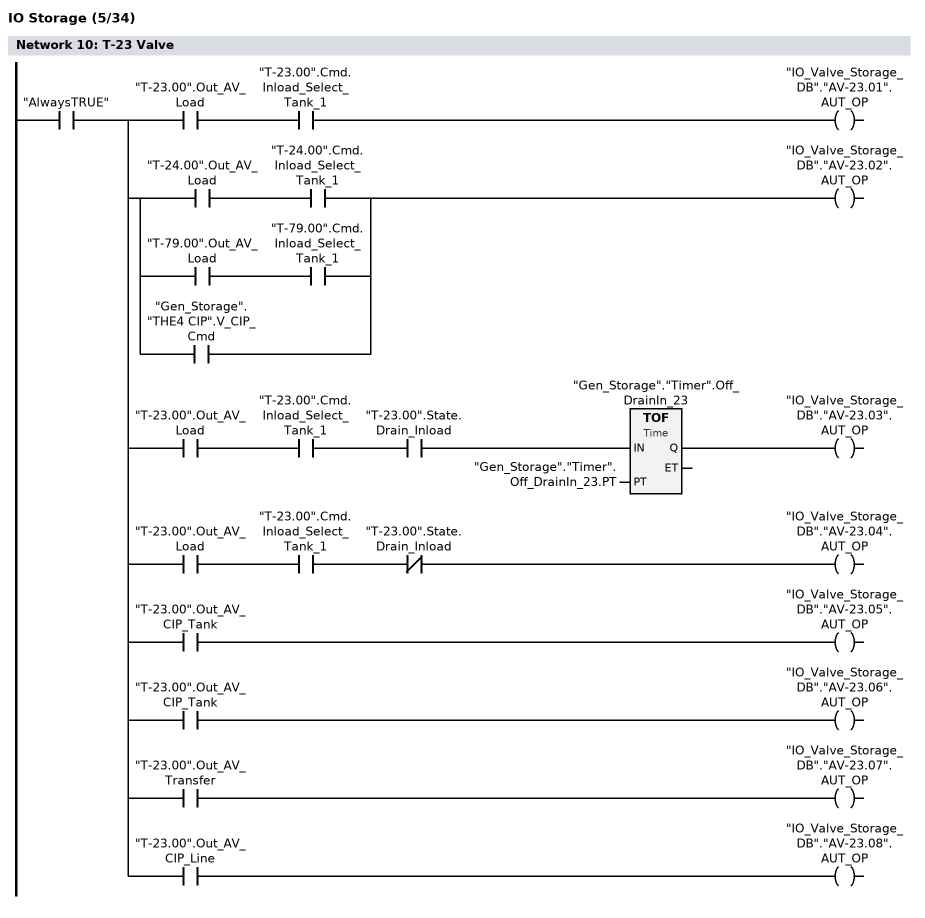
   RUNG wire#powerrail
      Contact( "AlwaysTRUE" )
      wire#w1
      Contact( "T-23.00".Out_AV_Load )
      Contact( "T-23.00".Cmd.Inload_Select_Tank_1 )
      Coil( "IO_Valve_Storage_DB"."AV-23.01".AUT_OP )
   END_RUNG
   RUNG wire#w1
      Contact( "T-24.00".Out_AV_Load )
      Contact( "T-24.00".Cmd.Inload_Select_Tank_1 )
      wire#w2
      Coil( "IO_Valve_Storage_DB"."AV-23.02".AUT_OP )
   END_RUNG
   RUNG wire#w1
      Contact( "T-79.00".Out_AV_Load )
      Contact( "T-79.00".Cmd.Inload_Select_Tank_1 )
   END_RUNG wire#w2
   RUNG wire#w1
      Contact( "Gen_Storage"."THE4 CIP".V_CIP_Cmd )
   END_RUNG wire#w2
   RUNG wire#w1
      Contact( "T-23.00".Out_AV_Load )
      Contact( "T-23.00".Cmd.Inload_Select_Tank_1 )
      Contact( "T-23.00".State.Drain_Inload )
      { S7_Templates := "time_type := Time" } "Gen_Storage"."Timer".Off_DrainIn_23.TOF(pt := "Gen_Storage"."Timer".Off_DrainIn_23.PT, et =>)
      Coil( "IO_Valve_Storage_DB"."AV-23.03".AUT_OP )
   END_RUNG
   RUNG wire#w1
      Contact( "T-23.00".Out_AV_Load )
      Contact( "T-23.00".Cmd.Inload_Select_Tank_1 )
      I_Contact( "T-23.00".State.Drain_Inload )
      Coil( "IO_Valve_Storage_DB"."AV-23.04".AUT_OP )
   END_RUNG
   RUNG wire#w1
      Contact( "T-23.00".Out_AV_CIP_Tank )
      Coil( "IO_Valve_Storage_DB"."AV-23.05".AUT_OP )
   END_RUNG
   RUNG wire#w1
      Contact( "T-23.00".Out_AV_CIP_Tank )
      Coil( "IO_Valve_Storage_DB"."AV-23.06".AUT_OP )
   END_RUNG
   RUNG wire#w1
      Contact( "T-23.00".Out_AV_Transfer )
      Coil( "IO_Valve_Storage_DB"."AV-23.07".AUT_OP )
   END_RUNG
   RUNG wire#w1
      Contact( "T-23.00".Out_AV_CIP_Line )
      Coil( "IO_Valve_Storage_DB"."AV-23.08".AUT_OP )
   END_RUNG
   // the same network as SCL:
   "IO_Valve_Storage_DB"."AV-23.01".AUT_OP := "AlwaysTRUE" AND "T-23.00".Out_AV_Load AND "T-23.00".Cmd.Inload_Select_Tank_1;
   "IO_Valve_Storage_DB"."AV-23.02".AUT_OP := "AlwaysTRUE" AND (("T-24.00".Out_AV_Load AND "T-24.00".Cmd.Inload_Select_Tank_1) OR ("T-79.00".Out_AV_Load AND "T-79.00".Cmd.Inload_Select_Tank_1) OR "Gen_Storage"."THE4 CIP".V_CIP_Cmd);
   "Gen_Storage"."Timer".Off_DrainIn_23.TOF(IN := "AlwaysTRUE" AND "T-23.00".Out_AV_Load AND "T-23.00".Cmd.Inload_Select_Tank_1 AND "T-23.00".State.Drain_Inload,
                           PT := "Gen_Storage"."Timer".Off_DrainIn_23.PT);
   "IO_Valve_Storage_DB"."AV-23.03".AUT_OP := "Gen_Storage"."Timer".Off_DrainIn_23.Q;
   "IO_Valve_Storage_DB"."AV-23.04".AUT_OP := "AlwaysTRUE" AND "T-23.00".Out_AV_Load AND "T-23.00".Cmd.Inload_Select_Tank_1 AND NOT "T-23.00".State.Drain_Inload;
   "IO_Valve_Storage_DB"."AV-23.05".AUT_OP := "AlwaysTRUE" AND "T-23.00".Out_AV_CIP_Tank;
   "IO_Valve_Storage_DB"."AV-23.06".AUT_OP := "AlwaysTRUE" AND "T-23.00".Out_AV_CIP_Tank;
   "IO_Valve_Storage_DB"."AV-23.07".AUT_OP := "AlwaysTRUE" AND "T-23.00".Out_AV_Transfer;
   "IO_Valve_Storage_DB"."AV-23.08".AUT_OP := "AlwaysTRUE" AND "T-23.00".Out_AV_CIP_Line;
END_REGION

REGION Network 12: T-24.00 ST-07
   // Inload 1 : THE 4
   // Inload 2 : THE 1
   // Inload 3 : THE 5
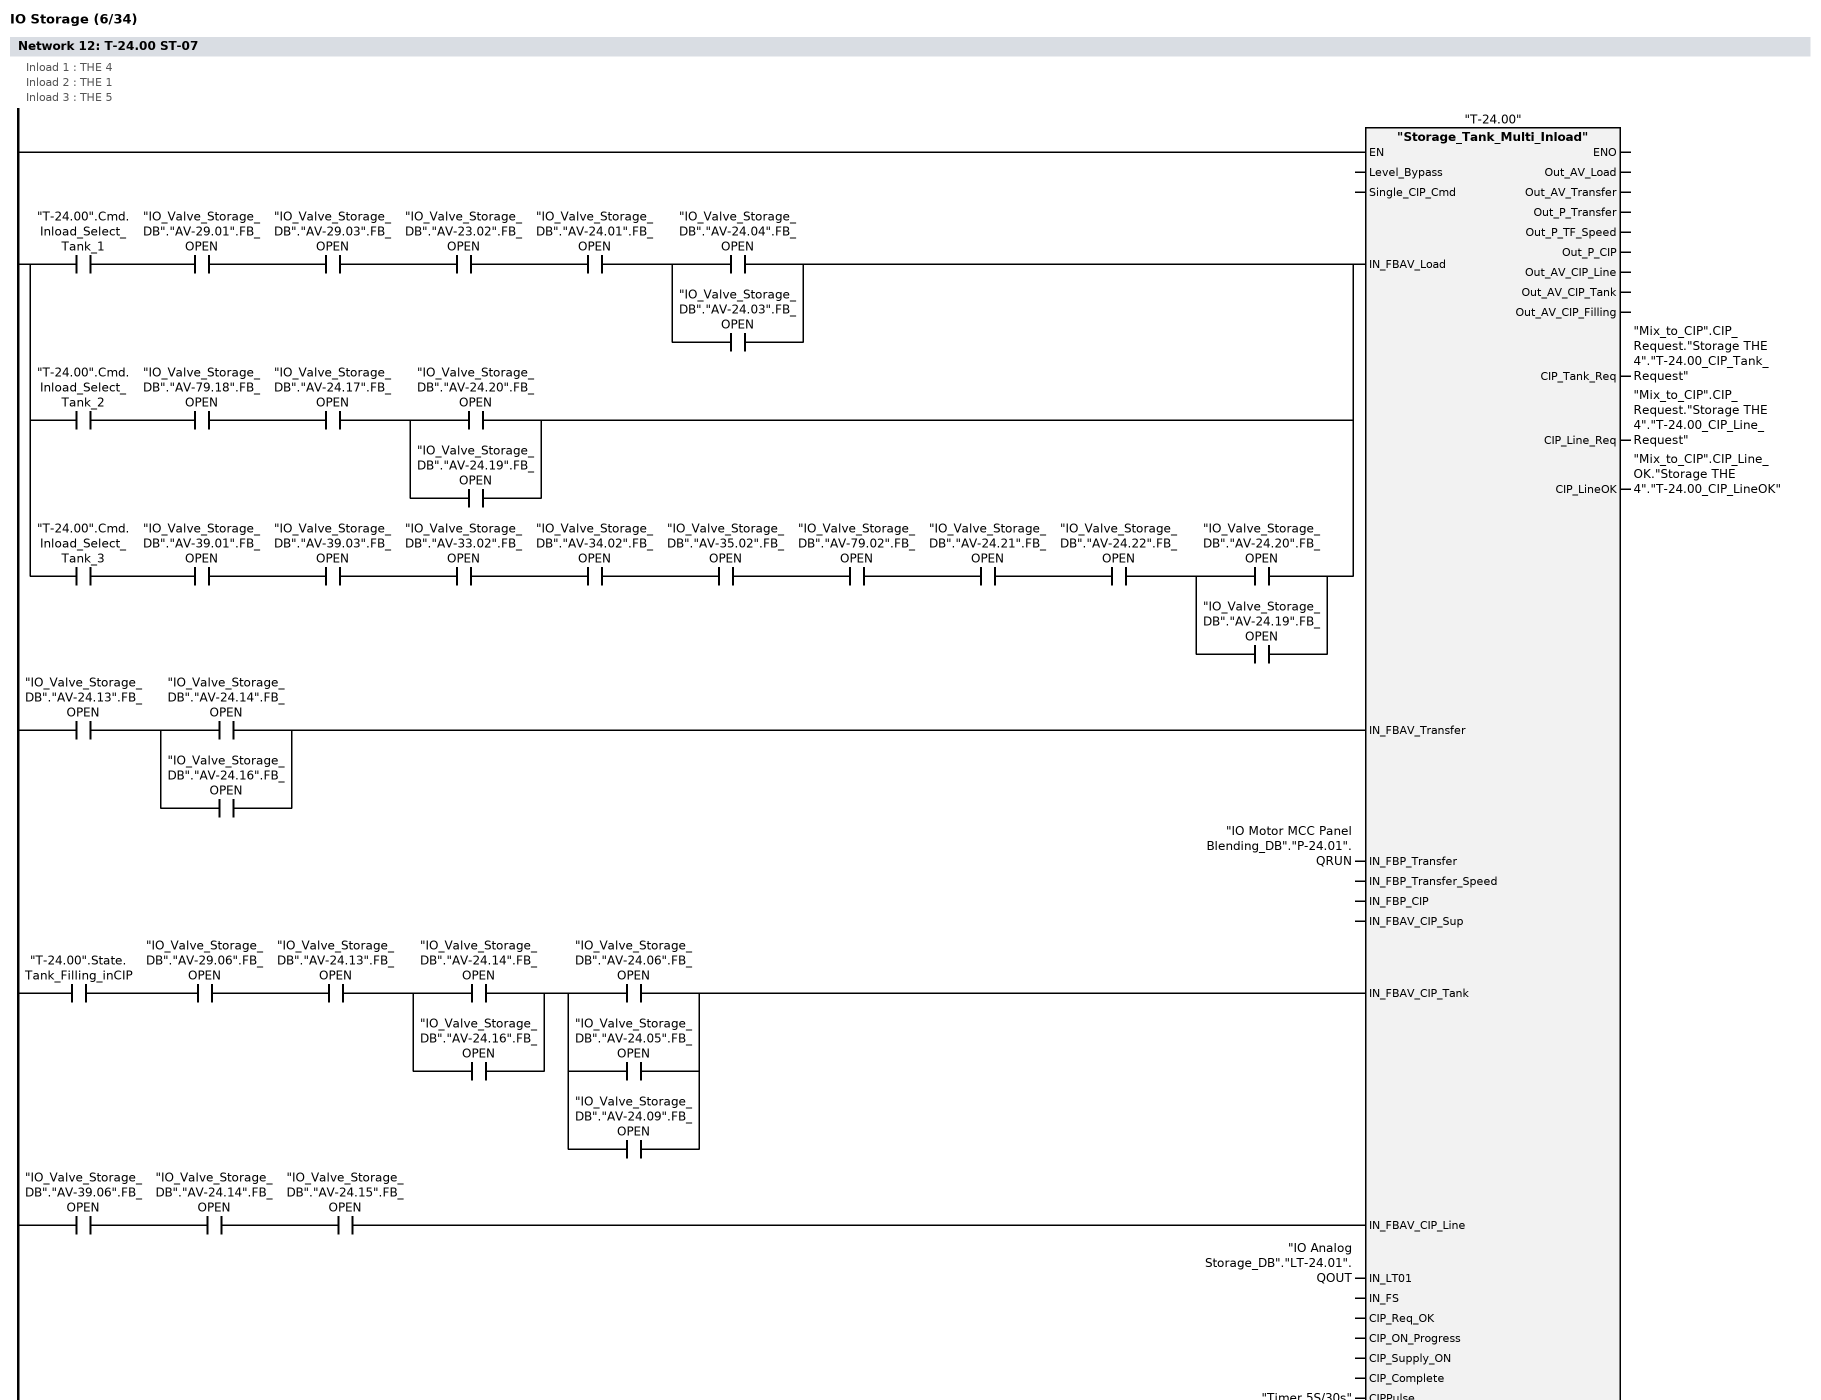
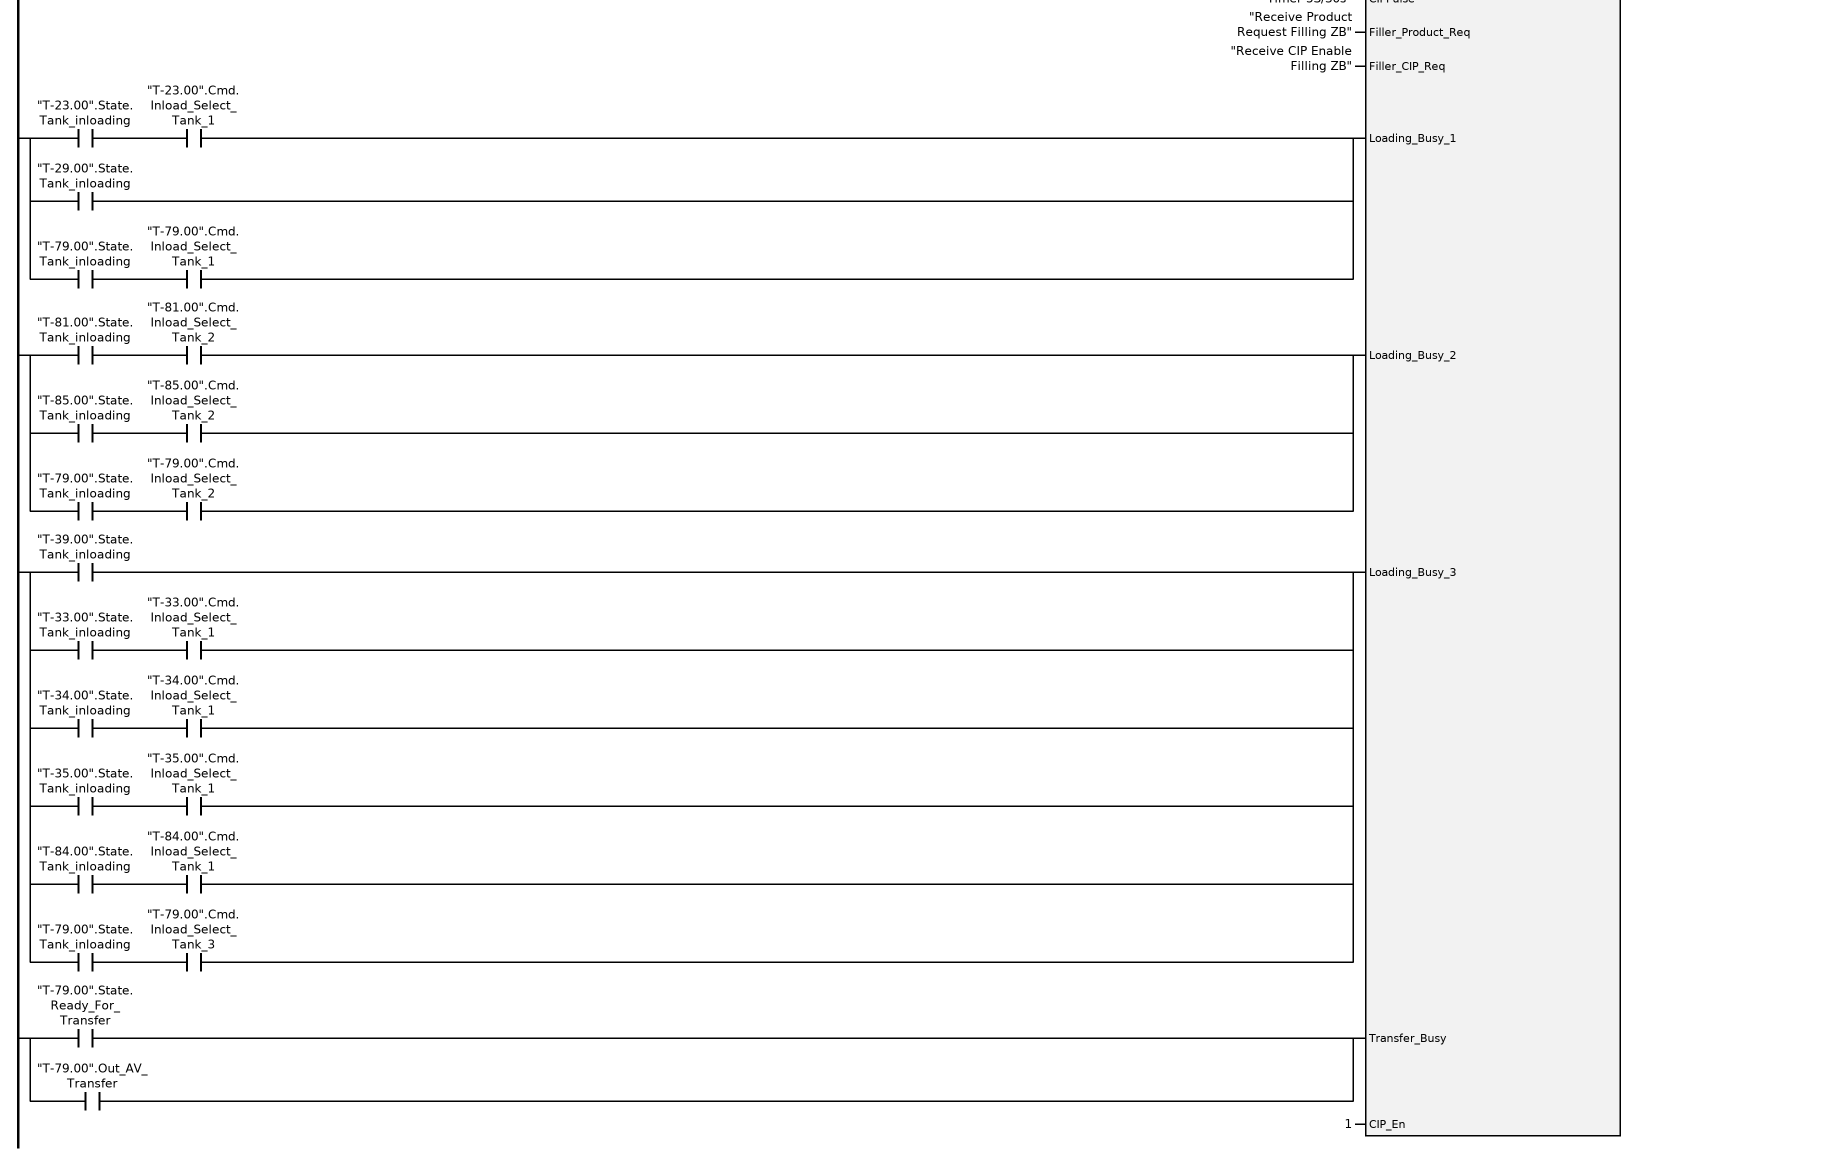
   RUNG wire#powerrail
      "T-24.00"(IN_FBAV_Load := wire#w4, IN_FBAV_Transfer := wire#w6, IN_FBAV_CIP_Tank := wire#w9, IN_FBAV_CIP_Line := wire#w10, Loading_Busy_1 := wire#w11, Loading_Busy_2 := wire#w12, Loading_Busy_3 := wire#w13, Transfer_Busy := wire#w14, Level_Bypass :=, Single_CIP_Cmd :=, IN_FBP_Transfer := "IO Motor MCC Panel Blending_DB"."P-24.01".QRUN, IN_FBP_Transfer_Speed :=, IN_FBP_CIP :=, IN_FBAV_CIP_Sup :=, IN_LT01 := "IO Analog Storage_DB"."LT-24.01".QOUT, IN_FS :=, CIP_Req_OK :=, CIP_ON_Progress :=, CIP_Supply_ON :=, CIP_Complete :=, CIPPulse := "Timer 5S/30s", Filler_Product_Req := "Receive Product Request Filling ZB", Filler_CIP_Req := "Receive CIP Enable Filling ZB", CIP_En := 1, Out_AV_Load =>, Out_AV_Transfer =>, Out_P_Transfer =>, Out_P_TF_Speed =>, Out_P_CIP =>, Out_AV_CIP_Line =>, Out_AV_CIP_Tank =>, Out_AV_CIP_Filling =>, CIP_Tank_Req => "Mix_to_CIP".CIP_Request."Storage THE 4"."T-24.00_CIP_Tank_Request", CIP_Line_Req => "Mix_to_CIP".CIP_Request."Storage THE 4"."T-24.00_CIP_Line_Request", CIP_LineOK => "Mix_to_CIP".CIP_Line_OK."Storage THE 4"."T-24.00_CIP_LineOK")
   END_RUNG
   RUNG wire#powerrail
      Contact( "T-24.00".Cmd.Inload_Select_Tank_1 )
      Contact( "IO_Valve_Storage_DB"."AV-29.01".FB_OPEN )
      Contact( "IO_Valve_Storage_DB"."AV-29.03".FB_OPEN )
      Contact( "IO_Valve_Storage_DB"."AV-23.02".FB_OPEN )
      Contact( "IO_Valve_Storage_DB"."AV-24.01".FB_OPEN )
      wire#w1
      Contact( "IO_Valve_Storage_DB"."AV-24.04".FB_OPEN )
   END_RUNG wire#w4
   RUNG wire#w1
      Contact( "IO_Valve_Storage_DB"."AV-24.03".FB_OPEN )
   END_RUNG wire#w4
   RUNG wire#powerrail
      Contact( "T-24.00".Cmd.Inload_Select_Tank_2 )
      Contact( "IO_Valve_Storage_DB"."AV-79.18".FB_OPEN )
      Contact( "IO_Valve_Storage_DB"."AV-24.17".FB_OPEN )
      wire#w2
      Contact( "IO_Valve_Storage_DB"."AV-24.20".FB_OPEN )
   END_RUNG wire#w4
   RUNG wire#w2
      Contact( "IO_Valve_Storage_DB"."AV-24.19".FB_OPEN )
   END_RUNG wire#w4
   RUNG wire#powerrail
      Contact( "T-24.00".Cmd.Inload_Select_Tank_3 )
      Contact( "IO_Valve_Storage_DB"."AV-39.01".FB_OPEN )
      Contact( "IO_Valve_Storage_DB"."AV-39.03".FB_OPEN )
      Contact( "IO_Valve_Storage_DB"."AV-33.02".FB_OPEN )
      Contact( "IO_Valve_Storage_DB"."AV-34.02".FB_OPEN )
      Contact( "IO_Valve_Storage_DB"."AV-35.02".FB_OPEN )
      Contact( "IO_Valve_Storage_DB"."AV-79.02".FB_OPEN )
      Contact( "IO_Valve_Storage_DB"."AV-24.21".FB_OPEN )
      Contact( "IO_Valve_Storage_DB"."AV-24.22".FB_OPEN )
      wire#w3
      Contact( "IO_Valve_Storage_DB"."AV-24.20".FB_OPEN )
   END_RUNG wire#w4
   RUNG wire#w3
      Contact( "IO_Valve_Storage_DB"."AV-24.19".FB_OPEN )
   END_RUNG wire#w4
   RUNG wire#powerrail
      Contact( "IO_Valve_Storage_DB"."AV-24.13".FB_OPEN )
      wire#w5
      Contact( "IO_Valve_Storage_DB"."AV-24.14".FB_OPEN )
   END_RUNG wire#w6
   RUNG wire#w5
      Contact( "IO_Valve_Storage_DB"."AV-24.16".FB_OPEN )
   END_RUNG wire#w6
   RUNG wire#powerrail
      Contact( "T-24.00".State.Tank_Filling_inCIP )
      Contact( "IO_Valve_Storage_DB"."AV-29.06".FB_OPEN )
      Contact( "IO_Valve_Storage_DB"."AV-24.13".FB_OPEN )
      wire#w7
      Contact( "IO_Valve_Storage_DB"."AV-24.14".FB_OPEN )
      wire#w8
      Contact( "IO_Valve_Storage_DB"."AV-24.06".FB_OPEN )
   END_RUNG wire#w9
   RUNG wire#w7
      Contact( "IO_Valve_Storage_DB"."AV-24.16".FB_OPEN )
   END_RUNG wire#w8
   RUNG wire#w8
      Contact( "IO_Valve_Storage_DB"."AV-24.05".FB_OPEN )
   END_RUNG wire#w9
   RUNG wire#w8
      Contact( "IO_Valve_Storage_DB"."AV-24.09".FB_OPEN )
   END_RUNG wire#w9
   RUNG wire#powerrail
      Contact( "IO_Valve_Storage_DB"."AV-39.06".FB_OPEN )
      Contact( "IO_Valve_Storage_DB"."AV-24.14".FB_OPEN )
      Contact( "IO_Valve_Storage_DB"."AV-24.15".FB_OPEN )
   END_RUNG wire#w10
   RUNG wire#powerrail
      Contact( "T-23.00".State.Tank_inloading )
      Contact( "T-23.00".Cmd.Inload_Select_Tank_1 )
   END_RUNG wire#w11
   RUNG wire#powerrail
      Contact( "T-29.00".State.Tank_inloading )
   END_RUNG wire#w11
   RUNG wire#powerrail
      Contact( "T-79.00".State.Tank_inloading )
      Contact( "T-79.00".Cmd.Inload_Select_Tank_1 )
   END_RUNG wire#w11
   RUNG wire#powerrail
      Contact( "T-81.00".State.Tank_inloading )
      Contact( "T-81.00".Cmd.Inload_Select_Tank_2 )
   END_RUNG wire#w12
   RUNG wire#powerrail
      Contact( "T-85.00".State.Tank_inloading )
      Contact( "T-85.00".Cmd.Inload_Select_Tank_2 )
   END_RUNG wire#w12
   RUNG wire#powerrail
      Contact( "T-79.00".State.Tank_inloading )
      Contact( "T-79.00".Cmd.Inload_Select_Tank_2 )
   END_RUNG wire#w12
   RUNG wire#powerrail
      Contact( "T-39.00".State.Tank_inloading )
   END_RUNG wire#w13
   RUNG wire#powerrail
      Contact( "T-33.00".State.Tank_inloading )
      Contact( "T-33.00".Cmd.Inload_Select_Tank_1 )
   END_RUNG wire#w13
   RUNG wire#powerrail
      Contact( "T-34.00".State.Tank_inloading )
      Contact( "T-34.00".Cmd.Inload_Select_Tank_1 )
   END_RUNG wire#w13
   RUNG wire#powerrail
      Contact( "T-35.00".State.Tank_inloading )
      Contact( "T-35.00".Cmd.Inload_Select_Tank_1 )
   END_RUNG wire#w13
   RUNG wire#powerrail
      Contact( "T-84.00".State.Tank_inloading )
      Contact( "T-84.00".Cmd.Inload_Select_Tank_1 )
   END_RUNG wire#w13
   RUNG wire#powerrail
      Contact( "T-79.00".State.Tank_inloading )
      Contact( "T-79.00".Cmd.Inload_Select_Tank_3 )
   END_RUNG wire#w13
   RUNG wire#powerrail
      Contact( "T-79.00".State.Ready_For_Transfer )
   END_RUNG wire#w14
   RUNG wire#powerrail
      Contact( "T-79.00".Out_AV_Transfer )
   END_RUNG wire#w14
   // the same network as SCL:
   "T-24.00"(IN_FBAV_Load := ("T-24.00".Cmd.Inload_Select_Tank_1 AND "IO_Valve_Storage_DB"."AV-29.01".FB_OPEN AND "IO_Valve_Storage_DB"."AV-29.03".FB_OPEN AND "IO_Valve_Storage_DB"."AV-23.02".FB_OPEN AND "IO_Valve_Storage_DB"."AV-24.01".FB_OPEN AND ("IO_Valve_Storage_DB"."AV-24.04".FB_OPEN OR "IO_Valve_Storage_DB"."AV-24.03".FB_OPEN)) OR ("T-24.00".Cmd.Inload_Select_Tank_2 AND "IO_Valve_Storage_DB"."AV-79.18".FB_OPEN AND "IO_Valve_Storage_DB"."AV-24.17".FB_OPEN AND ("IO_Valve_Storage_DB"."AV-24.20".FB_OPEN OR "IO_Valve_Storage_DB"."AV-24.19".FB_OPEN)) OR ("T-24.00".Cmd.Inload_Select_Tank_3 AND "IO_Valve_Storage_DB"."AV-39.01".FB_OPEN AND "IO_Valve_Storage_DB"."AV-39.03".FB_OPEN AND "IO_Valve_Storage_DB"."AV-33.02".FB_OPEN AND "IO_Valve_Storage_DB"."AV-34.02".FB_OPEN AND "IO_Valve_Storage_DB"."AV-35.02".FB_OPEN AND "IO_Valve_Storage_DB"."AV-79.02".FB_OPEN AND "IO_Valve_Storage_DB"."AV-24.21".FB_OPEN AND "IO_Valve_Storage_DB"."AV-24.22".FB_OPEN AND ("IO_Valve_Storage_DB"."AV-24.20".FB_OPEN OR "IO_Valve_Storage_DB"."AV-24.19".FB_OPEN)),   // "Storage_Tank_Multi_Inload"
             IN_FBAV_Transfer := "IO_Valve_Storage_DB"."AV-24.13".FB_OPEN AND ("IO_Valve_Storage_DB"."AV-24.14".FB_OPEN OR "IO_Valve_Storage_DB"."AV-24.16".FB_OPEN),
             IN_FBP_Transfer := "IO Motor MCC Panel Blending_DB"."P-24.01".QRUN,
             IN_FBAV_CIP_Tank := "T-24.00".State.Tank_Filling_inCIP AND "IO_Valve_Storage_DB"."AV-29.06".FB_OPEN AND "IO_Valve_Storage_DB"."AV-24.13".FB_OPEN AND ("IO_Valve_Storage_DB"."AV-24.14".FB_OPEN OR "IO_Valve_Storage_DB"."AV-24.16".FB_OPEN) AND ("IO_Valve_Storage_DB"."AV-24.06".FB_OPEN OR "IO_Valve_Storage_DB"."AV-24.05".FB_OPEN OR "IO_Valve_Storage_DB"."AV-24.09".FB_OPEN),
             IN_FBAV_CIP_Line := "IO_Valve_Storage_DB"."AV-39.06".FB_OPEN AND "IO_Valve_Storage_DB"."AV-24.14".FB_OPEN AND "IO_Valve_Storage_DB"."AV-24.15".FB_OPEN,
             IN_LT01 := "IO Analog Storage_DB"."LT-24.01".QOUT,
             CIPPulse := "Timer 5S/30s",
             Filler_Product_Req := "Receive Product Request Filling ZB",
             Filler_CIP_Req := "Receive CIP Enable Filling ZB",
             Loading_Busy_1 := ("T-23.00".State.Tank_inloading AND "T-23.00".Cmd.Inload_Select_Tank_1) OR "T-29.00".State.Tank_inloading OR ("T-79.00".State.Tank_inloading AND "T-79.00".Cmd.Inload_Select_Tank_1),
             Loading_Busy_2 := ("T-81.00".State.Tank_inloading AND "T-81.00".Cmd.Inload_Select_Tank_2) OR ("T-85.00".State.Tank_inloading AND "T-85.00".Cmd.Inload_Select_Tank_2) OR ("T-79.00".State.Tank_inloading AND "T-79.00".Cmd.Inload_Select_Tank_2),
             Loading_Busy_3 := "T-39.00".State.Tank_inloading OR ("T-33.00".State.Tank_inloading AND "T-33.00".Cmd.Inload_Select_Tank_1) OR ("T-34.00".State.Tank_inloading AND "T-34.00".Cmd.Inload_Select_Tank_1) OR ("T-35.00".State.Tank_inloading AND "T-35.00".Cmd.Inload_Select_Tank_1) OR ("T-84.00".State.Tank_inloading AND "T-84.00".Cmd.Inload_Select_Tank_1) OR ("T-79.00".State.Tank_inloading AND "T-79.00".Cmd.Inload_Select_Tank_3),
             Transfer_Busy := "T-79.00".State.Ready_For_Transfer OR "T-79.00".Out_AV_Transfer,
             CIP_En := 1,
             CIP_Tank_Req => "Mix_to_CIP".CIP_Request."Storage THE 4"."T-24.00_CIP_Tank_Request",
             CIP_Line_Req => "Mix_to_CIP".CIP_Request."Storage THE 4"."T-24.00_CIP_Line_Request",
             CIP_LineOK => "Mix_to_CIP".CIP_Line_OK."Storage THE 4"."T-24.00_CIP_LineOK");
END_REGION

REGION Network 13: T-24 CIP Interlock
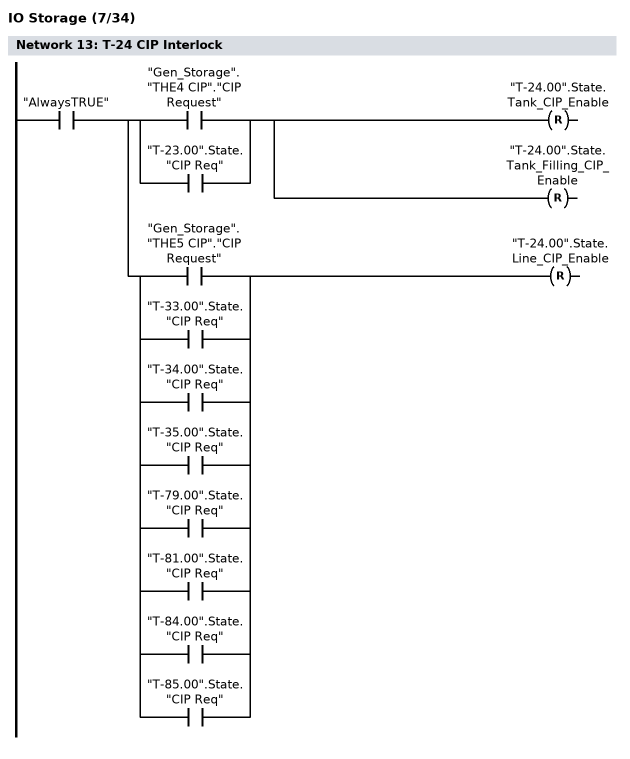
   RUNG wire#powerrail
      Contact( "AlwaysTRUE" )
      wire#w1
      Contact( "Gen_Storage"."THE4 CIP"."CIP Request" )
      wire#w2
      R_Coil( "T-24.00".State.Tank_CIP_Enable )
   END_RUNG
   RUNG wire#w1
      Contact( "T-23.00".State."CIP Req" )
   END_RUNG wire#w2
   RUNG wire#w2
      R_Coil( "T-24.00".State.Tank_Filling_CIP_Enable )
   END_RUNG
   RUNG wire#w1
      Contact( "Gen_Storage"."THE5 CIP"."CIP Request" )
      wire#w3
      R_Coil( "T-24.00".State.Line_CIP_Enable )
   END_RUNG
   RUNG wire#w1
      Contact( "T-33.00".State."CIP Req" )
   END_RUNG wire#w3
   RUNG wire#w1
      Contact( "T-34.00".State."CIP Req" )
   END_RUNG wire#w3
   RUNG wire#w1
      Contact( "T-35.00".State."CIP Req" )
   END_RUNG wire#w3
   RUNG wire#w1
      Contact( "T-79.00".State."CIP Req" )
   END_RUNG wire#w3
   RUNG wire#w1
      Contact( "T-81.00".State."CIP Req" )
   END_RUNG wire#w3
   RUNG wire#w1
      Contact( "T-84.00".State."CIP Req" )
   END_RUNG wire#w3
   RUNG wire#w1
      Contact( "T-85.00".State."CIP Req" )
   END_RUNG wire#w3
   // the same network as SCL:
   IF "AlwaysTRUE" AND ("Gen_Storage"."THE4 CIP"."CIP Request" OR "T-23.00".State."CIP Req") THEN
       "T-24.00".State.Tank_CIP_Enable := FALSE;
       "T-24.00".State.Tank_Filling_CIP_Enable := FALSE;
   END_IF;
   IF "AlwaysTRUE" AND ("Gen_Storage"."THE5 CIP"."CIP Request" OR "T-33.00".State."CIP Req" OR "T-34.00".State."CIP Req" OR "T-35.00".State."CIP Req" OR "T-79.00".State."CIP Req" OR "T-81.00".State."CIP Req" OR "T-84.00".State."CIP Req" OR "T-85.00".State."CIP Req") THEN
       "T-24.00".State.Line_CIP_Enable := FALSE;
   END_IF;
END_REGION

REGION Network 14: T-24 Valve
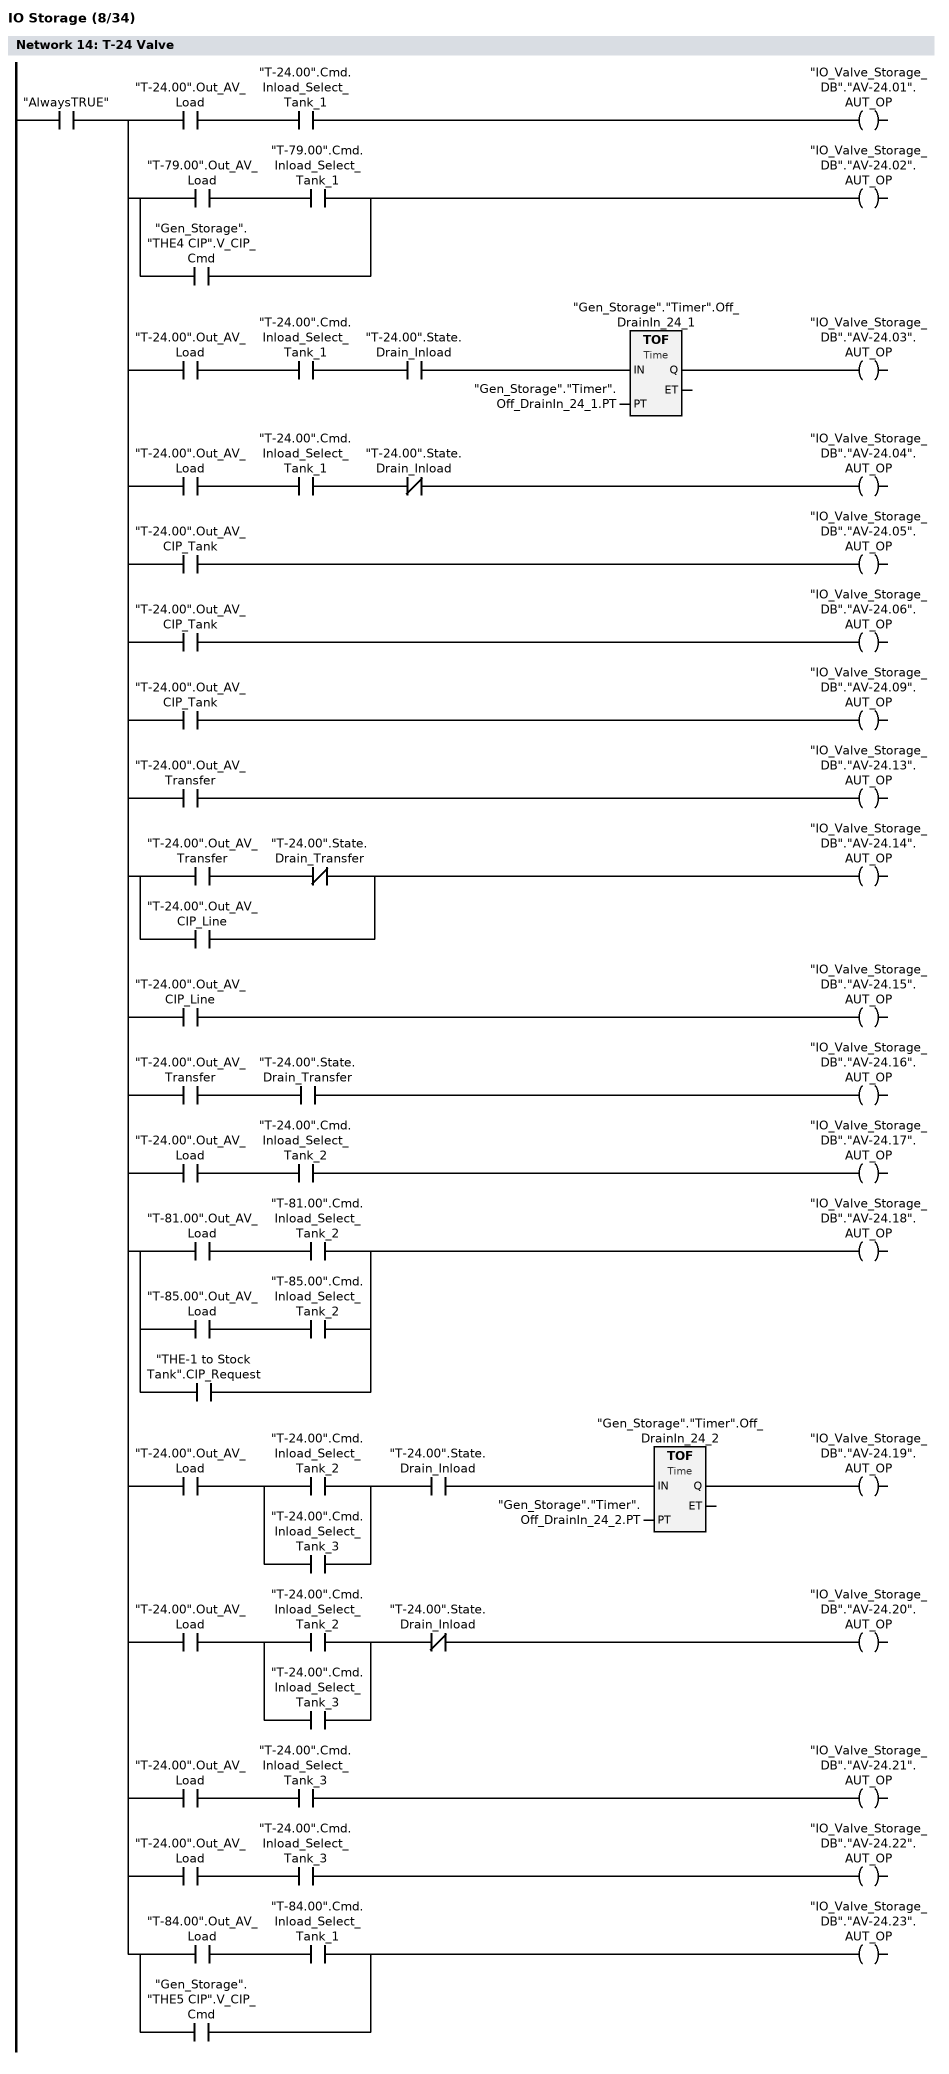
   RUNG wire#powerrail
      Contact( "AlwaysTRUE" )
      wire#w1
      Contact( "T-24.00".Out_AV_Load )
      Contact( "T-24.00".Cmd.Inload_Select_Tank_1 )
      Coil( "IO_Valve_Storage_DB"."AV-24.01".AUT_OP )
   END_RUNG
   RUNG wire#w1
      Contact( "T-79.00".Out_AV_Load )
      Contact( "T-79.00".Cmd.Inload_Select_Tank_1 )
      wire#w2
      Coil( "IO_Valve_Storage_DB"."AV-24.02".AUT_OP )
   END_RUNG
   RUNG wire#w1
      Contact( "Gen_Storage"."THE4 CIP".V_CIP_Cmd )
   END_RUNG wire#w2
   RUNG wire#w1
      Contact( "T-24.00".Out_AV_Load )
      Contact( "T-24.00".Cmd.Inload_Select_Tank_1 )
      Contact( "T-24.00".State.Drain_Inload )
      { S7_Templates := "time_type := Time" } "Gen_Storage"."Timer".Off_DrainIn_24_1.TOF(pt := "Gen_Storage"."Timer".Off_DrainIn_24_1.PT, et =>)
      Coil( "IO_Valve_Storage_DB"."AV-24.03".AUT_OP )
   END_RUNG
   RUNG wire#w1
      Contact( "T-24.00".Out_AV_Load )
      Contact( "T-24.00".Cmd.Inload_Select_Tank_1 )
      I_Contact( "T-24.00".State.Drain_Inload )
      Coil( "IO_Valve_Storage_DB"."AV-24.04".AUT_OP )
   END_RUNG
   RUNG wire#w1
      Contact( "T-24.00".Out_AV_CIP_Tank )
      Coil( "IO_Valve_Storage_DB"."AV-24.05".AUT_OP )
   END_RUNG
   RUNG wire#w1
      Contact( "T-24.00".Out_AV_CIP_Tank )
      Coil( "IO_Valve_Storage_DB"."AV-24.06".AUT_OP )
   END_RUNG
   RUNG wire#w1
      Contact( "T-24.00".Out_AV_CIP_Tank )
      Coil( "IO_Valve_Storage_DB"."AV-24.09".AUT_OP )
   END_RUNG
   RUNG wire#w1
      Contact( "T-24.00".Out_AV_Transfer )
      Coil( "IO_Valve_Storage_DB"."AV-24.13".AUT_OP )
   END_RUNG
   RUNG wire#w1
      Contact( "T-24.00".Out_AV_Transfer )
      I_Contact( "T-24.00".State.Drain_Transfer )
      wire#w3
      Coil( "IO_Valve_Storage_DB"."AV-24.14".AUT_OP )
   END_RUNG
   RUNG wire#w1
      Contact( "T-24.00".Out_AV_CIP_Line )
   END_RUNG wire#w3
   RUNG wire#w1
      Contact( "T-24.00".Out_AV_CIP_Line )
      Coil( "IO_Valve_Storage_DB"."AV-24.15".AUT_OP )
   END_RUNG
   RUNG wire#w1
      Contact( "T-24.00".Out_AV_Transfer )
      Contact( "T-24.00".State.Drain_Transfer )
      Coil( "IO_Valve_Storage_DB"."AV-24.16".AUT_OP )
   END_RUNG
   RUNG wire#w1
      Contact( "T-24.00".Out_AV_Load )
      Contact( "T-24.00".Cmd.Inload_Select_Tank_2 )
      Coil( "IO_Valve_Storage_DB"."AV-24.17".AUT_OP )
   END_RUNG
   RUNG wire#w1
      Contact( "T-81.00".Out_AV_Load )
      Contact( "T-81.00".Cmd.Inload_Select_Tank_2 )
      wire#w4
      Coil( "IO_Valve_Storage_DB"."AV-24.18".AUT_OP )
   END_RUNG
   RUNG wire#w1
      Contact( "T-85.00".Out_AV_Load )
      Contact( "T-85.00".Cmd.Inload_Select_Tank_2 )
   END_RUNG wire#w4
   RUNG wire#w1
      Contact( "THE-1 to Stock Tank".CIP_Request )
   END_RUNG wire#w4
   RUNG wire#w1
      Contact( "T-24.00".Out_AV_Load )
      wire#w5
      Contact( "T-24.00".Cmd.Inload_Select_Tank_2 )
      wire#w6
      Contact( "T-24.00".State.Drain_Inload )
      { S7_Templates := "time_type := Time" } "Gen_Storage"."Timer".Off_DrainIn_24_2.TOF(pt := "Gen_Storage"."Timer".Off_DrainIn_24_2.PT, et =>)
      Coil( "IO_Valve_Storage_DB"."AV-24.19".AUT_OP )
   END_RUNG
   RUNG wire#w5
      Contact( "T-24.00".Cmd.Inload_Select_Tank_3 )
   END_RUNG wire#w6
   RUNG wire#w1
      Contact( "T-24.00".Out_AV_Load )
      wire#w7
      Contact( "T-24.00".Cmd.Inload_Select_Tank_2 )
      wire#w8
      I_Contact( "T-24.00".State.Drain_Inload )
      Coil( "IO_Valve_Storage_DB"."AV-24.20".AUT_OP )
   END_RUNG
   RUNG wire#w7
      Contact( "T-24.00".Cmd.Inload_Select_Tank_3 )
   END_RUNG wire#w8
   RUNG wire#w1
      Contact( "T-24.00".Out_AV_Load )
      Contact( "T-24.00".Cmd.Inload_Select_Tank_3 )
      Coil( "IO_Valve_Storage_DB"."AV-24.21".AUT_OP )
   END_RUNG
   RUNG wire#w1
      Contact( "T-24.00".Out_AV_Load )
      Contact( "T-24.00".Cmd.Inload_Select_Tank_3 )
      Coil( "IO_Valve_Storage_DB"."AV-24.22".AUT_OP )
   END_RUNG
   RUNG wire#w1
      Contact( "T-84.00".Out_AV_Load )
      Contact( "T-84.00".Cmd.Inload_Select_Tank_1 )
      wire#w9
      Coil( "IO_Valve_Storage_DB"."AV-24.23".AUT_OP )
   END_RUNG
   RUNG wire#w1
      Contact( "Gen_Storage"."THE5 CIP".V_CIP_Cmd )
   END_RUNG wire#w9
   // the same network as SCL:
   "IO_Valve_Storage_DB"."AV-24.01".AUT_OP := "AlwaysTRUE" AND "T-24.00".Out_AV_Load AND "T-24.00".Cmd.Inload_Select_Tank_1;
   "IO_Valve_Storage_DB"."AV-24.02".AUT_OP := "AlwaysTRUE" AND (("T-79.00".Out_AV_Load AND "T-79.00".Cmd.Inload_Select_Tank_1) OR "Gen_Storage"."THE4 CIP".V_CIP_Cmd);
   "Gen_Storage"."Timer".Off_DrainIn_24_1.TOF(IN := "AlwaysTRUE" AND "T-24.00".Out_AV_Load AND "T-24.00".Cmd.Inload_Select_Tank_1 AND "T-24.00".State.Drain_Inload,
                           PT := "Gen_Storage"."Timer".Off_DrainIn_24_1.PT);
   "IO_Valve_Storage_DB"."AV-24.03".AUT_OP := "Gen_Storage"."Timer".Off_DrainIn_24_1.Q;
   "IO_Valve_Storage_DB"."AV-24.04".AUT_OP := "AlwaysTRUE" AND "T-24.00".Out_AV_Load AND "T-24.00".Cmd.Inload_Select_Tank_1 AND NOT "T-24.00".State.Drain_Inload;
   "IO_Valve_Storage_DB"."AV-24.05".AUT_OP := "AlwaysTRUE" AND "T-24.00".Out_AV_CIP_Tank;
   "IO_Valve_Storage_DB"."AV-24.06".AUT_OP := "AlwaysTRUE" AND "T-24.00".Out_AV_CIP_Tank;
   "IO_Valve_Storage_DB"."AV-24.09".AUT_OP := "AlwaysTRUE" AND "T-24.00".Out_AV_CIP_Tank;
   "IO_Valve_Storage_DB"."AV-24.13".AUT_OP := "AlwaysTRUE" AND "T-24.00".Out_AV_Transfer;
   "IO_Valve_Storage_DB"."AV-24.14".AUT_OP := "AlwaysTRUE" AND (("T-24.00".Out_AV_Transfer AND NOT "T-24.00".State.Drain_Transfer) OR "T-24.00".Out_AV_CIP_Line);
   "IO_Valve_Storage_DB"."AV-24.15".AUT_OP := "AlwaysTRUE" AND "T-24.00".Out_AV_CIP_Line;
   "IO_Valve_Storage_DB"."AV-24.16".AUT_OP := "AlwaysTRUE" AND "T-24.00".Out_AV_Transfer AND "T-24.00".State.Drain_Transfer;
   "IO_Valve_Storage_DB"."AV-24.17".AUT_OP := "AlwaysTRUE" AND "T-24.00".Out_AV_Load AND "T-24.00".Cmd.Inload_Select_Tank_2;
   "IO_Valve_Storage_DB"."AV-24.18".AUT_OP := "AlwaysTRUE" AND (("T-81.00".Out_AV_Load AND "T-81.00".Cmd.Inload_Select_Tank_2) OR ("T-85.00".Out_AV_Load AND "T-85.00".Cmd.Inload_Select_Tank_2) OR "THE-1 to Stock Tank".CIP_Request);
   "Gen_Storage"."Timer".Off_DrainIn_24_2.TOF(IN := "AlwaysTRUE" AND "T-24.00".Out_AV_Load AND ("T-24.00".Cmd.Inload_Select_Tank_2 OR "T-24.00".Cmd.Inload_Select_Tank_3) AND "T-24.00".State.Drain_Inload,
                           PT := "Gen_Storage"."Timer".Off_DrainIn_24_2.PT);
   "IO_Valve_Storage_DB"."AV-24.19".AUT_OP := "Gen_Storage"."Timer".Off_DrainIn_24_2.Q;
   "IO_Valve_Storage_DB"."AV-24.20".AUT_OP := "AlwaysTRUE" AND "T-24.00".Out_AV_Load AND ("T-24.00".Cmd.Inload_Select_Tank_2 OR "T-24.00".Cmd.Inload_Select_Tank_3) AND NOT "T-24.00".State.Drain_Inload;
   "IO_Valve_Storage_DB"."AV-24.21".AUT_OP := "AlwaysTRUE" AND "T-24.00".Out_AV_Load AND "T-24.00".Cmd.Inload_Select_Tank_3;
   "IO_Valve_Storage_DB"."AV-24.22".AUT_OP := "AlwaysTRUE" AND "T-24.00".Out_AV_Load AND "T-24.00".Cmd.Inload_Select_Tank_3;
   "IO_Valve_Storage_DB"."AV-24.23".AUT_OP := "AlwaysTRUE" AND (("T-84.00".Out_AV_Load AND "T-84.00".Cmd.Inload_Select_Tank_1) OR "Gen_Storage"."THE5 CIP".V_CIP_Cmd);
END_REGION

REGION Network 15: Comm T-24 to THE-1
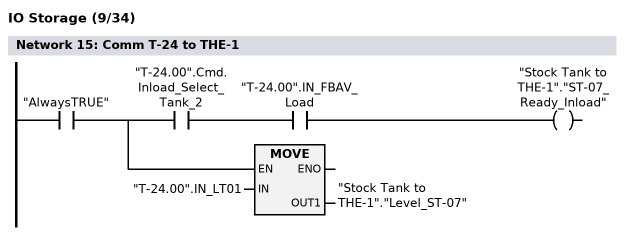
   RUNG wire#powerrail
      Contact( "AlwaysTRUE" )
      wire#w1
      Contact( "T-24.00".Cmd.Inload_Select_Tank_2 )
      Contact( "T-24.00".IN_FBAV_Load )
      Coil( "Stock Tank to THE-1"."ST-07_Ready_Inload" )
   END_RUNG
   RUNG wire#w1
      Move(in := "T-24.00".IN_LT01, out1 => "Stock Tank to THE-1"."Level_ST-07")
   END_RUNG
   // the same network as SCL:
   "Stock Tank to THE-1"."ST-07_Ready_Inload" := "AlwaysTRUE" AND "T-24.00".Cmd.Inload_Select_Tank_2 AND "T-24.00".IN_FBAV_Load;
   IF "AlwaysTRUE" THEN "Stock Tank to THE-1"."Level_ST-07" := "T-24.00".IN_LT01; END_IF;
END_REGION

REGION Network 16: Line THE 4
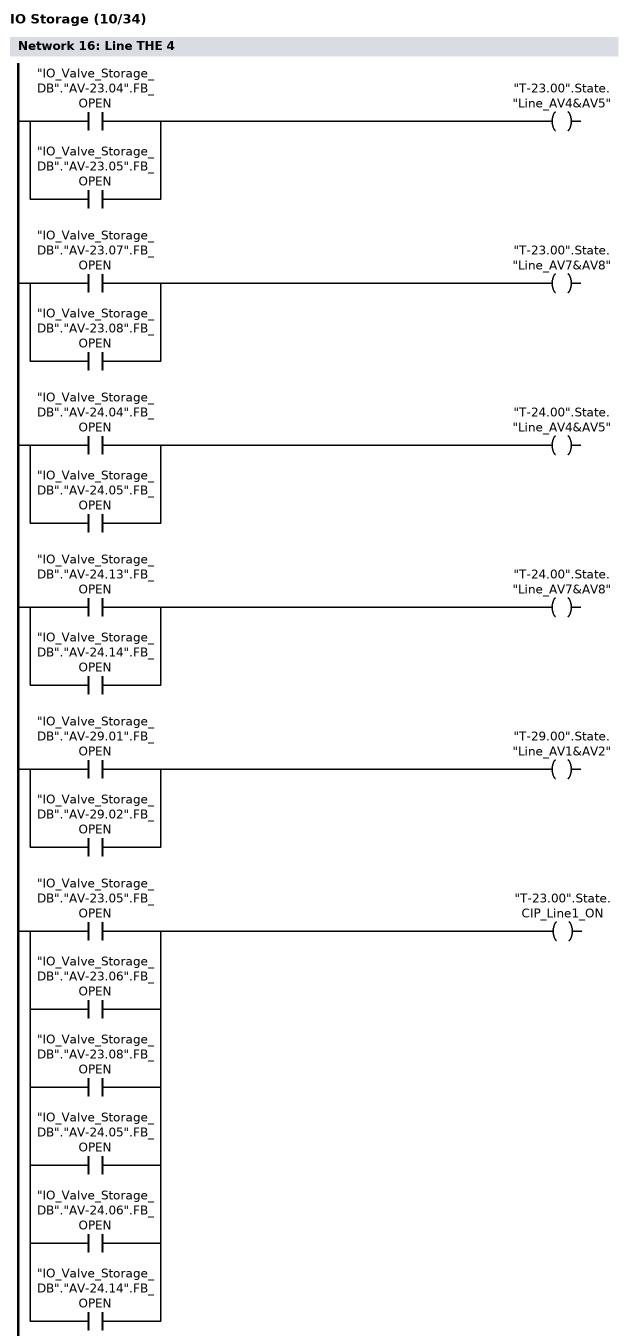
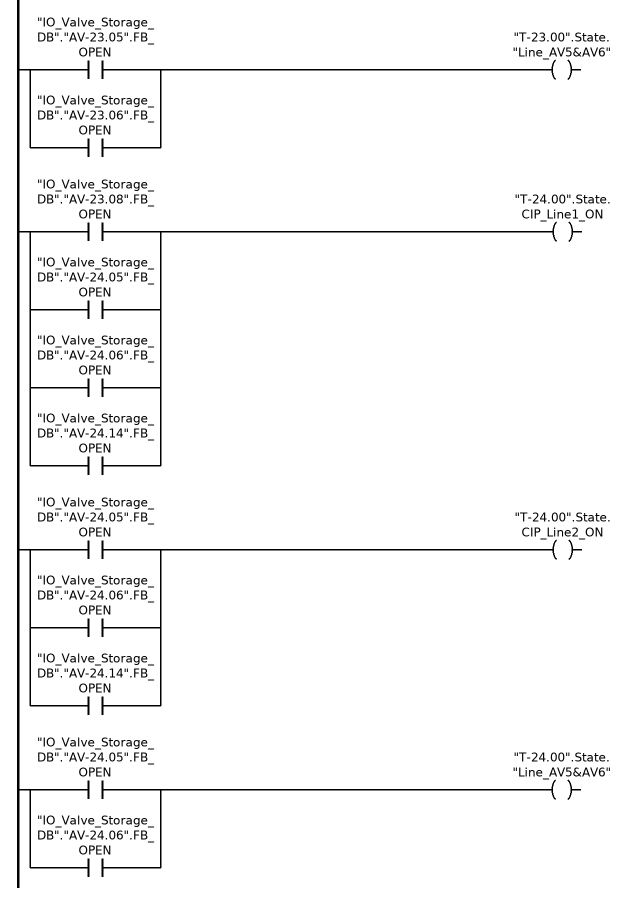
   RUNG wire#powerrail
      Contact( "IO_Valve_Storage_DB"."AV-23.04".FB_OPEN )
      wire#w1
      Coil( "T-23.00".State."Line_AV4&AV5" )
   END_RUNG
   RUNG wire#powerrail
      Contact( "IO_Valve_Storage_DB"."AV-23.05".FB_OPEN )
   END_RUNG wire#w1
   RUNG wire#powerrail
      Contact( "IO_Valve_Storage_DB"."AV-23.07".FB_OPEN )
      wire#w2
      Coil( "T-23.00".State."Line_AV7&AV8" )
   END_RUNG
   RUNG wire#powerrail
      Contact( "IO_Valve_Storage_DB"."AV-23.08".FB_OPEN )
   END_RUNG wire#w2
   RUNG wire#powerrail
      Contact( "IO_Valve_Storage_DB"."AV-24.04".FB_OPEN )
      wire#w3
      Coil( "T-24.00".State."Line_AV4&AV5" )
   END_RUNG
   RUNG wire#powerrail
      Contact( "IO_Valve_Storage_DB"."AV-24.05".FB_OPEN )
   END_RUNG wire#w3
   RUNG wire#powerrail
      Contact( "IO_Valve_Storage_DB"."AV-24.13".FB_OPEN )
      wire#w4
      Coil( "T-24.00".State."Line_AV7&AV8" )
   END_RUNG
   RUNG wire#powerrail
      Contact( "IO_Valve_Storage_DB"."AV-24.14".FB_OPEN )
   END_RUNG wire#w4
   RUNG wire#powerrail
      Contact( "IO_Valve_Storage_DB"."AV-29.01".FB_OPEN )
      wire#w5
      Coil( "T-29.00".State."Line_AV1&AV2" )
   END_RUNG
   RUNG wire#powerrail
      Contact( "IO_Valve_Storage_DB"."AV-29.02".FB_OPEN )
   END_RUNG wire#w5
   RUNG wire#powerrail
      Contact( "IO_Valve_Storage_DB"."AV-23.05".FB_OPEN )
      wire#w6
      Coil( "T-23.00".State.CIP_Line1_ON )
   END_RUNG
   RUNG wire#powerrail
      Contact( "IO_Valve_Storage_DB"."AV-23.06".FB_OPEN )
   END_RUNG wire#w6
   RUNG wire#powerrail
      Contact( "IO_Valve_Storage_DB"."AV-23.08".FB_OPEN )
   END_RUNG wire#w6
   RUNG wire#powerrail
      Contact( "IO_Valve_Storage_DB"."AV-24.05".FB_OPEN )
   END_RUNG wire#w6
   RUNG wire#powerrail
      Contact( "IO_Valve_Storage_DB"."AV-24.06".FB_OPEN )
   END_RUNG wire#w6
   RUNG wire#powerrail
      Contact( "IO_Valve_Storage_DB"."AV-24.14".FB_OPEN )
   END_RUNG wire#w6
   RUNG wire#powerrail
      Contact( "IO_Valve_Storage_DB"."AV-23.05".FB_OPEN )
      wire#w7
      Coil( "T-23.00".State."Line_AV5&AV6" )
   END_RUNG
   RUNG wire#powerrail
      Contact( "IO_Valve_Storage_DB"."AV-23.06".FB_OPEN )
   END_RUNG wire#w7
   RUNG wire#powerrail
      Contact( "IO_Valve_Storage_DB"."AV-23.08".FB_OPEN )
      wire#w8
      Coil( "T-24.00".State.CIP_Line1_ON )
   END_RUNG
   RUNG wire#powerrail
      Contact( "IO_Valve_Storage_DB"."AV-24.05".FB_OPEN )
   END_RUNG wire#w8
   RUNG wire#powerrail
      Contact( "IO_Valve_Storage_DB"."AV-24.06".FB_OPEN )
   END_RUNG wire#w8
   RUNG wire#powerrail
      Contact( "IO_Valve_Storage_DB"."AV-24.14".FB_OPEN )
   END_RUNG wire#w8
   RUNG wire#powerrail
      Contact( "IO_Valve_Storage_DB"."AV-24.05".FB_OPEN )
      wire#w9
      Coil( "T-24.00".State.CIP_Line2_ON )
   END_RUNG
   RUNG wire#powerrail
      Contact( "IO_Valve_Storage_DB"."AV-24.06".FB_OPEN )
   END_RUNG wire#w9
   RUNG wire#powerrail
      Contact( "IO_Valve_Storage_DB"."AV-24.14".FB_OPEN )
   END_RUNG wire#w9
   RUNG wire#powerrail
      Contact( "IO_Valve_Storage_DB"."AV-24.05".FB_OPEN )
      wire#w10
      Coil( "T-24.00".State."Line_AV5&AV6" )
   END_RUNG
   RUNG wire#powerrail
      Contact( "IO_Valve_Storage_DB"."AV-24.06".FB_OPEN )
   END_RUNG wire#w10
   // the same network as SCL:
   "T-23.00".State."Line_AV4&AV5" := "IO_Valve_Storage_DB"."AV-23.04".FB_OPEN OR "IO_Valve_Storage_DB"."AV-23.05".FB_OPEN;
   "T-23.00".State."Line_AV7&AV8" := "IO_Valve_Storage_DB"."AV-23.07".FB_OPEN OR "IO_Valve_Storage_DB"."AV-23.08".FB_OPEN;
   "T-24.00".State."Line_AV4&AV5" := "IO_Valve_Storage_DB"."AV-24.04".FB_OPEN OR "IO_Valve_Storage_DB"."AV-24.05".FB_OPEN;
   "T-24.00".State."Line_AV7&AV8" := "IO_Valve_Storage_DB"."AV-24.13".FB_OPEN OR "IO_Valve_Storage_DB"."AV-24.14".FB_OPEN;
   "T-29.00".State."Line_AV1&AV2" := "IO_Valve_Storage_DB"."AV-29.01".FB_OPEN OR "IO_Valve_Storage_DB"."AV-29.02".FB_OPEN;
   "T-23.00".State.CIP_Line1_ON := "IO_Valve_Storage_DB"."AV-23.05".FB_OPEN OR "IO_Valve_Storage_DB"."AV-23.06".FB_OPEN OR "IO_Valve_Storage_DB"."AV-23.08".FB_OPEN OR "IO_Valve_Storage_DB"."AV-24.05".FB_OPEN OR "IO_Valve_Storage_DB"."AV-24.06".FB_OPEN OR "IO_Valve_Storage_DB"."AV-24.14".FB_OPEN;
   "T-23.00".State."Line_AV5&AV6" := "IO_Valve_Storage_DB"."AV-23.05".FB_OPEN OR "IO_Valve_Storage_DB"."AV-23.06".FB_OPEN;
   "T-24.00".State.CIP_Line1_ON := "IO_Valve_Storage_DB"."AV-23.08".FB_OPEN OR "IO_Valve_Storage_DB"."AV-24.05".FB_OPEN OR "IO_Valve_Storage_DB"."AV-24.06".FB_OPEN OR "IO_Valve_Storage_DB"."AV-24.14".FB_OPEN;
   "T-24.00".State.CIP_Line2_ON := "IO_Valve_Storage_DB"."AV-24.05".FB_OPEN OR "IO_Valve_Storage_DB"."AV-24.06".FB_OPEN OR "IO_Valve_Storage_DB"."AV-24.14".FB_OPEN;
   "T-24.00".State."Line_AV5&AV6" := "IO_Valve_Storage_DB"."AV-24.05".FB_OPEN OR "IO_Valve_Storage_DB"."AV-24.06".FB_OPEN;
END_REGION

REGION Network 18: T-39.00 ST-04 -> Tank Storage By JBT
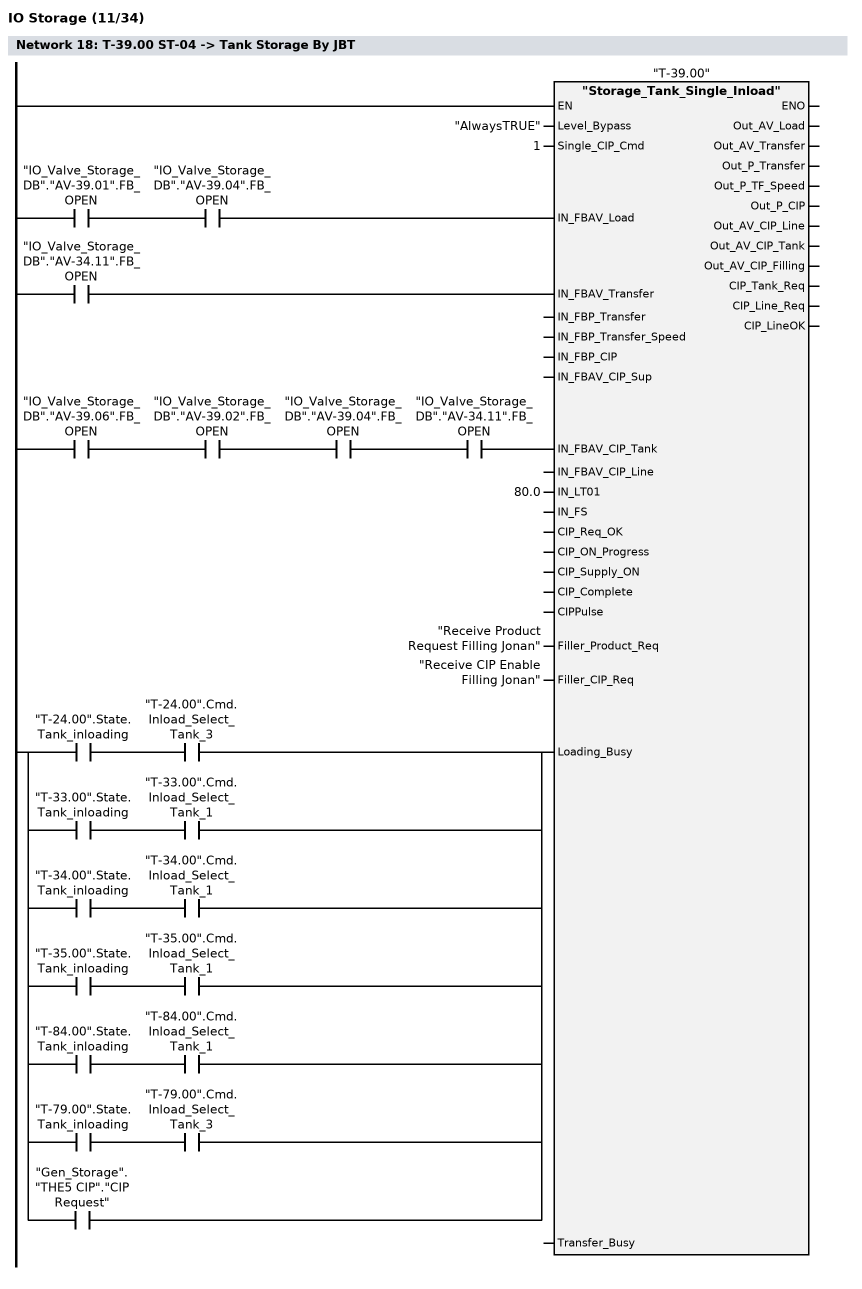
   RUNG wire#powerrail
      "T-39.00"(IN_FBAV_Load := wire#w1, IN_FBAV_Transfer := wire#w2, IN_FBAV_CIP_Tank := wire#w3, Loading_Busy := wire#w4, Level_Bypass := "AlwaysTRUE", Single_CIP_Cmd := 1, IN_FBP_Transfer :=, IN_FBP_Transfer_Speed :=, IN_FBP_CIP :=, IN_FBAV_CIP_Sup :=, IN_FBAV_CIP_Line :=, IN_LT01 := 80.0, IN_FS :=, CIP_Req_OK :=, CIP_ON_Progress :=, CIP_Supply_ON :=, CIP_Complete :=, CIPPulse :=, Filler_Product_Req := "Receive Product Request Filling Jonan", Filler_CIP_Req := "Receive CIP Enable Filling Jonan", Transfer_Busy :=, Out_AV_Load =>, Out_AV_Transfer =>, Out_P_Transfer =>, Out_P_TF_Speed =>, Out_P_CIP =>, Out_AV_CIP_Line =>, Out_AV_CIP_Tank =>, Out_AV_CIP_Filling =>, CIP_Tank_Req =>, CIP_Line_Req =>, CIP_LineOK =>)
   END_RUNG
   RUNG wire#powerrail
      Contact( "IO_Valve_Storage_DB"."AV-39.01".FB_OPEN )
      Contact( "IO_Valve_Storage_DB"."AV-39.04".FB_OPEN )
   END_RUNG wire#w1
   RUNG wire#powerrail
      Contact( "IO_Valve_Storage_DB"."AV-34.11".FB_OPEN )
   END_RUNG wire#w2
   RUNG wire#powerrail
      Contact( "IO_Valve_Storage_DB"."AV-39.06".FB_OPEN )
      Contact( "IO_Valve_Storage_DB"."AV-39.02".FB_OPEN )
      Contact( "IO_Valve_Storage_DB"."AV-39.04".FB_OPEN )
      Contact( "IO_Valve_Storage_DB"."AV-34.11".FB_OPEN )
   END_RUNG wire#w3
   RUNG wire#powerrail
      Contact( "T-24.00".State.Tank_inloading )
      Contact( "T-24.00".Cmd.Inload_Select_Tank_3 )
   END_RUNG wire#w4
   RUNG wire#powerrail
      Contact( "T-33.00".State.Tank_inloading )
      Contact( "T-33.00".Cmd.Inload_Select_Tank_1 )
   END_RUNG wire#w4
   RUNG wire#powerrail
      Contact( "T-34.00".State.Tank_inloading )
      Contact( "T-34.00".Cmd.Inload_Select_Tank_1 )
   END_RUNG wire#w4
   RUNG wire#powerrail
      Contact( "T-35.00".State.Tank_inloading )
      Contact( "T-35.00".Cmd.Inload_Select_Tank_1 )
   END_RUNG wire#w4
   RUNG wire#powerrail
      Contact( "T-84.00".State.Tank_inloading )
      Contact( "T-84.00".Cmd.Inload_Select_Tank_1 )
   END_RUNG wire#w4
   RUNG wire#powerrail
      Contact( "T-79.00".State.Tank_inloading )
      Contact( "T-79.00".Cmd.Inload_Select_Tank_3 )
   END_RUNG wire#w4
   RUNG wire#powerrail
      Contact( "Gen_Storage"."THE5 CIP"."CIP Request" )
   END_RUNG wire#w4
   // the same network as SCL:
   "T-39.00"(Level_Bypass := "AlwaysTRUE",   // "Storage_Tank_Single_Inload"
             Single_CIP_Cmd := 1,
             IN_FBAV_Load := "IO_Valve_Storage_DB"."AV-39.01".FB_OPEN AND "IO_Valve_Storage_DB"."AV-39.04".FB_OPEN,
             IN_FBAV_Transfer := "IO_Valve_Storage_DB"."AV-34.11".FB_OPEN,
             IN_FBAV_CIP_Tank := "IO_Valve_Storage_DB"."AV-39.06".FB_OPEN AND "IO_Valve_Storage_DB"."AV-39.02".FB_OPEN AND "IO_Valve_Storage_DB"."AV-39.04".FB_OPEN AND "IO_Valve_Storage_DB"."AV-34.11".FB_OPEN,
             IN_LT01 := 80.0,
             Filler_Product_Req := "Receive Product Request Filling Jonan",
             Filler_CIP_Req := "Receive CIP Enable Filling Jonan",
             Loading_Busy := ("T-24.00".State.Tank_inloading AND "T-24.00".Cmd.Inload_Select_Tank_3) OR ("T-33.00".State.Tank_inloading AND "T-33.00".Cmd.Inload_Select_Tank_1) OR ("T-34.00".State.Tank_inloading AND "T-34.00".Cmd.Inload_Select_Tank_1) OR ("T-35.00".State.Tank_inloading AND "T-35.00".Cmd.Inload_Select_Tank_1) OR ("T-84.00".State.Tank_inloading AND "T-84.00".Cmd.Inload_Select_Tank_1) OR ("T-79.00".State.Tank_inloading AND "T-79.00".Cmd.Inload_Select_Tank_3) OR "Gen_Storage"."THE5 CIP"."CIP Request");
END_REGION

REGION Network 19: T-39 Valve
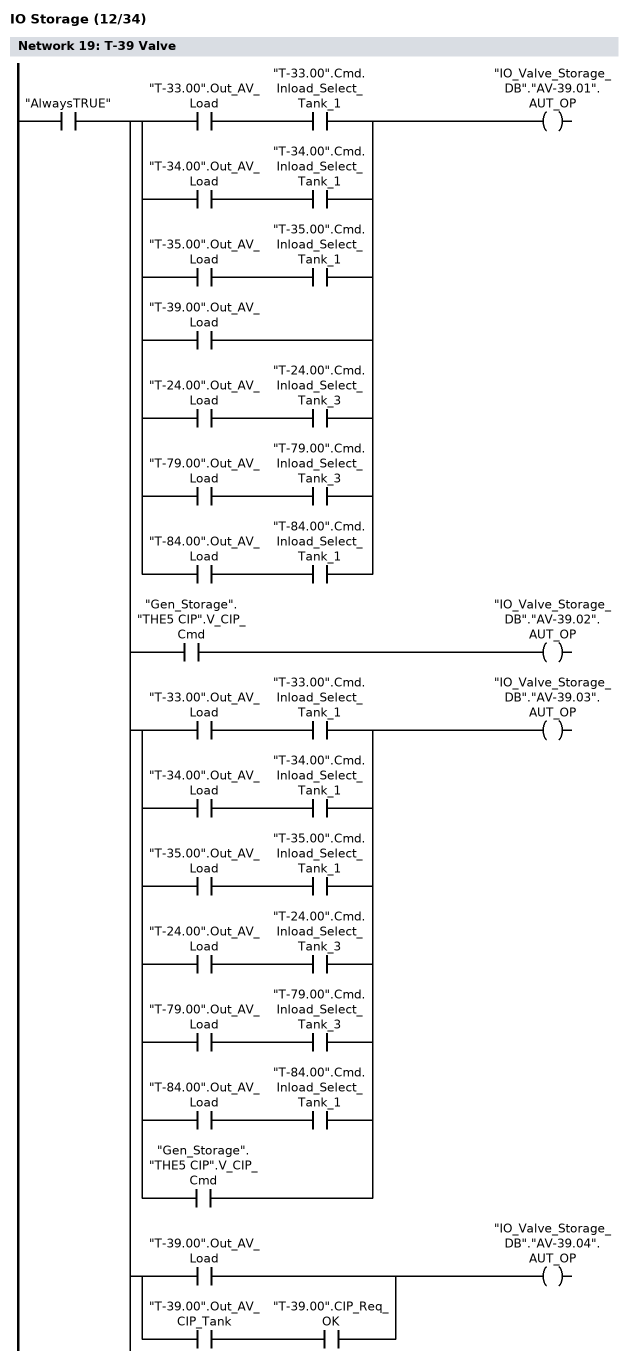
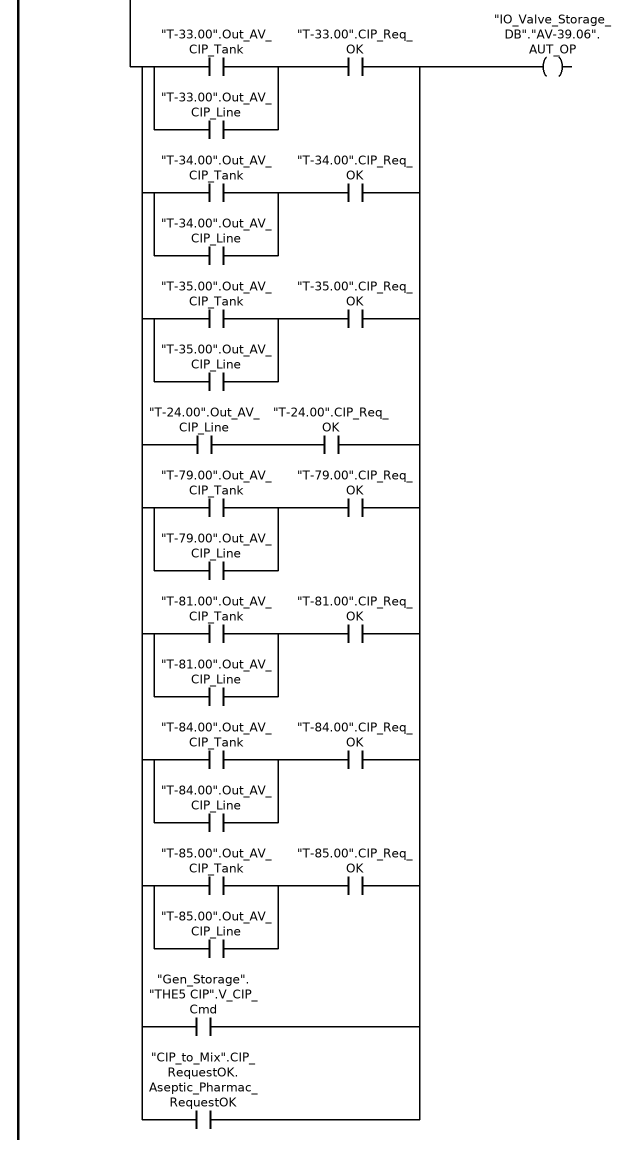
   RUNG wire#powerrail
      Contact( "AlwaysTRUE" )
      wire#w1
      Contact( "T-33.00".Out_AV_Load )
      Contact( "T-33.00".Cmd.Inload_Select_Tank_1 )
      wire#w2
      Coil( "IO_Valve_Storage_DB"."AV-39.01".AUT_OP )
   END_RUNG
   RUNG wire#w1
      Contact( "T-34.00".Out_AV_Load )
      Contact( "T-34.00".Cmd.Inload_Select_Tank_1 )
   END_RUNG wire#w2
   RUNG wire#w1
      Contact( "T-35.00".Out_AV_Load )
      Contact( "T-35.00".Cmd.Inload_Select_Tank_1 )
   END_RUNG wire#w2
   RUNG wire#w1
      Contact( "T-39.00".Out_AV_Load )
   END_RUNG wire#w2
   RUNG wire#w1
      Contact( "T-24.00".Out_AV_Load )
      Contact( "T-24.00".Cmd.Inload_Select_Tank_3 )
   END_RUNG wire#w2
   RUNG wire#w1
      Contact( "T-79.00".Out_AV_Load )
      Contact( "T-79.00".Cmd.Inload_Select_Tank_3 )
   END_RUNG wire#w2
   RUNG wire#w1
      Contact( "T-84.00".Out_AV_Load )
      Contact( "T-84.00".Cmd.Inload_Select_Tank_1 )
   END_RUNG wire#w2
   RUNG wire#w1
      Contact( "Gen_Storage"."THE5 CIP".V_CIP_Cmd )
      Coil( "IO_Valve_Storage_DB"."AV-39.02".AUT_OP )
   END_RUNG
   RUNG wire#w1
      Contact( "T-33.00".Out_AV_Load )
      Contact( "T-33.00".Cmd.Inload_Select_Tank_1 )
      wire#w3
      Coil( "IO_Valve_Storage_DB"."AV-39.03".AUT_OP )
   END_RUNG
   RUNG wire#w1
      Contact( "T-34.00".Out_AV_Load )
      Contact( "T-34.00".Cmd.Inload_Select_Tank_1 )
   END_RUNG wire#w3
   RUNG wire#w1
      Contact( "T-35.00".Out_AV_Load )
      Contact( "T-35.00".Cmd.Inload_Select_Tank_1 )
   END_RUNG wire#w3
   RUNG wire#w1
      Contact( "T-24.00".Out_AV_Load )
      Contact( "T-24.00".Cmd.Inload_Select_Tank_3 )
   END_RUNG wire#w3
   RUNG wire#w1
      Contact( "T-79.00".Out_AV_Load )
      Contact( "T-79.00".Cmd.Inload_Select_Tank_3 )
   END_RUNG wire#w3
   RUNG wire#w1
      Contact( "T-84.00".Out_AV_Load )
      Contact( "T-84.00".Cmd.Inload_Select_Tank_1 )
   END_RUNG wire#w3
   RUNG wire#w1
      Contact( "Gen_Storage"."THE5 CIP".V_CIP_Cmd )
   END_RUNG wire#w3
   RUNG wire#w1
      Contact( "T-39.00".Out_AV_Load )
      wire#w4
      Coil( "IO_Valve_Storage_DB"."AV-39.04".AUT_OP )
   END_RUNG
   RUNG wire#w1
      Contact( "T-39.00".Out_AV_CIP_Tank )
      Contact( "T-39.00".CIP_Req_OK )
   END_RUNG wire#w4
   RUNG wire#w1
      Contact( "T-33.00".Out_AV_CIP_Tank )
      wire#w5
      Contact( "T-33.00".CIP_Req_OK )
      wire#w6
      Coil( "IO_Valve_Storage_DB"."AV-39.06".AUT_OP )
   END_RUNG
   RUNG wire#w1
      Contact( "T-33.00".Out_AV_CIP_Line )
   END_RUNG wire#w5
   RUNG wire#w1
      Contact( "T-34.00".Out_AV_CIP_Tank )
      wire#w7
      Contact( "T-34.00".CIP_Req_OK )
   END_RUNG wire#w6
   RUNG wire#w1
      Contact( "T-34.00".Out_AV_CIP_Line )
   END_RUNG wire#w7
   RUNG wire#w1
      Contact( "T-35.00".Out_AV_CIP_Tank )
      wire#w8
      Contact( "T-35.00".CIP_Req_OK )
   END_RUNG wire#w6
   RUNG wire#w1
      Contact( "T-35.00".Out_AV_CIP_Line )
   END_RUNG wire#w8
   RUNG wire#w1
      Contact( "T-24.00".Out_AV_CIP_Line )
      Contact( "T-24.00".CIP_Req_OK )
   END_RUNG wire#w6
   RUNG wire#w1
      Contact( "T-79.00".Out_AV_CIP_Tank )
      wire#w9
      Contact( "T-79.00".CIP_Req_OK )
   END_RUNG wire#w6
   RUNG wire#w1
      Contact( "T-79.00".Out_AV_CIP_Line )
   END_RUNG wire#w9
   RUNG wire#w1
      Contact( "T-81.00".Out_AV_CIP_Tank )
      wire#w10
      Contact( "T-81.00".CIP_Req_OK )
   END_RUNG wire#w6
   RUNG wire#w1
      Contact( "T-81.00".Out_AV_CIP_Line )
   END_RUNG wire#w10
   RUNG wire#w1
      Contact( "T-84.00".Out_AV_CIP_Tank )
      wire#w11
      Contact( "T-84.00".CIP_Req_OK )
   END_RUNG wire#w6
   RUNG wire#w1
      Contact( "T-84.00".Out_AV_CIP_Line )
   END_RUNG wire#w11
   RUNG wire#w1
      Contact( "T-85.00".Out_AV_CIP_Tank )
      wire#w12
      Contact( "T-85.00".CIP_Req_OK )
   END_RUNG wire#w6
   RUNG wire#w1
      Contact( "T-85.00".Out_AV_CIP_Line )
   END_RUNG wire#w12
   RUNG wire#w1
      Contact( "Gen_Storage"."THE5 CIP".V_CIP_Cmd )
   END_RUNG wire#w6
   RUNG wire#w1
      Contact( "CIP_to_Mix".CIP_RequestOK.Aseptic_Pharmac_RequestOK )
   END_RUNG wire#w6
   // the same network as SCL:
   "IO_Valve_Storage_DB"."AV-39.01".AUT_OP := "AlwaysTRUE" AND (("T-33.00".Out_AV_Load AND "T-33.00".Cmd.Inload_Select_Tank_1) OR ("T-34.00".Out_AV_Load AND "T-34.00".Cmd.Inload_Select_Tank_1) OR ("T-35.00".Out_AV_Load AND "T-35.00".Cmd.Inload_Select_Tank_1) OR "T-39.00".Out_AV_Load OR ("T-24.00".Out_AV_Load AND "T-24.00".Cmd.Inload_Select_Tank_3) OR ("T-79.00".Out_AV_Load AND "T-79.00".Cmd.Inload_Select_Tank_3) OR ("T-84.00".Out_AV_Load AND "T-84.00".Cmd.Inload_Select_Tank_1));
   "IO_Valve_Storage_DB"."AV-39.02".AUT_OP := "AlwaysTRUE" AND "Gen_Storage"."THE5 CIP".V_CIP_Cmd;
   "IO_Valve_Storage_DB"."AV-39.03".AUT_OP := "AlwaysTRUE" AND (("T-33.00".Out_AV_Load AND "T-33.00".Cmd.Inload_Select_Tank_1) OR ("T-34.00".Out_AV_Load AND "T-34.00".Cmd.Inload_Select_Tank_1) OR ("T-35.00".Out_AV_Load AND "T-35.00".Cmd.Inload_Select_Tank_1) OR ("T-24.00".Out_AV_Load AND "T-24.00".Cmd.Inload_Select_Tank_3) OR ("T-79.00".Out_AV_Load AND "T-79.00".Cmd.Inload_Select_Tank_3) OR ("T-84.00".Out_AV_Load AND "T-84.00".Cmd.Inload_Select_Tank_1) OR "Gen_Storage"."THE5 CIP".V_CIP_Cmd);
   "IO_Valve_Storage_DB"."AV-39.04".AUT_OP := "AlwaysTRUE" AND ("T-39.00".Out_AV_Load OR ("T-39.00".Out_AV_CIP_Tank AND "T-39.00".CIP_Req_OK));
   "IO_Valve_Storage_DB"."AV-39.06".AUT_OP := "AlwaysTRUE" AND ((("T-33.00".Out_AV_CIP_Tank OR "T-33.00".Out_AV_CIP_Line) AND "T-33.00".CIP_Req_OK) OR (("T-34.00".Out_AV_CIP_Tank OR "T-34.00".Out_AV_CIP_Line) AND "T-34.00".CIP_Req_OK) OR (("T-35.00".Out_AV_CIP_Tank OR "T-35.00".Out_AV_CIP_Line) AND "T-35.00".CIP_Req_OK) OR ("T-24.00".Out_AV_CIP_Line AND "T-24.00".CIP_Req_OK) OR (("T-79.00".Out_AV_CIP_Tank OR "T-79.00".Out_AV_CIP_Line) AND "T-79.00".CIP_Req_OK) OR (("T-81.00".Out_AV_CIP_Tank OR "T-81.00".Out_AV_CIP_Line) AND "T-81.00".CIP_Req_OK) OR (("T-84.00".Out_AV_CIP_Tank OR "T-84.00".Out_AV_CIP_Line) AND "T-84.00".CIP_Req_OK) OR (("T-85.00".Out_AV_CIP_Tank OR "T-85.00".Out_AV_CIP_Line) AND "T-85.00".CIP_Req_OK) OR "Gen_Storage"."THE5 CIP".V_CIP_Cmd OR "CIP_to_Mix".CIP_RequestOK.Aseptic_Pharmac_RequestOK);
END_REGION

REGION Network 21: T-33.00 ST-06
   // Inload 1 : THE-5
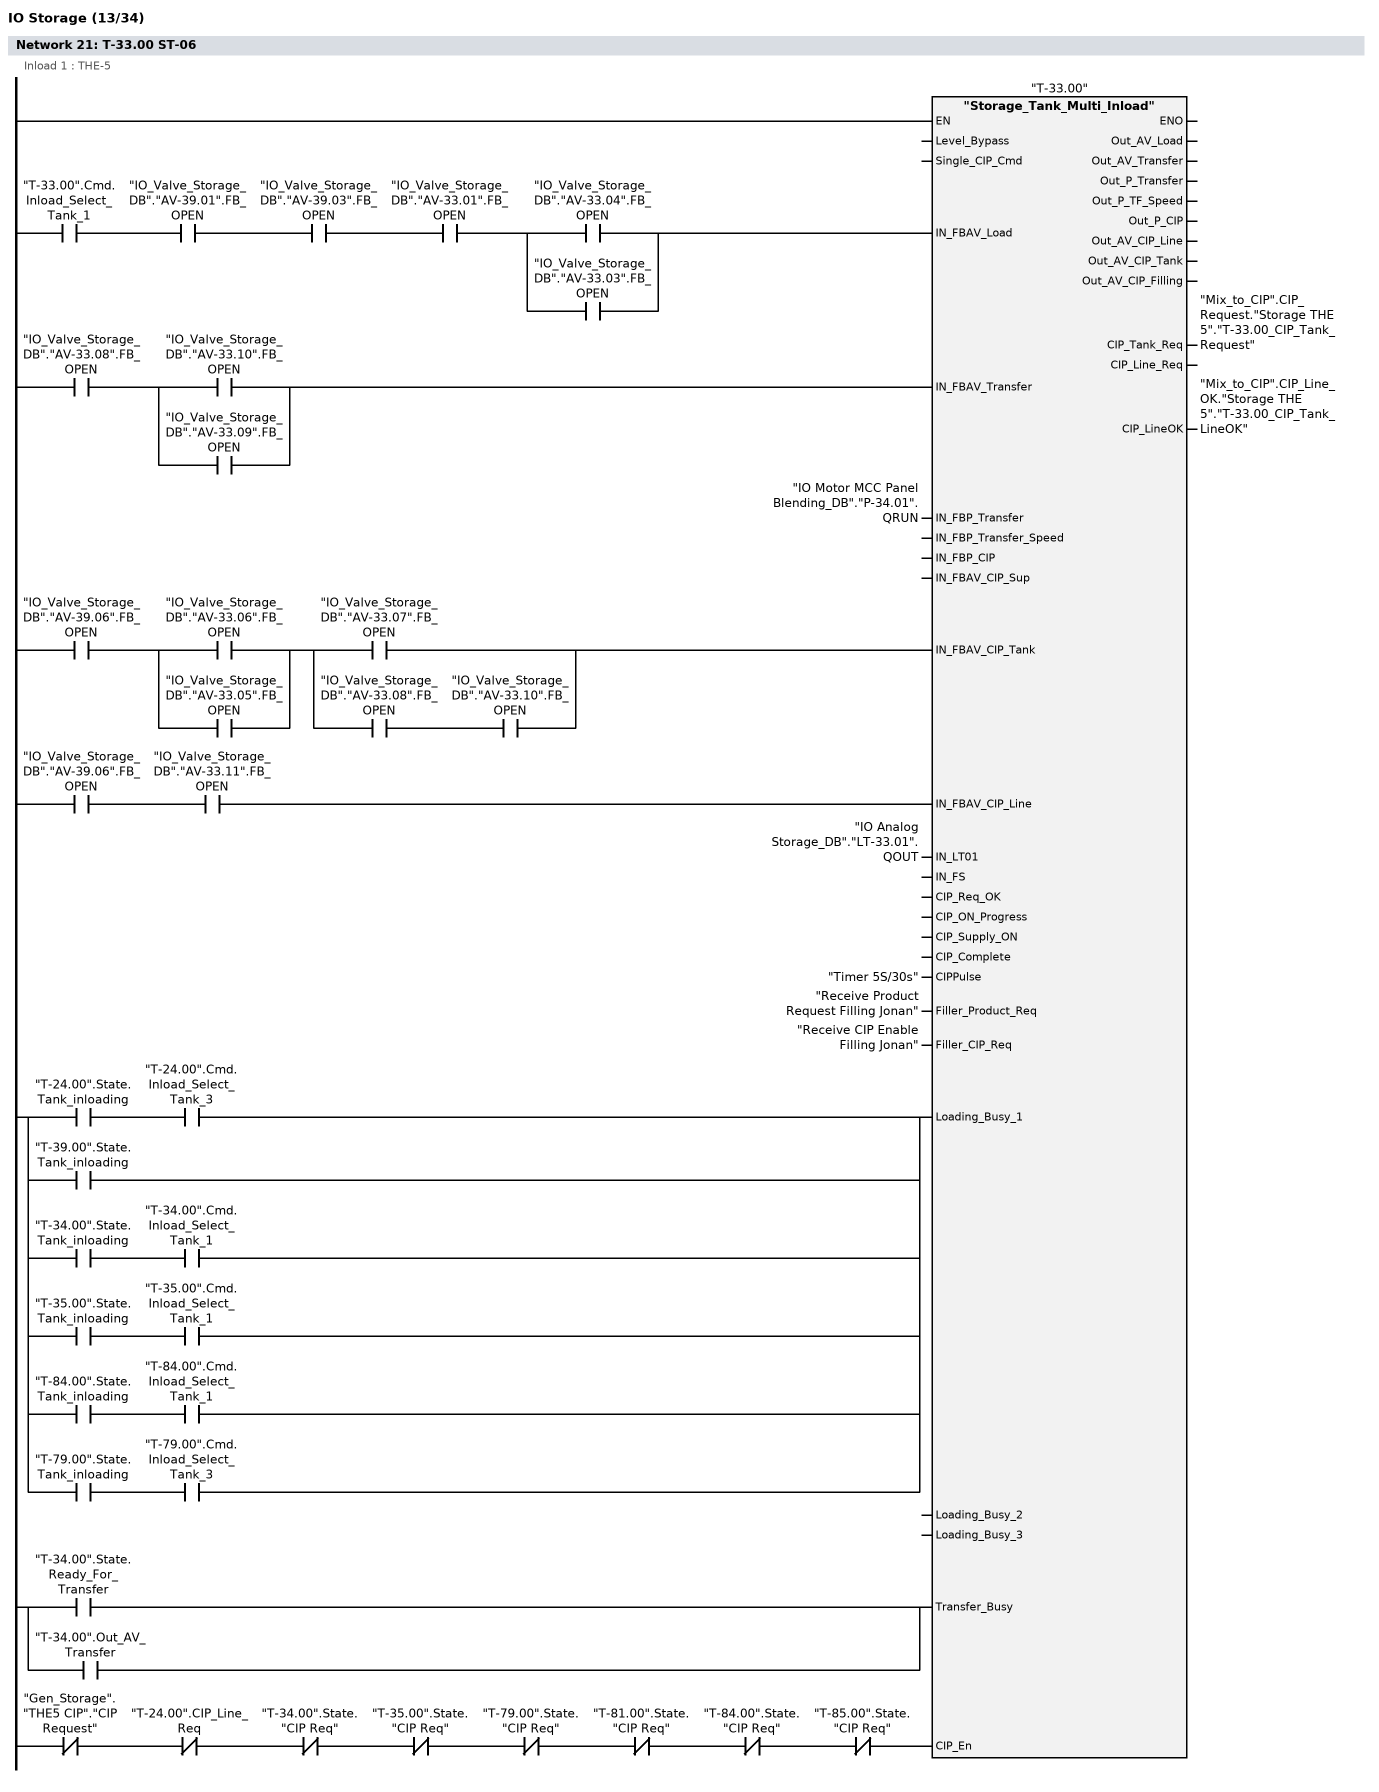
   RUNG wire#powerrail
      "T-33.00"(IN_FBAV_Load := wire#w2, IN_FBAV_Transfer := wire#w4, IN_FBAV_CIP_Tank := wire#w7, IN_FBAV_CIP_Line := wire#w8, Loading_Busy_1 := wire#w9, Transfer_Busy := wire#w10, CIP_En := wire#w11, Level_Bypass :=, Single_CIP_Cmd :=, IN_FBP_Transfer := "IO Motor MCC Panel Blending_DB"."P-34.01".QRUN, IN_FBP_Transfer_Speed :=, IN_FBP_CIP :=, IN_FBAV_CIP_Sup :=, IN_LT01 := "IO Analog Storage_DB"."LT-33.01".QOUT, IN_FS :=, CIP_Req_OK :=, CIP_ON_Progress :=, CIP_Supply_ON :=, CIP_Complete :=, CIPPulse := "Timer 5S/30s", Filler_Product_Req := "Receive Product Request Filling Jonan", Filler_CIP_Req := "Receive CIP Enable Filling Jonan", Loading_Busy_2 :=, Loading_Busy_3 :=, Out_AV_Load =>, Out_AV_Transfer =>, Out_P_Transfer =>, Out_P_TF_Speed =>, Out_P_CIP =>, Out_AV_CIP_Line =>, Out_AV_CIP_Tank =>, Out_AV_CIP_Filling =>, CIP_Tank_Req => "Mix_to_CIP".CIP_Request."Storage THE 5"."T-33.00_CIP_Tank_Request", CIP_Line_Req =>, CIP_LineOK => "Mix_to_CIP".CIP_Line_OK."Storage THE 5"."T-33.00_CIP_Tank_LineOK")
   END_RUNG
   RUNG wire#powerrail
      Contact( "T-33.00".Cmd.Inload_Select_Tank_1 )
      Contact( "IO_Valve_Storage_DB"."AV-39.01".FB_OPEN )
      Contact( "IO_Valve_Storage_DB"."AV-39.03".FB_OPEN )
      Contact( "IO_Valve_Storage_DB"."AV-33.01".FB_OPEN )
      wire#w1
      Contact( "IO_Valve_Storage_DB"."AV-33.04".FB_OPEN )
   END_RUNG wire#w2
   RUNG wire#w1
      Contact( "IO_Valve_Storage_DB"."AV-33.03".FB_OPEN )
   END_RUNG wire#w2
   RUNG wire#powerrail
      Contact( "IO_Valve_Storage_DB"."AV-33.08".FB_OPEN )
      wire#w3
      Contact( "IO_Valve_Storage_DB"."AV-33.10".FB_OPEN )
   END_RUNG wire#w4
   RUNG wire#w3
      Contact( "IO_Valve_Storage_DB"."AV-33.09".FB_OPEN )
   END_RUNG wire#w4
   RUNG wire#powerrail
      Contact( "IO_Valve_Storage_DB"."AV-39.06".FB_OPEN )
      wire#w5
      Contact( "IO_Valve_Storage_DB"."AV-33.06".FB_OPEN )
      wire#w6
      Contact( "IO_Valve_Storage_DB"."AV-33.07".FB_OPEN )
   END_RUNG wire#w7
   RUNG wire#w5
      Contact( "IO_Valve_Storage_DB"."AV-33.05".FB_OPEN )
   END_RUNG wire#w6
   RUNG wire#w6
      Contact( "IO_Valve_Storage_DB"."AV-33.08".FB_OPEN )
      Contact( "IO_Valve_Storage_DB"."AV-33.10".FB_OPEN )
   END_RUNG wire#w7
   RUNG wire#powerrail
      Contact( "IO_Valve_Storage_DB"."AV-39.06".FB_OPEN )
      Contact( "IO_Valve_Storage_DB"."AV-33.11".FB_OPEN )
   END_RUNG wire#w8
   RUNG wire#powerrail
      Contact( "T-24.00".State.Tank_inloading )
      Contact( "T-24.00".Cmd.Inload_Select_Tank_3 )
   END_RUNG wire#w9
   RUNG wire#powerrail
      Contact( "T-39.00".State.Tank_inloading )
   END_RUNG wire#w9
   RUNG wire#powerrail
      Contact( "T-34.00".State.Tank_inloading )
      Contact( "T-34.00".Cmd.Inload_Select_Tank_1 )
   END_RUNG wire#w9
   RUNG wire#powerrail
      Contact( "T-35.00".State.Tank_inloading )
      Contact( "T-35.00".Cmd.Inload_Select_Tank_1 )
   END_RUNG wire#w9
   RUNG wire#powerrail
      Contact( "T-84.00".State.Tank_inloading )
      Contact( "T-84.00".Cmd.Inload_Select_Tank_1 )
   END_RUNG wire#w9
   RUNG wire#powerrail
      Contact( "T-79.00".State.Tank_inloading )
      Contact( "T-79.00".Cmd.Inload_Select_Tank_3 )
   END_RUNG wire#w9
   RUNG wire#powerrail
      Contact( "T-34.00".State.Ready_For_Transfer )
   END_RUNG wire#w10
   RUNG wire#powerrail
      Contact( "T-34.00".Out_AV_Transfer )
   END_RUNG wire#w10
   RUNG wire#powerrail
      I_Contact( "Gen_Storage"."THE5 CIP"."CIP Request" )
      I_Contact( "T-24.00".CIP_Line_Req )
      I_Contact( "T-34.00".State."CIP Req" )
      I_Contact( "T-35.00".State."CIP Req" )
      I_Contact( "T-79.00".State."CIP Req" )
      I_Contact( "T-81.00".State."CIP Req" )
      I_Contact( "T-84.00".State."CIP Req" )
      I_Contact( "T-85.00".State."CIP Req" )
   END_RUNG wire#w11
   // the same network as SCL:
   "T-33.00"(IN_FBAV_Load := "T-33.00".Cmd.Inload_Select_Tank_1 AND "IO_Valve_Storage_DB"."AV-39.01".FB_OPEN AND "IO_Valve_Storage_DB"."AV-39.03".FB_OPEN AND "IO_Valve_Storage_DB"."AV-33.01".FB_OPEN AND ("IO_Valve_Storage_DB"."AV-33.04".FB_OPEN OR "IO_Valve_Storage_DB"."AV-33.03".FB_OPEN),   // "Storage_Tank_Multi_Inload"
             IN_FBAV_Transfer := "IO_Valve_Storage_DB"."AV-33.08".FB_OPEN AND ("IO_Valve_Storage_DB"."AV-33.10".FB_OPEN OR "IO_Valve_Storage_DB"."AV-33.09".FB_OPEN),
             IN_FBP_Transfer := "IO Motor MCC Panel Blending_DB"."P-34.01".QRUN,
             IN_FBAV_CIP_Tank := "IO_Valve_Storage_DB"."AV-39.06".FB_OPEN AND ("IO_Valve_Storage_DB"."AV-33.06".FB_OPEN OR "IO_Valve_Storage_DB"."AV-33.05".FB_OPEN) AND ("IO_Valve_Storage_DB"."AV-33.07".FB_OPEN OR ("IO_Valve_Storage_DB"."AV-33.08".FB_OPEN AND "IO_Valve_Storage_DB"."AV-33.10".FB_OPEN)),
             IN_FBAV_CIP_Line := "IO_Valve_Storage_DB"."AV-39.06".FB_OPEN AND "IO_Valve_Storage_DB"."AV-33.11".FB_OPEN,
             IN_LT01 := "IO Analog Storage_DB"."LT-33.01".QOUT,
             CIPPulse := "Timer 5S/30s",
             Filler_Product_Req := "Receive Product Request Filling Jonan",
             Filler_CIP_Req := "Receive CIP Enable Filling Jonan",
             Loading_Busy_1 := ("T-24.00".State.Tank_inloading AND "T-24.00".Cmd.Inload_Select_Tank_3) OR "T-39.00".State.Tank_inloading OR ("T-34.00".State.Tank_inloading AND "T-34.00".Cmd.Inload_Select_Tank_1) OR ("T-35.00".State.Tank_inloading AND "T-35.00".Cmd.Inload_Select_Tank_1) OR ("T-84.00".State.Tank_inloading AND "T-84.00".Cmd.Inload_Select_Tank_1) OR ("T-79.00".State.Tank_inloading AND "T-79.00".Cmd.Inload_Select_Tank_3),
             Transfer_Busy := "T-34.00".State.Ready_For_Transfer OR "T-34.00".Out_AV_Transfer,
             CIP_En := NOT "Gen_Storage"."THE5 CIP"."CIP Request" AND NOT "T-24.00".CIP_Line_Req AND NOT "T-34.00".State."CIP Req" AND NOT "T-35.00".State."CIP Req" AND NOT "T-79.00".State."CIP Req" AND NOT "T-81.00".State."CIP Req" AND NOT "T-84.00".State."CIP Req" AND NOT "T-85.00".State."CIP Req",
             CIP_Tank_Req => "Mix_to_CIP".CIP_Request."Storage THE 5"."T-33.00_CIP_Tank_Request",
             CIP_LineOK => "Mix_to_CIP".CIP_Line_OK."Storage THE 5"."T-33.00_CIP_Tank_LineOK");
END_REGION

REGION Network 22: T-33 Valve
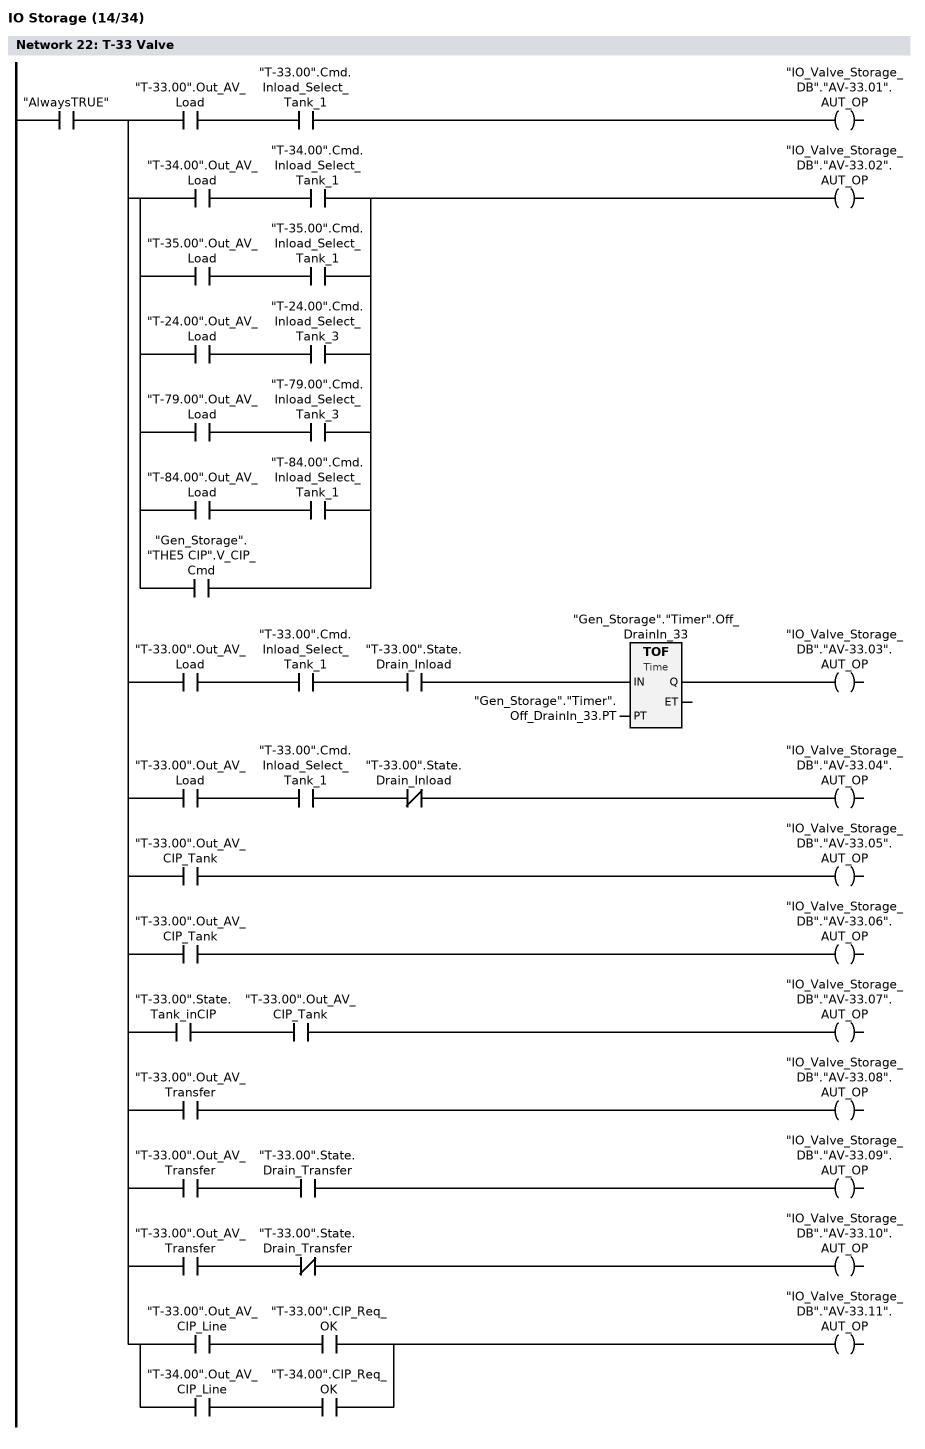
   RUNG wire#powerrail
      Contact( "AlwaysTRUE" )
      wire#w1
      Contact( "T-33.00".Out_AV_Load )
      Contact( "T-33.00".Cmd.Inload_Select_Tank_1 )
      Coil( "IO_Valve_Storage_DB"."AV-33.01".AUT_OP )
   END_RUNG
   RUNG wire#w1
      Contact( "T-34.00".Out_AV_Load )
      Contact( "T-34.00".Cmd.Inload_Select_Tank_1 )
      wire#w2
      Coil( "IO_Valve_Storage_DB"."AV-33.02".AUT_OP )
   END_RUNG
   RUNG wire#w1
      Contact( "T-35.00".Out_AV_Load )
      Contact( "T-35.00".Cmd.Inload_Select_Tank_1 )
   END_RUNG wire#w2
   RUNG wire#w1
      Contact( "T-24.00".Out_AV_Load )
      Contact( "T-24.00".Cmd.Inload_Select_Tank_3 )
   END_RUNG wire#w2
   RUNG wire#w1
      Contact( "T-79.00".Out_AV_Load )
      Contact( "T-79.00".Cmd.Inload_Select_Tank_3 )
   END_RUNG wire#w2
   RUNG wire#w1
      Contact( "T-84.00".Out_AV_Load )
      Contact( "T-84.00".Cmd.Inload_Select_Tank_1 )
   END_RUNG wire#w2
   RUNG wire#w1
      Contact( "Gen_Storage"."THE5 CIP".V_CIP_Cmd )
   END_RUNG wire#w2
   RUNG wire#w1
      Contact( "T-33.00".Out_AV_Load )
      Contact( "T-33.00".Cmd.Inload_Select_Tank_1 )
      Contact( "T-33.00".State.Drain_Inload )
      { S7_Templates := "time_type := Time" } "Gen_Storage"."Timer".Off_DrainIn_33.TOF(pt := "Gen_Storage"."Timer".Off_DrainIn_33.PT, et =>)
      Coil( "IO_Valve_Storage_DB"."AV-33.03".AUT_OP )
   END_RUNG
   RUNG wire#w1
      Contact( "T-33.00".Out_AV_Load )
      Contact( "T-33.00".Cmd.Inload_Select_Tank_1 )
      I_Contact( "T-33.00".State.Drain_Inload )
      Coil( "IO_Valve_Storage_DB"."AV-33.04".AUT_OP )
   END_RUNG
   RUNG wire#w1
      Contact( "T-33.00".Out_AV_CIP_Tank )
      Coil( "IO_Valve_Storage_DB"."AV-33.05".AUT_OP )
   END_RUNG
   RUNG wire#w1
      Contact( "T-33.00".Out_AV_CIP_Tank )
      Coil( "IO_Valve_Storage_DB"."AV-33.06".AUT_OP )
   END_RUNG
   RUNG wire#w1
      Contact( "T-33.00".State.Tank_inCIP )
      Contact( "T-33.00".Out_AV_CIP_Tank )
      Coil( "IO_Valve_Storage_DB"."AV-33.07".AUT_OP )
   END_RUNG
   RUNG wire#w1
      Contact( "T-33.00".Out_AV_Transfer )
      Coil( "IO_Valve_Storage_DB"."AV-33.08".AUT_OP )
   END_RUNG
   RUNG wire#w1
      Contact( "T-33.00".Out_AV_Transfer )
      Contact( "T-33.00".State.Drain_Transfer )
      Coil( "IO_Valve_Storage_DB"."AV-33.09".AUT_OP )
   END_RUNG
   RUNG wire#w1
      Contact( "T-33.00".Out_AV_Transfer )
      I_Contact( "T-33.00".State.Drain_Transfer )
      Coil( "IO_Valve_Storage_DB"."AV-33.10".AUT_OP )
   END_RUNG
   RUNG wire#w1
      Contact( "T-33.00".Out_AV_CIP_Line )
      Contact( "T-33.00".CIP_Req_OK )
      wire#w3
      Coil( "IO_Valve_Storage_DB"."AV-33.11".AUT_OP )
   END_RUNG
   RUNG wire#w1
      Contact( "T-34.00".Out_AV_CIP_Line )
      Contact( "T-34.00".CIP_Req_OK )
   END_RUNG wire#w3
   // the same network as SCL:
   "IO_Valve_Storage_DB"."AV-33.01".AUT_OP := "AlwaysTRUE" AND "T-33.00".Out_AV_Load AND "T-33.00".Cmd.Inload_Select_Tank_1;
   "IO_Valve_Storage_DB"."AV-33.02".AUT_OP := "AlwaysTRUE" AND (("T-34.00".Out_AV_Load AND "T-34.00".Cmd.Inload_Select_Tank_1) OR ("T-35.00".Out_AV_Load AND "T-35.00".Cmd.Inload_Select_Tank_1) OR ("T-24.00".Out_AV_Load AND "T-24.00".Cmd.Inload_Select_Tank_3) OR ("T-79.00".Out_AV_Load AND "T-79.00".Cmd.Inload_Select_Tank_3) OR ("T-84.00".Out_AV_Load AND "T-84.00".Cmd.Inload_Select_Tank_1) OR "Gen_Storage"."THE5 CIP".V_CIP_Cmd);
   "Gen_Storage"."Timer".Off_DrainIn_33.TOF(IN := "AlwaysTRUE" AND "T-33.00".Out_AV_Load AND "T-33.00".Cmd.Inload_Select_Tank_1 AND "T-33.00".State.Drain_Inload,
                           PT := "Gen_Storage"."Timer".Off_DrainIn_33.PT);
   "IO_Valve_Storage_DB"."AV-33.03".AUT_OP := "Gen_Storage"."Timer".Off_DrainIn_33.Q;
   "IO_Valve_Storage_DB"."AV-33.04".AUT_OP := "AlwaysTRUE" AND "T-33.00".Out_AV_Load AND "T-33.00".Cmd.Inload_Select_Tank_1 AND NOT "T-33.00".State.Drain_Inload;
   "IO_Valve_Storage_DB"."AV-33.05".AUT_OP := "AlwaysTRUE" AND "T-33.00".Out_AV_CIP_Tank;
   "IO_Valve_Storage_DB"."AV-33.06".AUT_OP := "AlwaysTRUE" AND "T-33.00".Out_AV_CIP_Tank;
   "IO_Valve_Storage_DB"."AV-33.07".AUT_OP := "AlwaysTRUE" AND "T-33.00".State.Tank_inCIP AND "T-33.00".Out_AV_CIP_Tank;
   "IO_Valve_Storage_DB"."AV-33.08".AUT_OP := "AlwaysTRUE" AND "T-33.00".Out_AV_Transfer;
   "IO_Valve_Storage_DB"."AV-33.09".AUT_OP := "AlwaysTRUE" AND "T-33.00".Out_AV_Transfer AND "T-33.00".State.Drain_Transfer;
   "IO_Valve_Storage_DB"."AV-33.10".AUT_OP := "AlwaysTRUE" AND "T-33.00".Out_AV_Transfer AND NOT "T-33.00".State.Drain_Transfer;
   "IO_Valve_Storage_DB"."AV-33.11".AUT_OP := "AlwaysTRUE" AND (("T-33.00".Out_AV_CIP_Line AND "T-33.00".CIP_Req_OK) OR ("T-34.00".Out_AV_CIP_Line AND "T-34.00".CIP_Req_OK));
END_REGION

REGION Network 24: T-34.00 ST-08
   // Inload 1 : THE-5
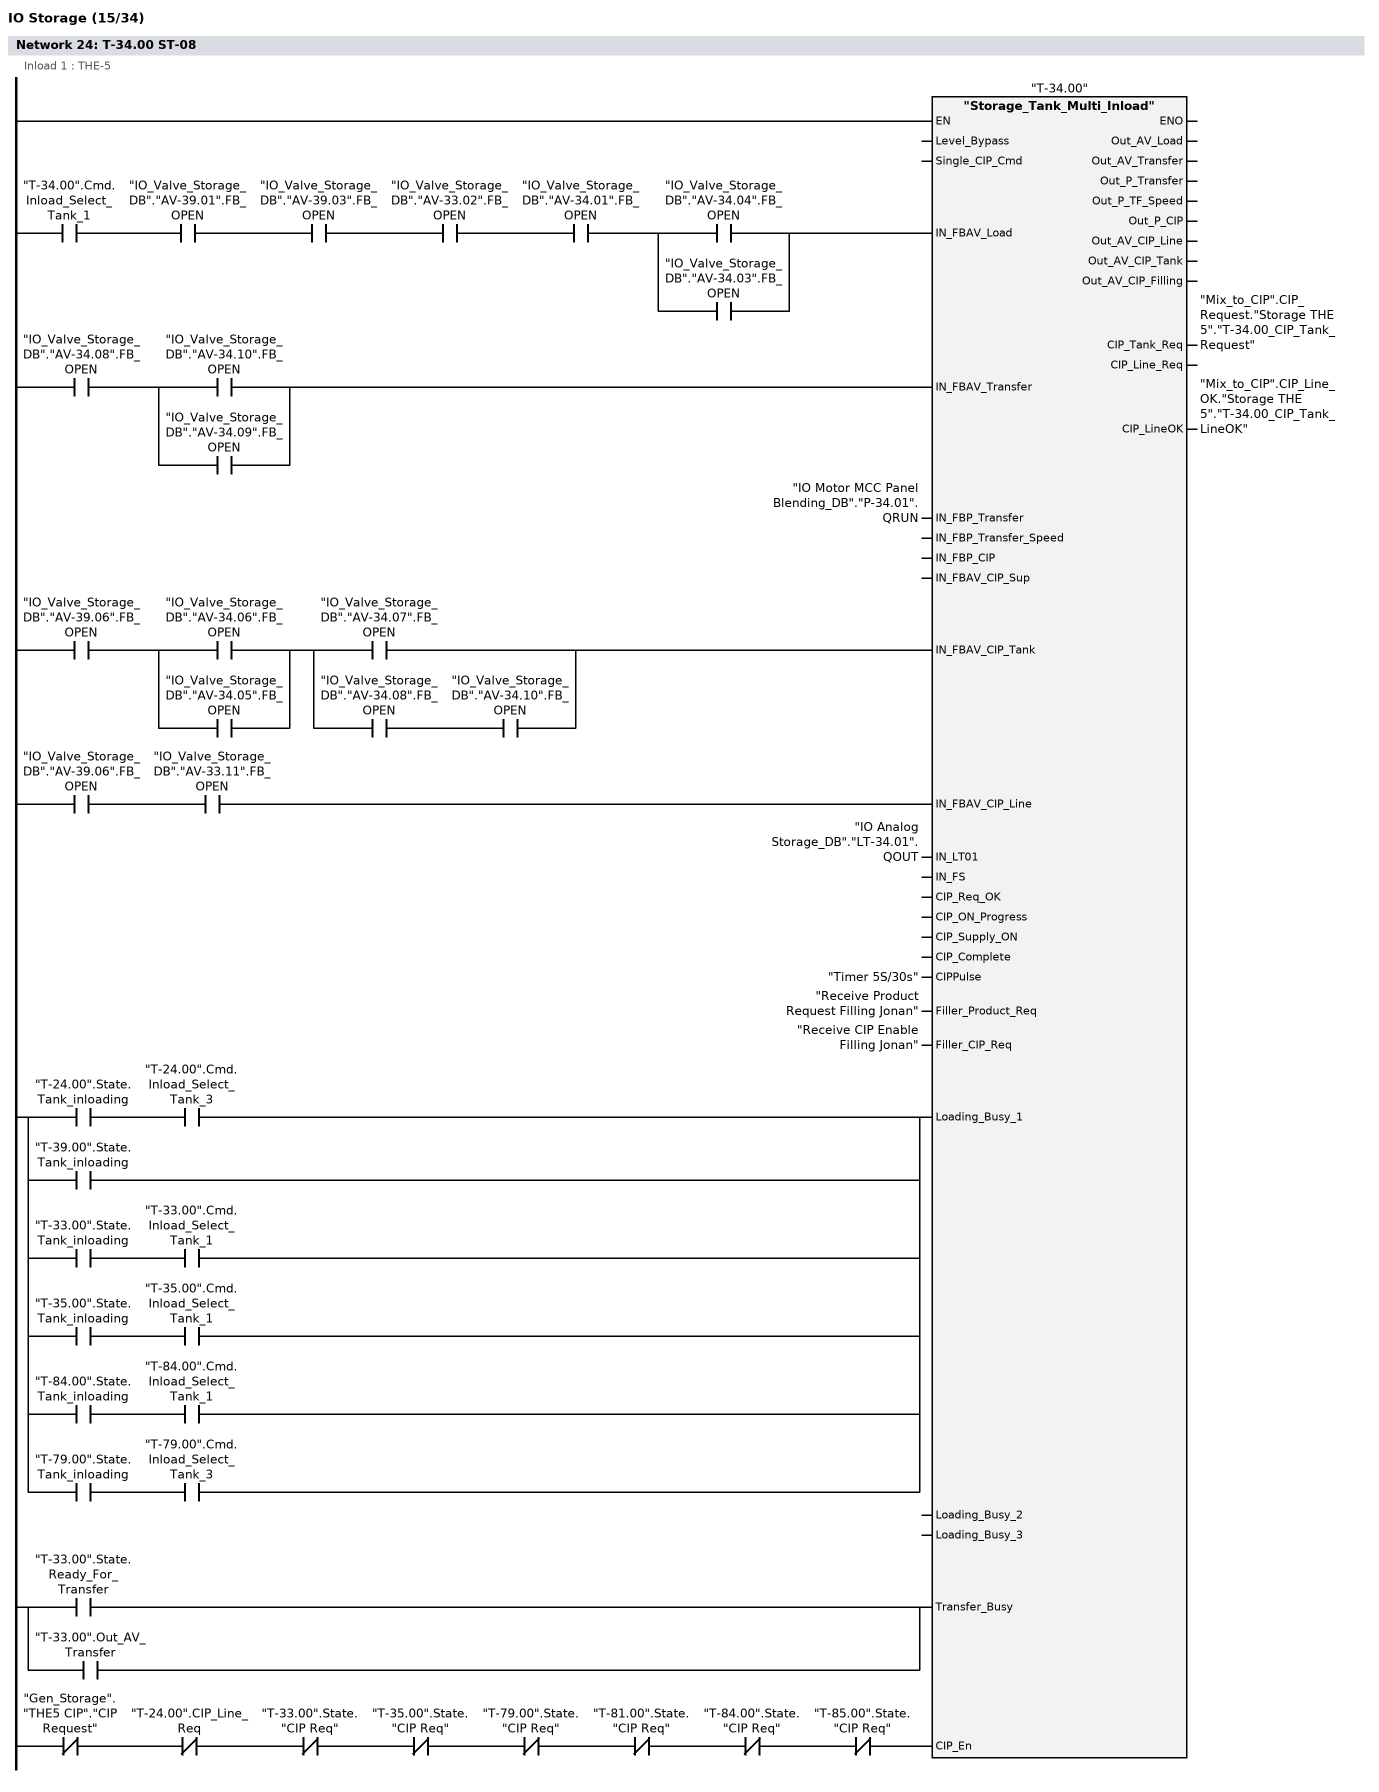
   RUNG wire#powerrail
      "T-34.00"(IN_FBAV_Load := wire#w2, IN_FBAV_Transfer := wire#w4, IN_FBAV_CIP_Tank := wire#w7, IN_FBAV_CIP_Line := wire#w8, Loading_Busy_1 := wire#w9, Transfer_Busy := wire#w10, CIP_En := wire#w11, Level_Bypass :=, Single_CIP_Cmd :=, IN_FBP_Transfer := "IO Motor MCC Panel Blending_DB"."P-34.01".QRUN, IN_FBP_Transfer_Speed :=, IN_FBP_CIP :=, IN_FBAV_CIP_Sup :=, IN_LT01 := "IO Analog Storage_DB"."LT-34.01".QOUT, IN_FS :=, CIP_Req_OK :=, CIP_ON_Progress :=, CIP_Supply_ON :=, CIP_Complete :=, CIPPulse := "Timer 5S/30s", Filler_Product_Req := "Receive Product Request Filling Jonan", Filler_CIP_Req := "Receive CIP Enable Filling Jonan", Loading_Busy_2 :=, Loading_Busy_3 :=, Out_AV_Load =>, Out_AV_Transfer =>, Out_P_Transfer =>, Out_P_TF_Speed =>, Out_P_CIP =>, Out_AV_CIP_Line =>, Out_AV_CIP_Tank =>, Out_AV_CIP_Filling =>, CIP_Tank_Req => "Mix_to_CIP".CIP_Request."Storage THE 5"."T-34.00_CIP_Tank_Request", CIP_Line_Req =>, CIP_LineOK => "Mix_to_CIP".CIP_Line_OK."Storage THE 5"."T-34.00_CIP_Tank_LineOK")
   END_RUNG
   RUNG wire#powerrail
      Contact( "T-34.00".Cmd.Inload_Select_Tank_1 )
      Contact( "IO_Valve_Storage_DB"."AV-39.01".FB_OPEN )
      Contact( "IO_Valve_Storage_DB"."AV-39.03".FB_OPEN )
      Contact( "IO_Valve_Storage_DB"."AV-33.02".FB_OPEN )
      Contact( "IO_Valve_Storage_DB"."AV-34.01".FB_OPEN )
      wire#w1
      Contact( "IO_Valve_Storage_DB"."AV-34.04".FB_OPEN )
   END_RUNG wire#w2
   RUNG wire#w1
      Contact( "IO_Valve_Storage_DB"."AV-34.03".FB_OPEN )
   END_RUNG wire#w2
   RUNG wire#powerrail
      Contact( "IO_Valve_Storage_DB"."AV-34.08".FB_OPEN )
      wire#w3
      Contact( "IO_Valve_Storage_DB"."AV-34.10".FB_OPEN )
   END_RUNG wire#w4
   RUNG wire#w3
      Contact( "IO_Valve_Storage_DB"."AV-34.09".FB_OPEN )
   END_RUNG wire#w4
   RUNG wire#powerrail
      Contact( "IO_Valve_Storage_DB"."AV-39.06".FB_OPEN )
      wire#w5
      Contact( "IO_Valve_Storage_DB"."AV-34.06".FB_OPEN )
      wire#w6
      Contact( "IO_Valve_Storage_DB"."AV-34.07".FB_OPEN )
   END_RUNG wire#w7
   RUNG wire#w5
      Contact( "IO_Valve_Storage_DB"."AV-34.05".FB_OPEN )
   END_RUNG wire#w6
   RUNG wire#w6
      Contact( "IO_Valve_Storage_DB"."AV-34.08".FB_OPEN )
      Contact( "IO_Valve_Storage_DB"."AV-34.10".FB_OPEN )
   END_RUNG wire#w7
   RUNG wire#powerrail
      Contact( "IO_Valve_Storage_DB"."AV-39.06".FB_OPEN )
      Contact( "IO_Valve_Storage_DB"."AV-33.11".FB_OPEN )
   END_RUNG wire#w8
   RUNG wire#powerrail
      Contact( "T-24.00".State.Tank_inloading )
      Contact( "T-24.00".Cmd.Inload_Select_Tank_3 )
   END_RUNG wire#w9
   RUNG wire#powerrail
      Contact( "T-39.00".State.Tank_inloading )
   END_RUNG wire#w9
   RUNG wire#powerrail
      Contact( "T-33.00".State.Tank_inloading )
      Contact( "T-33.00".Cmd.Inload_Select_Tank_1 )
   END_RUNG wire#w9
   RUNG wire#powerrail
      Contact( "T-35.00".State.Tank_inloading )
      Contact( "T-35.00".Cmd.Inload_Select_Tank_1 )
   END_RUNG wire#w9
   RUNG wire#powerrail
      Contact( "T-84.00".State.Tank_inloading )
      Contact( "T-84.00".Cmd.Inload_Select_Tank_1 )
   END_RUNG wire#w9
   RUNG wire#powerrail
      Contact( "T-79.00".State.Tank_inloading )
      Contact( "T-79.00".Cmd.Inload_Select_Tank_3 )
   END_RUNG wire#w9
   RUNG wire#powerrail
      Contact( "T-33.00".State.Ready_For_Transfer )
   END_RUNG wire#w10
   RUNG wire#powerrail
      Contact( "T-33.00".Out_AV_Transfer )
   END_RUNG wire#w10
   RUNG wire#powerrail
      I_Contact( "Gen_Storage"."THE5 CIP"."CIP Request" )
      I_Contact( "T-24.00".CIP_Line_Req )
      I_Contact( "T-33.00".State."CIP Req" )
      I_Contact( "T-35.00".State."CIP Req" )
      I_Contact( "T-79.00".State."CIP Req" )
      I_Contact( "T-81.00".State."CIP Req" )
      I_Contact( "T-84.00".State."CIP Req" )
      I_Contact( "T-85.00".State."CIP Req" )
   END_RUNG wire#w11
   // the same network as SCL:
   "T-34.00"(IN_FBAV_Load := "T-34.00".Cmd.Inload_Select_Tank_1 AND "IO_Valve_Storage_DB"."AV-39.01".FB_OPEN AND "IO_Valve_Storage_DB"."AV-39.03".FB_OPEN AND "IO_Valve_Storage_DB"."AV-33.02".FB_OPEN AND "IO_Valve_Storage_DB"."AV-34.01".FB_OPEN AND ("IO_Valve_Storage_DB"."AV-34.04".FB_OPEN OR "IO_Valve_Storage_DB"."AV-34.03".FB_OPEN),   // "Storage_Tank_Multi_Inload"
             IN_FBAV_Transfer := "IO_Valve_Storage_DB"."AV-34.08".FB_OPEN AND ("IO_Valve_Storage_DB"."AV-34.10".FB_OPEN OR "IO_Valve_Storage_DB"."AV-34.09".FB_OPEN),
             IN_FBP_Transfer := "IO Motor MCC Panel Blending_DB"."P-34.01".QRUN,
             IN_FBAV_CIP_Tank := "IO_Valve_Storage_DB"."AV-39.06".FB_OPEN AND ("IO_Valve_Storage_DB"."AV-34.06".FB_OPEN OR "IO_Valve_Storage_DB"."AV-34.05".FB_OPEN) AND ("IO_Valve_Storage_DB"."AV-34.07".FB_OPEN OR ("IO_Valve_Storage_DB"."AV-34.08".FB_OPEN AND "IO_Valve_Storage_DB"."AV-34.10".FB_OPEN)),
             IN_FBAV_CIP_Line := "IO_Valve_Storage_DB"."AV-39.06".FB_OPEN AND "IO_Valve_Storage_DB"."AV-33.11".FB_OPEN,
             IN_LT01 := "IO Analog Storage_DB"."LT-34.01".QOUT,
             CIPPulse := "Timer 5S/30s",
             Filler_Product_Req := "Receive Product Request Filling Jonan",
             Filler_CIP_Req := "Receive CIP Enable Filling Jonan",
             Loading_Busy_1 := ("T-24.00".State.Tank_inloading AND "T-24.00".Cmd.Inload_Select_Tank_3) OR "T-39.00".State.Tank_inloading OR ("T-33.00".State.Tank_inloading AND "T-33.00".Cmd.Inload_Select_Tank_1) OR ("T-35.00".State.Tank_inloading AND "T-35.00".Cmd.Inload_Select_Tank_1) OR ("T-84.00".State.Tank_inloading AND "T-84.00".Cmd.Inload_Select_Tank_1) OR ("T-79.00".State.Tank_inloading AND "T-79.00".Cmd.Inload_Select_Tank_3),
             Transfer_Busy := "T-33.00".State.Ready_For_Transfer OR "T-33.00".Out_AV_Transfer,
             CIP_En := NOT "Gen_Storage"."THE5 CIP"."CIP Request" AND NOT "T-24.00".CIP_Line_Req AND NOT "T-33.00".State."CIP Req" AND NOT "T-35.00".State."CIP Req" AND NOT "T-79.00".State."CIP Req" AND NOT "T-81.00".State."CIP Req" AND NOT "T-84.00".State."CIP Req" AND NOT "T-85.00".State."CIP Req",
             CIP_Tank_Req => "Mix_to_CIP".CIP_Request."Storage THE 5"."T-34.00_CIP_Tank_Request",
             CIP_LineOK => "Mix_to_CIP".CIP_Line_OK."Storage THE 5"."T-34.00_CIP_Tank_LineOK");
END_REGION

REGION Network 25: T-34 Valve
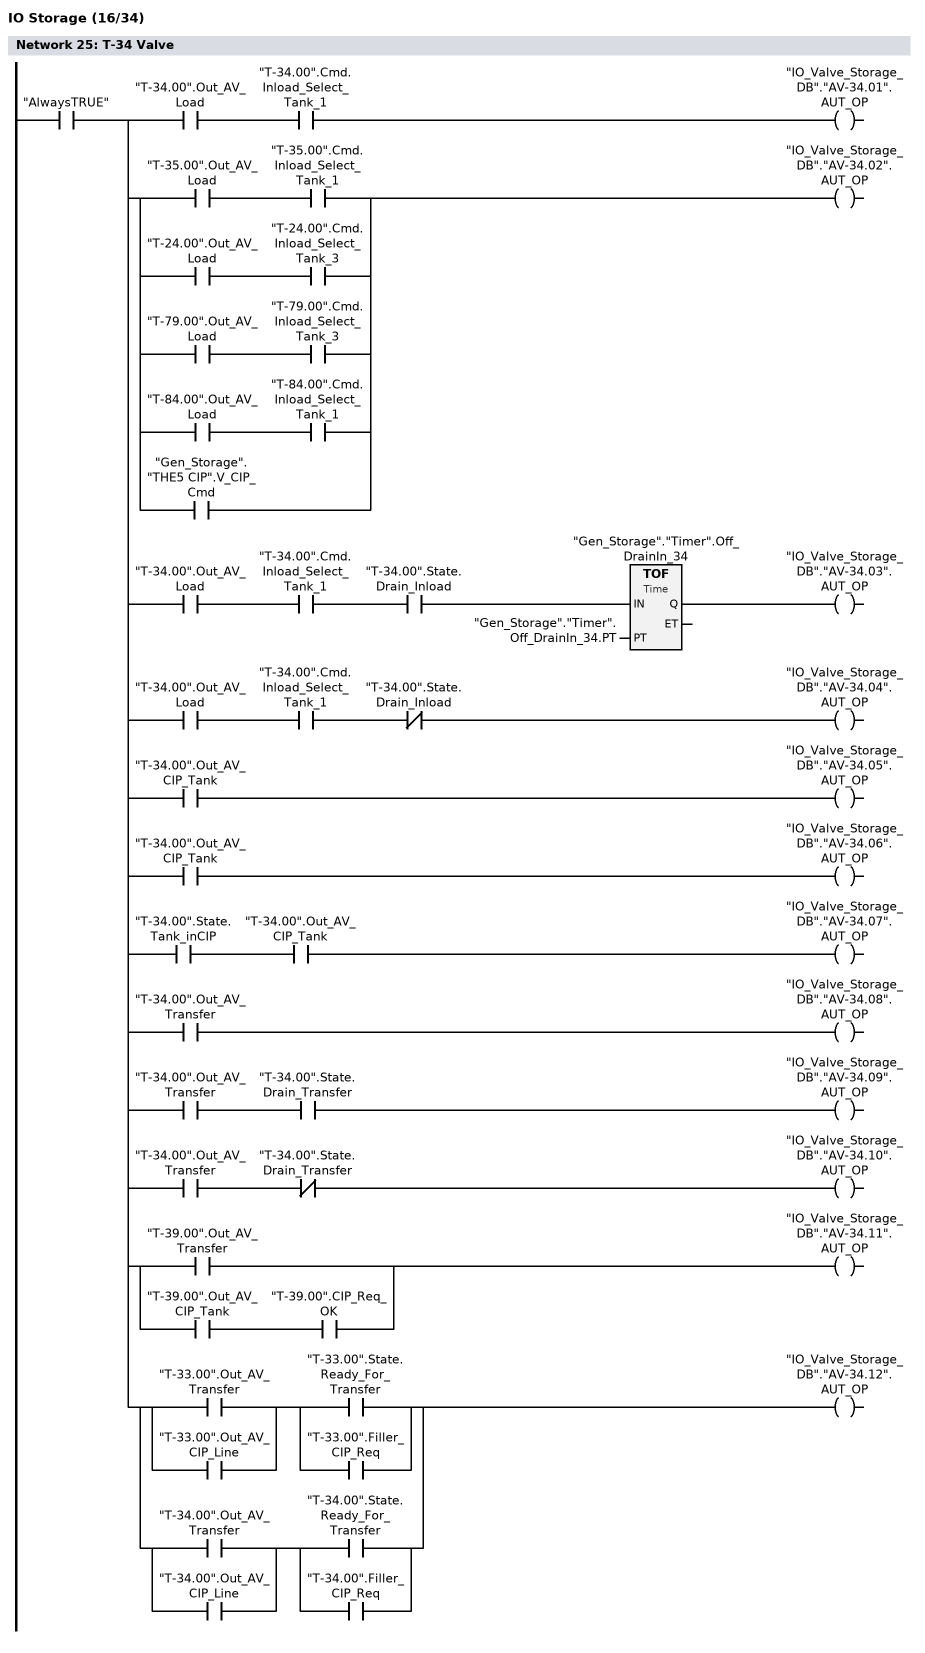
   RUNG wire#powerrail
      Contact( "AlwaysTRUE" )
      wire#w1
      Contact( "T-34.00".Out_AV_Load )
      Contact( "T-34.00".Cmd.Inload_Select_Tank_1 )
      Coil( "IO_Valve_Storage_DB"."AV-34.01".AUT_OP )
   END_RUNG
   RUNG wire#w1
      Contact( "T-35.00".Out_AV_Load )
      Contact( "T-35.00".Cmd.Inload_Select_Tank_1 )
      wire#w2
      Coil( "IO_Valve_Storage_DB"."AV-34.02".AUT_OP )
   END_RUNG
   RUNG wire#w1
      Contact( "T-24.00".Out_AV_Load )
      Contact( "T-24.00".Cmd.Inload_Select_Tank_3 )
   END_RUNG wire#w2
   RUNG wire#w1
      Contact( "T-79.00".Out_AV_Load )
      Contact( "T-79.00".Cmd.Inload_Select_Tank_3 )
   END_RUNG wire#w2
   RUNG wire#w1
      Contact( "T-84.00".Out_AV_Load )
      Contact( "T-84.00".Cmd.Inload_Select_Tank_1 )
   END_RUNG wire#w2
   RUNG wire#w1
      Contact( "Gen_Storage"."THE5 CIP".V_CIP_Cmd )
   END_RUNG wire#w2
   RUNG wire#w1
      Contact( "T-34.00".Out_AV_Load )
      Contact( "T-34.00".Cmd.Inload_Select_Tank_1 )
      Contact( "T-34.00".State.Drain_Inload )
      { S7_Templates := "time_type := Time" } "Gen_Storage"."Timer".Off_DrainIn_34.TOF(pt := "Gen_Storage"."Timer".Off_DrainIn_34.PT, et =>)
      Coil( "IO_Valve_Storage_DB"."AV-34.03".AUT_OP )
   END_RUNG
   RUNG wire#w1
      Contact( "T-34.00".Out_AV_Load )
      Contact( "T-34.00".Cmd.Inload_Select_Tank_1 )
      I_Contact( "T-34.00".State.Drain_Inload )
      Coil( "IO_Valve_Storage_DB"."AV-34.04".AUT_OP )
   END_RUNG
   RUNG wire#w1
      Contact( "T-34.00".Out_AV_CIP_Tank )
      Coil( "IO_Valve_Storage_DB"."AV-34.05".AUT_OP )
   END_RUNG
   RUNG wire#w1
      Contact( "T-34.00".Out_AV_CIP_Tank )
      Coil( "IO_Valve_Storage_DB"."AV-34.06".AUT_OP )
   END_RUNG
   RUNG wire#w1
      Contact( "T-34.00".State.Tank_inCIP )
      Contact( "T-34.00".Out_AV_CIP_Tank )
      Coil( "IO_Valve_Storage_DB"."AV-34.07".AUT_OP )
   END_RUNG
   RUNG wire#w1
      Contact( "T-34.00".Out_AV_Transfer )
      Coil( "IO_Valve_Storage_DB"."AV-34.08".AUT_OP )
   END_RUNG
   RUNG wire#w1
      Contact( "T-34.00".Out_AV_Transfer )
      Contact( "T-34.00".State.Drain_Transfer )
      Coil( "IO_Valve_Storage_DB"."AV-34.09".AUT_OP )
   END_RUNG
   RUNG wire#w1
      Contact( "T-34.00".Out_AV_Transfer )
      I_Contact( "T-34.00".State.Drain_Transfer )
      Coil( "IO_Valve_Storage_DB"."AV-34.10".AUT_OP )
   END_RUNG
   RUNG wire#w1
      Contact( "T-39.00".Out_AV_Transfer )
      wire#w3
      Coil( "IO_Valve_Storage_DB"."AV-34.11".AUT_OP )
   END_RUNG
   RUNG wire#w1
      Contact( "T-39.00".Out_AV_CIP_Tank )
      Contact( "T-39.00".CIP_Req_OK )
   END_RUNG wire#w3
   RUNG wire#w1
      Contact( "T-33.00".Out_AV_Transfer )
      wire#w4
      Contact( "T-33.00".State.Ready_For_Transfer )
      wire#w5
      Coil( "IO_Valve_Storage_DB"."AV-34.12".AUT_OP )
   END_RUNG
   RUNG wire#w1
      Contact( "T-33.00".Out_AV_CIP_Line )
   END_RUNG wire#w4
   RUNG wire#w4
      Contact( "T-33.00".Filler_CIP_Req )
   END_RUNG wire#w5
   RUNG wire#w1
      Contact( "T-34.00".Out_AV_Transfer )
      wire#w6
      Contact( "T-34.00".State.Ready_For_Transfer )
   END_RUNG wire#w5
   RUNG wire#w1
      Contact( "T-34.00".Out_AV_CIP_Line )
   END_RUNG wire#w6
   RUNG wire#w6
      Contact( "T-34.00".Filler_CIP_Req )
   END_RUNG wire#w5
   // the same network as SCL:
   "IO_Valve_Storage_DB"."AV-34.01".AUT_OP := "AlwaysTRUE" AND "T-34.00".Out_AV_Load AND "T-34.00".Cmd.Inload_Select_Tank_1;
   "IO_Valve_Storage_DB"."AV-34.02".AUT_OP := "AlwaysTRUE" AND (("T-35.00".Out_AV_Load AND "T-35.00".Cmd.Inload_Select_Tank_1) OR ("T-24.00".Out_AV_Load AND "T-24.00".Cmd.Inload_Select_Tank_3) OR ("T-79.00".Out_AV_Load AND "T-79.00".Cmd.Inload_Select_Tank_3) OR ("T-84.00".Out_AV_Load AND "T-84.00".Cmd.Inload_Select_Tank_1) OR "Gen_Storage"."THE5 CIP".V_CIP_Cmd);
   "Gen_Storage"."Timer".Off_DrainIn_34.TOF(IN := "AlwaysTRUE" AND "T-34.00".Out_AV_Load AND "T-34.00".Cmd.Inload_Select_Tank_1 AND "T-34.00".State.Drain_Inload,
                           PT := "Gen_Storage"."Timer".Off_DrainIn_34.PT);
   "IO_Valve_Storage_DB"."AV-34.03".AUT_OP := "Gen_Storage"."Timer".Off_DrainIn_34.Q;
   "IO_Valve_Storage_DB"."AV-34.04".AUT_OP := "AlwaysTRUE" AND "T-34.00".Out_AV_Load AND "T-34.00".Cmd.Inload_Select_Tank_1 AND NOT "T-34.00".State.Drain_Inload;
   "IO_Valve_Storage_DB"."AV-34.05".AUT_OP := "AlwaysTRUE" AND "T-34.00".Out_AV_CIP_Tank;
   "IO_Valve_Storage_DB"."AV-34.06".AUT_OP := "AlwaysTRUE" AND "T-34.00".Out_AV_CIP_Tank;
   "IO_Valve_Storage_DB"."AV-34.07".AUT_OP := "AlwaysTRUE" AND "T-34.00".State.Tank_inCIP AND "T-34.00".Out_AV_CIP_Tank;
   "IO_Valve_Storage_DB"."AV-34.08".AUT_OP := "AlwaysTRUE" AND "T-34.00".Out_AV_Transfer;
   "IO_Valve_Storage_DB"."AV-34.09".AUT_OP := "AlwaysTRUE" AND "T-34.00".Out_AV_Transfer AND "T-34.00".State.Drain_Transfer;
   "IO_Valve_Storage_DB"."AV-34.10".AUT_OP := "AlwaysTRUE" AND "T-34.00".Out_AV_Transfer AND NOT "T-34.00".State.Drain_Transfer;
   "IO_Valve_Storage_DB"."AV-34.11".AUT_OP := "AlwaysTRUE" AND ("T-39.00".Out_AV_Transfer OR ("T-39.00".Out_AV_CIP_Tank AND "T-39.00".CIP_Req_OK));
   "IO_Valve_Storage_DB"."AV-34.12".AUT_OP := "AlwaysTRUE" AND ((("T-33.00".Out_AV_Transfer OR "T-33.00".Out_AV_CIP_Line) AND ("T-33.00".State.Ready_For_Transfer OR "T-33.00".Filler_CIP_Req)) OR (("T-34.00".Out_AV_Transfer OR "T-34.00".Out_AV_CIP_Line) AND ("T-34.00".State.Ready_For_Transfer OR "T-34.00".Filler_CIP_Req)));
END_REGION

REGION Network 26: T-33.00 and T-34.00 CIP Line Request and LineOK
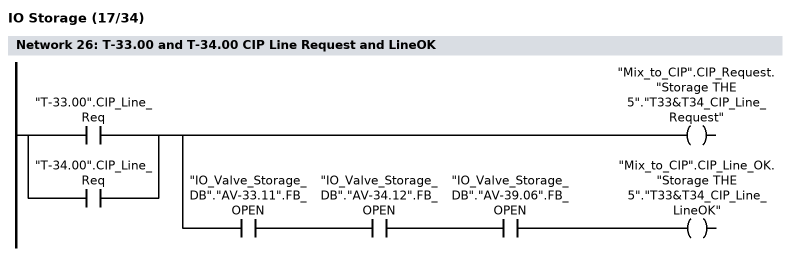
   RUNG wire#powerrail
      Contact( "T-33.00".CIP_Line_Req )
      wire#w1
      Coil( "Mix_to_CIP".CIP_Request."Storage THE 5"."T33&T34_CIP_Line_Request" )
   END_RUNG
   RUNG wire#powerrail
      Contact( "T-34.00".CIP_Line_Req )
   END_RUNG wire#w1
   RUNG wire#w1
      Contact( "IO_Valve_Storage_DB"."AV-33.11".FB_OPEN )
      Contact( "IO_Valve_Storage_DB"."AV-34.12".FB_OPEN )
      Contact( "IO_Valve_Storage_DB"."AV-39.06".FB_OPEN )
      Coil( "Mix_to_CIP".CIP_Line_OK."Storage THE 5"."T33&T34_CIP_Line_LineOK" )
   END_RUNG
   // the same network as SCL:
   "Mix_to_CIP".CIP_Request."Storage THE 5"."T33&T34_CIP_Line_Request" := "T-33.00".CIP_Line_Req OR "T-34.00".CIP_Line_Req;
   "Mix_to_CIP".CIP_Line_OK."Storage THE 5"."T33&T34_CIP_Line_LineOK" := "Mix_to_CIP".CIP_Request."Storage THE 5"."T33&T34_CIP_Line_Request" AND "IO_Valve_Storage_DB"."AV-33.11".FB_OPEN AND "IO_Valve_Storage_DB"."AV-34.12".FB_OPEN AND "IO_Valve_Storage_DB"."AV-39.06".FB_OPEN;
END_REGION

REGION Network 28: T-35.00 ST-10
   // Inload 1 : THE 5
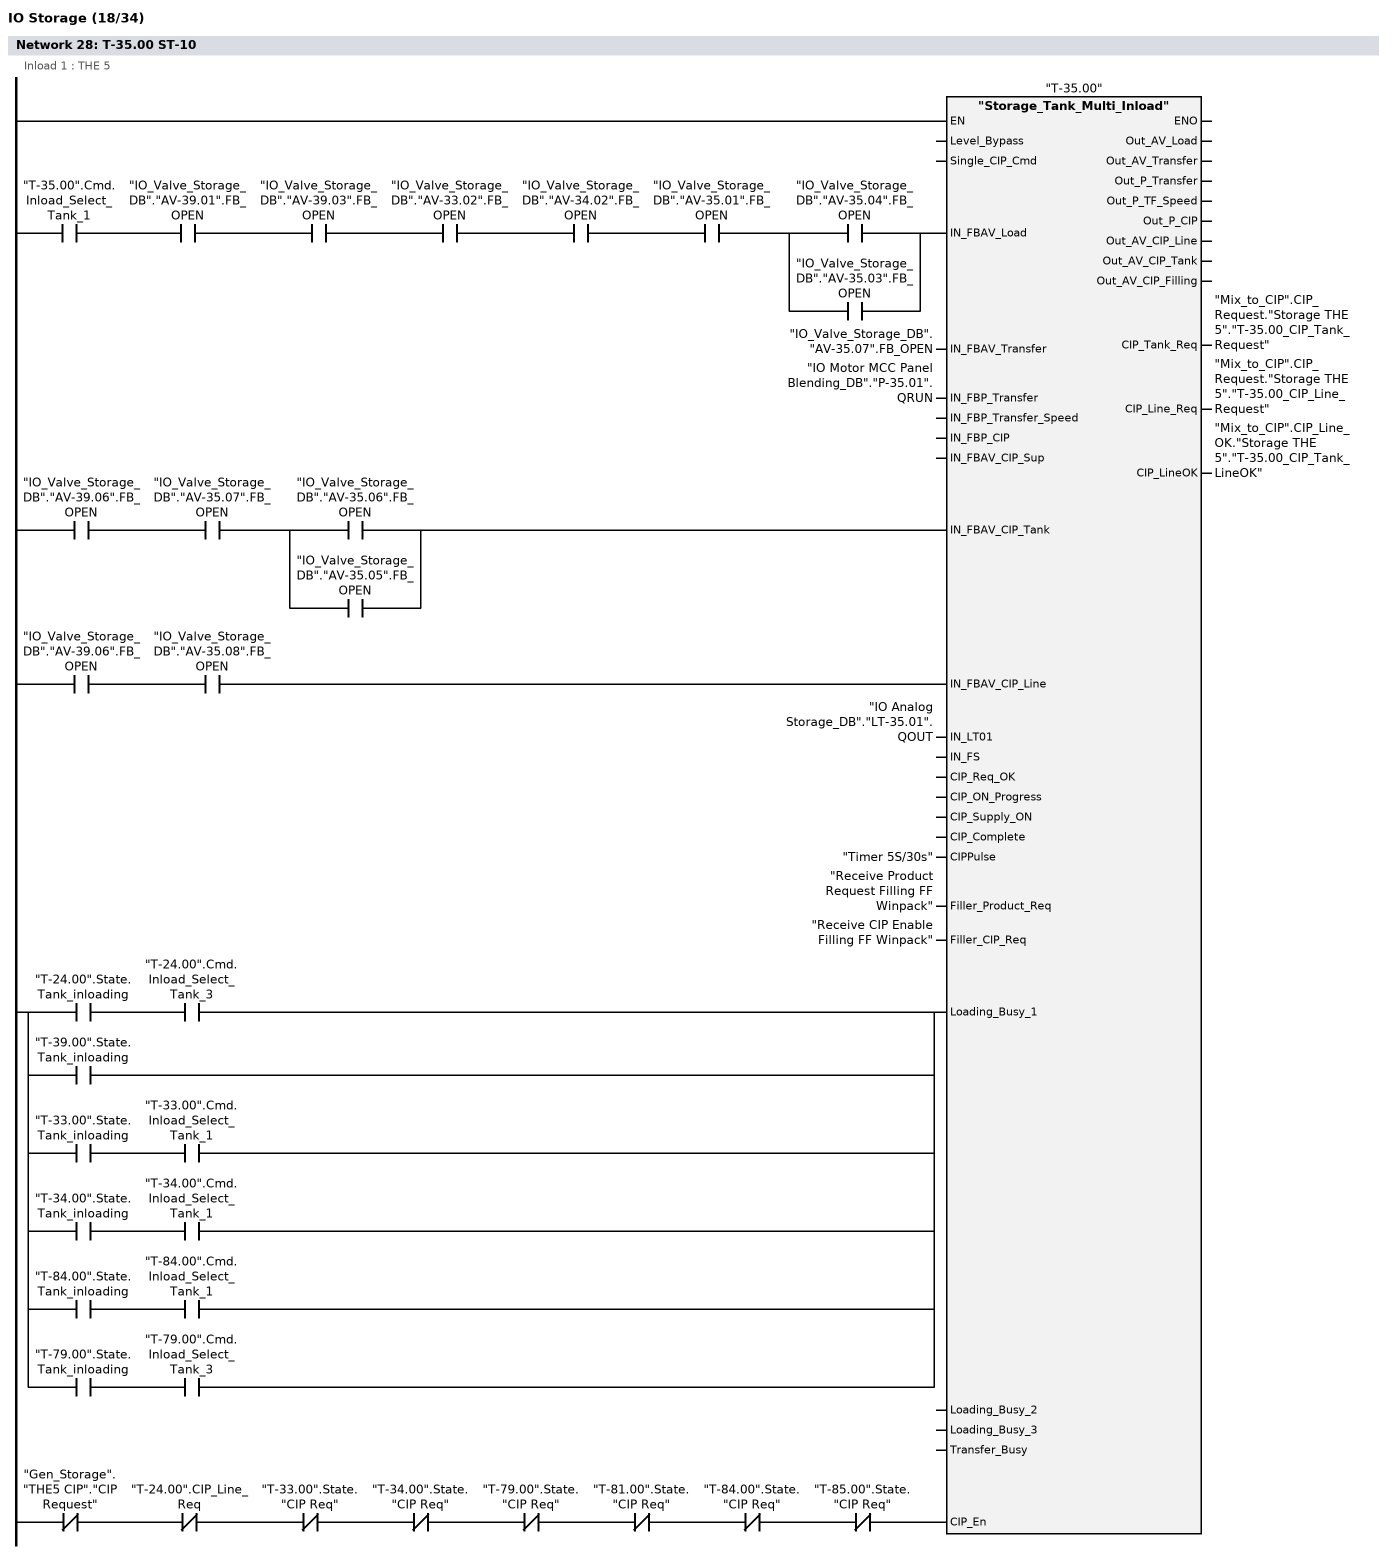
   RUNG wire#powerrail
      "T-35.00"(IN_FBAV_Load := wire#w2, IN_FBAV_CIP_Tank := wire#w4, IN_FBAV_CIP_Line := wire#w5, Loading_Busy_1 := wire#w6, CIP_En := wire#w7, Level_Bypass :=, Single_CIP_Cmd :=, IN_FBAV_Transfer := "IO_Valve_Storage_DB"."AV-35.07".FB_OPEN, IN_FBP_Transfer := "IO Motor MCC Panel Blending_DB"."P-35.01".QRUN, IN_FBP_Transfer_Speed :=, IN_FBP_CIP :=, IN_FBAV_CIP_Sup :=, IN_LT01 := "IO Analog Storage_DB"."LT-35.01".QOUT, IN_FS :=, CIP_Req_OK :=, CIP_ON_Progress :=, CIP_Supply_ON :=, CIP_Complete :=, CIPPulse := "Timer 5S/30s", Filler_Product_Req := "Receive Product Request Filling FF Winpack", Filler_CIP_Req := "Receive CIP Enable Filling FF Winpack", Loading_Busy_2 :=, Loading_Busy_3 :=, Transfer_Busy :=, Out_AV_Load =>, Out_AV_Transfer =>, Out_P_Transfer =>, Out_P_TF_Speed =>, Out_P_CIP =>, Out_AV_CIP_Line =>, Out_AV_CIP_Tank =>, Out_AV_CIP_Filling =>, CIP_Tank_Req => "Mix_to_CIP".CIP_Request."Storage THE 5"."T-35.00_CIP_Tank_Request", CIP_Line_Req => "Mix_to_CIP".CIP_Request."Storage THE 5"."T-35.00_CIP_Line_Request", CIP_LineOK => "Mix_to_CIP".CIP_Line_OK."Storage THE 5"."T-35.00_CIP_Tank_LineOK")
   END_RUNG
   RUNG wire#powerrail
      Contact( "T-35.00".Cmd.Inload_Select_Tank_1 )
      Contact( "IO_Valve_Storage_DB"."AV-39.01".FB_OPEN )
      Contact( "IO_Valve_Storage_DB"."AV-39.03".FB_OPEN )
      Contact( "IO_Valve_Storage_DB"."AV-33.02".FB_OPEN )
      Contact( "IO_Valve_Storage_DB"."AV-34.02".FB_OPEN )
      Contact( "IO_Valve_Storage_DB"."AV-35.01".FB_OPEN )
      wire#w1
      Contact( "IO_Valve_Storage_DB"."AV-35.04".FB_OPEN )
   END_RUNG wire#w2
   RUNG wire#w1
      Contact( "IO_Valve_Storage_DB"."AV-35.03".FB_OPEN )
   END_RUNG wire#w2
   RUNG wire#powerrail
      Contact( "IO_Valve_Storage_DB"."AV-39.06".FB_OPEN )
      Contact( "IO_Valve_Storage_DB"."AV-35.07".FB_OPEN )
      wire#w3
      Contact( "IO_Valve_Storage_DB"."AV-35.06".FB_OPEN )
   END_RUNG wire#w4
   RUNG wire#w3
      Contact( "IO_Valve_Storage_DB"."AV-35.05".FB_OPEN )
   END_RUNG wire#w4
   RUNG wire#powerrail
      Contact( "IO_Valve_Storage_DB"."AV-39.06".FB_OPEN )
      Contact( "IO_Valve_Storage_DB"."AV-35.08".FB_OPEN )
   END_RUNG wire#w5
   RUNG wire#powerrail
      Contact( "T-24.00".State.Tank_inloading )
      Contact( "T-24.00".Cmd.Inload_Select_Tank_3 )
   END_RUNG wire#w6
   RUNG wire#powerrail
      Contact( "T-39.00".State.Tank_inloading )
   END_RUNG wire#w6
   RUNG wire#powerrail
      Contact( "T-33.00".State.Tank_inloading )
      Contact( "T-33.00".Cmd.Inload_Select_Tank_1 )
   END_RUNG wire#w6
   RUNG wire#powerrail
      Contact( "T-34.00".State.Tank_inloading )
      Contact( "T-34.00".Cmd.Inload_Select_Tank_1 )
   END_RUNG wire#w6
   RUNG wire#powerrail
      Contact( "T-84.00".State.Tank_inloading )
      Contact( "T-84.00".Cmd.Inload_Select_Tank_1 )
   END_RUNG wire#w6
   RUNG wire#powerrail
      Contact( "T-79.00".State.Tank_inloading )
      Contact( "T-79.00".Cmd.Inload_Select_Tank_3 )
   END_RUNG wire#w6
   RUNG wire#powerrail
      I_Contact( "Gen_Storage"."THE5 CIP"."CIP Request" )
      I_Contact( "T-24.00".CIP_Line_Req )
      I_Contact( "T-33.00".State."CIP Req" )
      I_Contact( "T-34.00".State."CIP Req" )
      I_Contact( "T-79.00".State."CIP Req" )
      I_Contact( "T-81.00".State."CIP Req" )
      I_Contact( "T-84.00".State."CIP Req" )
      I_Contact( "T-85.00".State."CIP Req" )
   END_RUNG wire#w7
   // the same network as SCL:
   "T-35.00"(IN_FBAV_Load := "T-35.00".Cmd.Inload_Select_Tank_1 AND "IO_Valve_Storage_DB"."AV-39.01".FB_OPEN AND "IO_Valve_Storage_DB"."AV-39.03".FB_OPEN AND "IO_Valve_Storage_DB"."AV-33.02".FB_OPEN AND "IO_Valve_Storage_DB"."AV-34.02".FB_OPEN AND "IO_Valve_Storage_DB"."AV-35.01".FB_OPEN AND ("IO_Valve_Storage_DB"."AV-35.04".FB_OPEN OR "IO_Valve_Storage_DB"."AV-35.03".FB_OPEN),   // "Storage_Tank_Multi_Inload"
             IN_FBAV_Transfer := "IO_Valve_Storage_DB"."AV-35.07".FB_OPEN,
             IN_FBP_Transfer := "IO Motor MCC Panel Blending_DB"."P-35.01".QRUN,
             IN_FBAV_CIP_Tank := "IO_Valve_Storage_DB"."AV-39.06".FB_OPEN AND "IO_Valve_Storage_DB"."AV-35.07".FB_OPEN AND ("IO_Valve_Storage_DB"."AV-35.06".FB_OPEN OR "IO_Valve_Storage_DB"."AV-35.05".FB_OPEN),
             IN_FBAV_CIP_Line := "IO_Valve_Storage_DB"."AV-39.06".FB_OPEN AND "IO_Valve_Storage_DB"."AV-35.08".FB_OPEN,
             IN_LT01 := "IO Analog Storage_DB"."LT-35.01".QOUT,
             CIPPulse := "Timer 5S/30s",
             Filler_Product_Req := "Receive Product Request Filling FF Winpack",
             Filler_CIP_Req := "Receive CIP Enable Filling FF Winpack",
             Loading_Busy_1 := ("T-24.00".State.Tank_inloading AND "T-24.00".Cmd.Inload_Select_Tank_3) OR "T-39.00".State.Tank_inloading OR ("T-33.00".State.Tank_inloading AND "T-33.00".Cmd.Inload_Select_Tank_1) OR ("T-34.00".State.Tank_inloading AND "T-34.00".Cmd.Inload_Select_Tank_1) OR ("T-84.00".State.Tank_inloading AND "T-84.00".Cmd.Inload_Select_Tank_1) OR ("T-79.00".State.Tank_inloading AND "T-79.00".Cmd.Inload_Select_Tank_3),
             CIP_En := NOT "Gen_Storage"."THE5 CIP"."CIP Request" AND NOT "T-24.00".CIP_Line_Req AND NOT "T-33.00".State."CIP Req" AND NOT "T-34.00".State."CIP Req" AND NOT "T-79.00".State."CIP Req" AND NOT "T-81.00".State."CIP Req" AND NOT "T-84.00".State."CIP Req" AND NOT "T-85.00".State."CIP Req",
             CIP_Tank_Req => "Mix_to_CIP".CIP_Request."Storage THE 5"."T-35.00_CIP_Tank_Request",
             CIP_Line_Req => "Mix_to_CIP".CIP_Request."Storage THE 5"."T-35.00_CIP_Line_Request",
             CIP_LineOK => "Mix_to_CIP".CIP_Line_OK."Storage THE 5"."T-35.00_CIP_Tank_LineOK");
END_REGION

REGION Network 29: T-35 Valve
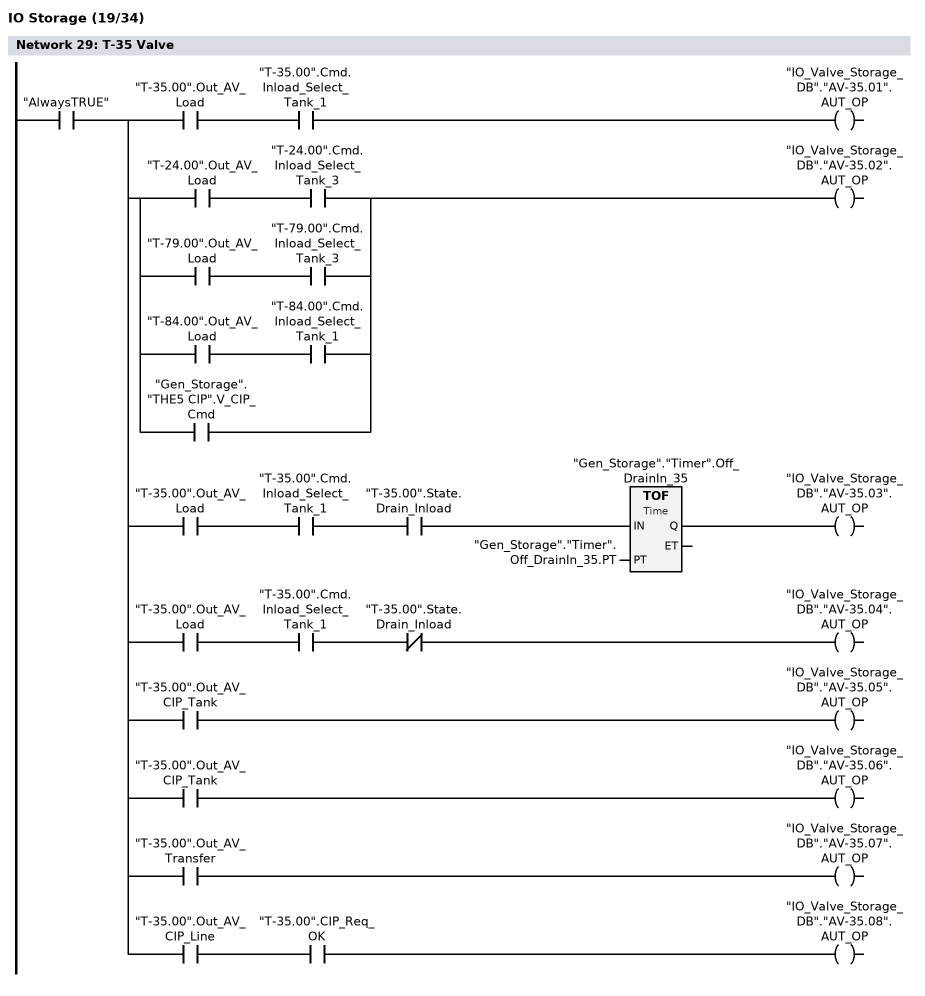
   RUNG wire#powerrail
      Contact( "AlwaysTRUE" )
      wire#w1
      Contact( "T-35.00".Out_AV_Load )
      Contact( "T-35.00".Cmd.Inload_Select_Tank_1 )
      Coil( "IO_Valve_Storage_DB"."AV-35.01".AUT_OP )
   END_RUNG
   RUNG wire#w1
      Contact( "T-24.00".Out_AV_Load )
      Contact( "T-24.00".Cmd.Inload_Select_Tank_3 )
      wire#w2
      Coil( "IO_Valve_Storage_DB"."AV-35.02".AUT_OP )
   END_RUNG
   RUNG wire#w1
      Contact( "T-79.00".Out_AV_Load )
      Contact( "T-79.00".Cmd.Inload_Select_Tank_3 )
   END_RUNG wire#w2
   RUNG wire#w1
      Contact( "T-84.00".Out_AV_Load )
      Contact( "T-84.00".Cmd.Inload_Select_Tank_1 )
   END_RUNG wire#w2
   RUNG wire#w1
      Contact( "Gen_Storage"."THE5 CIP".V_CIP_Cmd )
   END_RUNG wire#w2
   RUNG wire#w1
      Contact( "T-35.00".Out_AV_Load )
      Contact( "T-35.00".Cmd.Inload_Select_Tank_1 )
      Contact( "T-35.00".State.Drain_Inload )
      { S7_Templates := "time_type := Time" } "Gen_Storage"."Timer".Off_DrainIn_35.TOF(pt := "Gen_Storage"."Timer".Off_DrainIn_35.PT, et =>)
      Coil( "IO_Valve_Storage_DB"."AV-35.03".AUT_OP )
   END_RUNG
   RUNG wire#w1
      Contact( "T-35.00".Out_AV_Load )
      Contact( "T-35.00".Cmd.Inload_Select_Tank_1 )
      I_Contact( "T-35.00".State.Drain_Inload )
      Coil( "IO_Valve_Storage_DB"."AV-35.04".AUT_OP )
   END_RUNG
   RUNG wire#w1
      Contact( "T-35.00".Out_AV_CIP_Tank )
      Coil( "IO_Valve_Storage_DB"."AV-35.05".AUT_OP )
   END_RUNG
   RUNG wire#w1
      Contact( "T-35.00".Out_AV_CIP_Tank )
      Coil( "IO_Valve_Storage_DB"."AV-35.06".AUT_OP )
   END_RUNG
   RUNG wire#w1
      Contact( "T-35.00".Out_AV_Transfer )
      Coil( "IO_Valve_Storage_DB"."AV-35.07".AUT_OP )
   END_RUNG
   RUNG wire#w1
      Contact( "T-35.00".Out_AV_CIP_Line )
      Contact( "T-35.00".CIP_Req_OK )
      Coil( "IO_Valve_Storage_DB"."AV-35.08".AUT_OP )
   END_RUNG
   // the same network as SCL:
   "IO_Valve_Storage_DB"."AV-35.01".AUT_OP := "AlwaysTRUE" AND "T-35.00".Out_AV_Load AND "T-35.00".Cmd.Inload_Select_Tank_1;
   "IO_Valve_Storage_DB"."AV-35.02".AUT_OP := "AlwaysTRUE" AND (("T-24.00".Out_AV_Load AND "T-24.00".Cmd.Inload_Select_Tank_3) OR ("T-79.00".Out_AV_Load AND "T-79.00".Cmd.Inload_Select_Tank_3) OR ("T-84.00".Out_AV_Load AND "T-84.00".Cmd.Inload_Select_Tank_1) OR "Gen_Storage"."THE5 CIP".V_CIP_Cmd);
   "Gen_Storage"."Timer".Off_DrainIn_35.TOF(IN := "AlwaysTRUE" AND "T-35.00".Out_AV_Load AND "T-35.00".Cmd.Inload_Select_Tank_1 AND "T-35.00".State.Drain_Inload,
                           PT := "Gen_Storage"."Timer".Off_DrainIn_35.PT);
   "IO_Valve_Storage_DB"."AV-35.03".AUT_OP := "Gen_Storage"."Timer".Off_DrainIn_35.Q;
   "IO_Valve_Storage_DB"."AV-35.04".AUT_OP := "AlwaysTRUE" AND "T-35.00".Out_AV_Load AND "T-35.00".Cmd.Inload_Select_Tank_1 AND NOT "T-35.00".State.Drain_Inload;
   "IO_Valve_Storage_DB"."AV-35.05".AUT_OP := "AlwaysTRUE" AND "T-35.00".Out_AV_CIP_Tank;
   "IO_Valve_Storage_DB"."AV-35.06".AUT_OP := "AlwaysTRUE" AND "T-35.00".Out_AV_CIP_Tank;
   "IO_Valve_Storage_DB"."AV-35.07".AUT_OP := "AlwaysTRUE" AND "T-35.00".Out_AV_Transfer;
   "IO_Valve_Storage_DB"."AV-35.08".AUT_OP := "AlwaysTRUE" AND "T-35.00".Out_AV_CIP_Line AND "T-35.00".CIP_Req_OK;
END_REGION

REGION Network 30: Line THE 5
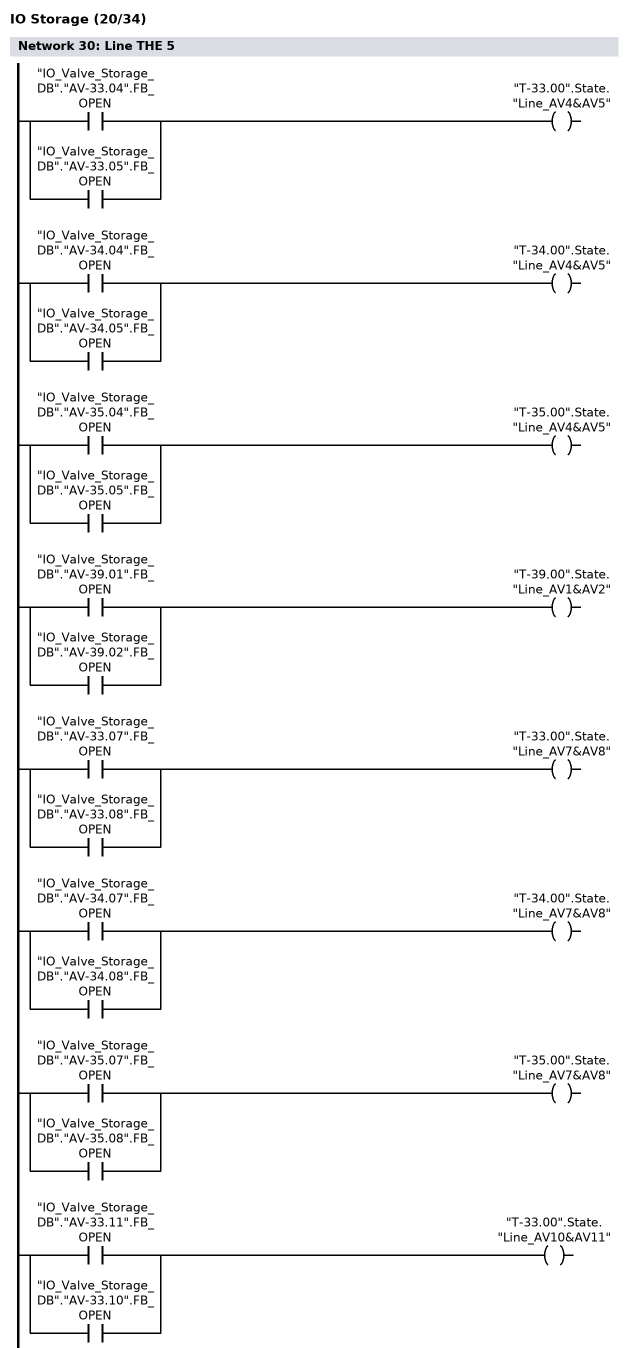
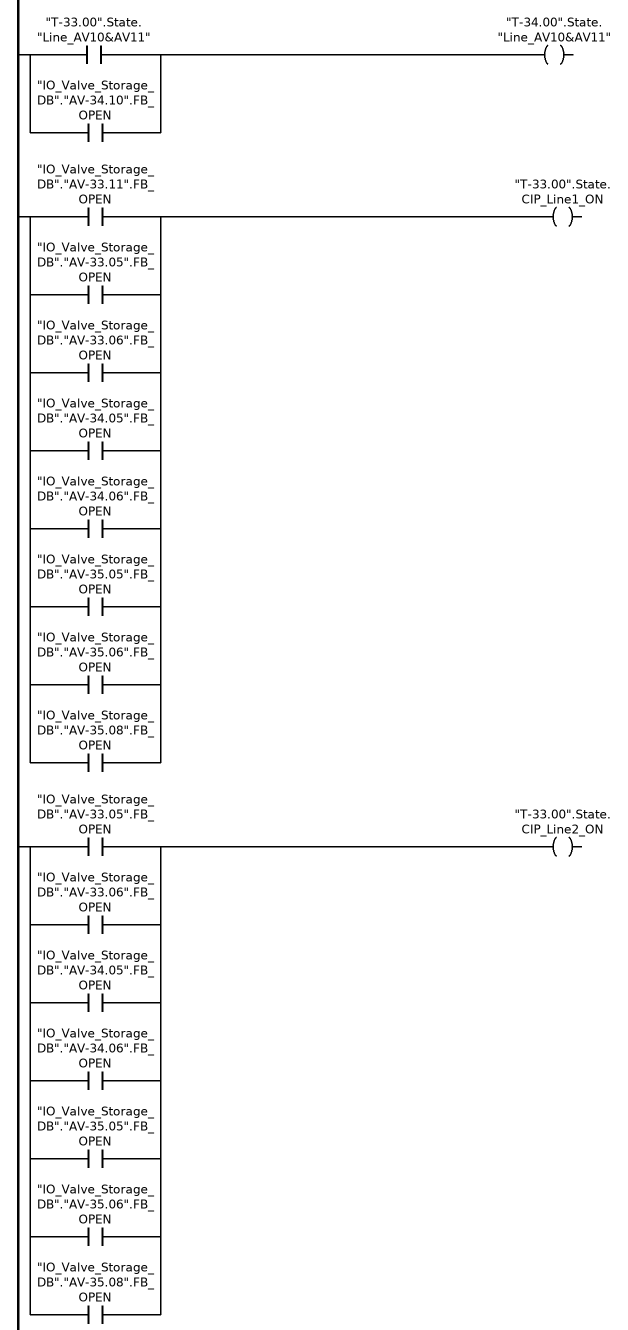
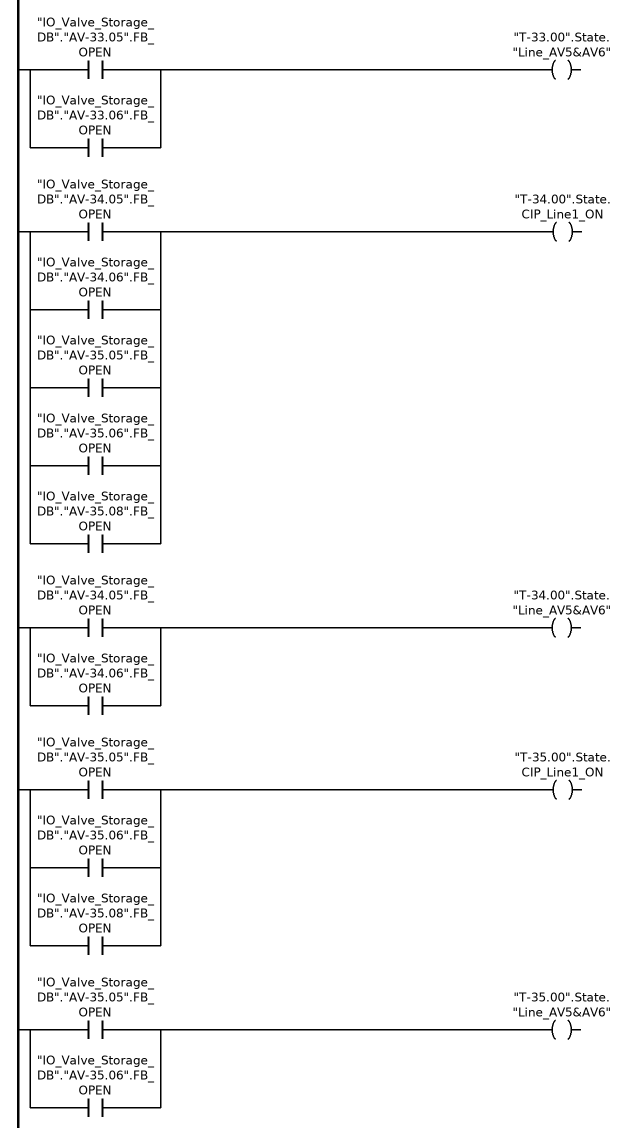
   RUNG wire#powerrail
      Contact( "IO_Valve_Storage_DB"."AV-33.04".FB_OPEN )
      wire#w1
      Coil( "T-33.00".State."Line_AV4&AV5" )
   END_RUNG
   RUNG wire#powerrail
      Contact( "IO_Valve_Storage_DB"."AV-33.05".FB_OPEN )
   END_RUNG wire#w1
   RUNG wire#powerrail
      Contact( "IO_Valve_Storage_DB"."AV-34.04".FB_OPEN )
      wire#w2
      Coil( "T-34.00".State."Line_AV4&AV5" )
   END_RUNG
   RUNG wire#powerrail
      Contact( "IO_Valve_Storage_DB"."AV-34.05".FB_OPEN )
   END_RUNG wire#w2
   RUNG wire#powerrail
      Contact( "IO_Valve_Storage_DB"."AV-35.04".FB_OPEN )
      wire#w3
      Coil( "T-35.00".State."Line_AV4&AV5" )
   END_RUNG
   RUNG wire#powerrail
      Contact( "IO_Valve_Storage_DB"."AV-35.05".FB_OPEN )
   END_RUNG wire#w3
   RUNG wire#powerrail
      Contact( "IO_Valve_Storage_DB"."AV-39.01".FB_OPEN )
      wire#w4
      Coil( "T-39.00".State."Line_AV1&AV2" )
   END_RUNG
   RUNG wire#powerrail
      Contact( "IO_Valve_Storage_DB"."AV-39.02".FB_OPEN )
   END_RUNG wire#w4
   RUNG wire#powerrail
      Contact( "IO_Valve_Storage_DB"."AV-33.07".FB_OPEN )
      wire#w5
      Coil( "T-33.00".State."Line_AV7&AV8" )
   END_RUNG
   RUNG wire#powerrail
      Contact( "IO_Valve_Storage_DB"."AV-33.08".FB_OPEN )
   END_RUNG wire#w5
   RUNG wire#powerrail
      Contact( "IO_Valve_Storage_DB"."AV-34.07".FB_OPEN )
      wire#w6
      Coil( "T-34.00".State."Line_AV7&AV8" )
   END_RUNG
   RUNG wire#powerrail
      Contact( "IO_Valve_Storage_DB"."AV-34.08".FB_OPEN )
   END_RUNG wire#w6
   RUNG wire#powerrail
      Contact( "IO_Valve_Storage_DB"."AV-35.07".FB_OPEN )
      wire#w7
      Coil( "T-35.00".State."Line_AV7&AV8" )
   END_RUNG
   RUNG wire#powerrail
      Contact( "IO_Valve_Storage_DB"."AV-35.08".FB_OPEN )
   END_RUNG wire#w7
   RUNG wire#powerrail
      Contact( "IO_Valve_Storage_DB"."AV-33.11".FB_OPEN )
      wire#w8
      Coil( "T-33.00".State."Line_AV10&AV11" )
   END_RUNG
   RUNG wire#powerrail
      Contact( "IO_Valve_Storage_DB"."AV-33.10".FB_OPEN )
   END_RUNG wire#w8
   RUNG wire#powerrail
      Contact( "T-33.00".State."Line_AV10&AV11" )
      wire#w9
      Coil( "T-34.00".State."Line_AV10&AV11" )
   END_RUNG
   RUNG wire#powerrail
      Contact( "IO_Valve_Storage_DB"."AV-34.10".FB_OPEN )
   END_RUNG wire#w9
   RUNG wire#powerrail
      Contact( "IO_Valve_Storage_DB"."AV-33.11".FB_OPEN )
      wire#w10
      Coil( "T-33.00".State.CIP_Line1_ON )
   END_RUNG
   RUNG wire#powerrail
      Contact( "IO_Valve_Storage_DB"."AV-33.05".FB_OPEN )
   END_RUNG wire#w10
   RUNG wire#powerrail
      Contact( "IO_Valve_Storage_DB"."AV-33.06".FB_OPEN )
   END_RUNG wire#w10
   RUNG wire#powerrail
      Contact( "IO_Valve_Storage_DB"."AV-34.05".FB_OPEN )
   END_RUNG wire#w10
   RUNG wire#powerrail
      Contact( "IO_Valve_Storage_DB"."AV-34.06".FB_OPEN )
   END_RUNG wire#w10
   RUNG wire#powerrail
      Contact( "IO_Valve_Storage_DB"."AV-35.05".FB_OPEN )
   END_RUNG wire#w10
   RUNG wire#powerrail
      Contact( "IO_Valve_Storage_DB"."AV-35.06".FB_OPEN )
   END_RUNG wire#w10
   RUNG wire#powerrail
      Contact( "IO_Valve_Storage_DB"."AV-35.08".FB_OPEN )
   END_RUNG wire#w10
   RUNG wire#powerrail
      Contact( "IO_Valve_Storage_DB"."AV-33.05".FB_OPEN )
      wire#w11
      Coil( "T-33.00".State.CIP_Line2_ON )
   END_RUNG
   RUNG wire#powerrail
      Contact( "IO_Valve_Storage_DB"."AV-33.06".FB_OPEN )
   END_RUNG wire#w11
   RUNG wire#powerrail
      Contact( "IO_Valve_Storage_DB"."AV-34.05".FB_OPEN )
   END_RUNG wire#w11
   RUNG wire#powerrail
      Contact( "IO_Valve_Storage_DB"."AV-34.06".FB_OPEN )
   END_RUNG wire#w11
   RUNG wire#powerrail
      Contact( "IO_Valve_Storage_DB"."AV-35.05".FB_OPEN )
   END_RUNG wire#w11
   RUNG wire#powerrail
      Contact( "IO_Valve_Storage_DB"."AV-35.06".FB_OPEN )
   END_RUNG wire#w11
   RUNG wire#powerrail
      Contact( "IO_Valve_Storage_DB"."AV-35.08".FB_OPEN )
   END_RUNG wire#w11
   RUNG wire#powerrail
      Contact( "IO_Valve_Storage_DB"."AV-33.05".FB_OPEN )
      wire#w12
      Coil( "T-33.00".State."Line_AV5&AV6" )
   END_RUNG
   RUNG wire#powerrail
      Contact( "IO_Valve_Storage_DB"."AV-33.06".FB_OPEN )
   END_RUNG wire#w12
   RUNG wire#powerrail
      Contact( "IO_Valve_Storage_DB"."AV-34.05".FB_OPEN )
      wire#w13
      Coil( "T-34.00".State.CIP_Line1_ON )
   END_RUNG
   RUNG wire#powerrail
      Contact( "IO_Valve_Storage_DB"."AV-34.06".FB_OPEN )
   END_RUNG wire#w13
   RUNG wire#powerrail
      Contact( "IO_Valve_Storage_DB"."AV-35.05".FB_OPEN )
   END_RUNG wire#w13
   RUNG wire#powerrail
      Contact( "IO_Valve_Storage_DB"."AV-35.06".FB_OPEN )
   END_RUNG wire#w13
   RUNG wire#powerrail
      Contact( "IO_Valve_Storage_DB"."AV-35.08".FB_OPEN )
   END_RUNG wire#w13
   RUNG wire#powerrail
      Contact( "IO_Valve_Storage_DB"."AV-34.05".FB_OPEN )
      wire#w14
      Coil( "T-34.00".State."Line_AV5&AV6" )
   END_RUNG
   RUNG wire#powerrail
      Contact( "IO_Valve_Storage_DB"."AV-34.06".FB_OPEN )
   END_RUNG wire#w14
   RUNG wire#powerrail
      Contact( "IO_Valve_Storage_DB"."AV-35.05".FB_OPEN )
      wire#w15
      Coil( "T-35.00".State.CIP_Line1_ON )
   END_RUNG
   RUNG wire#powerrail
      Contact( "IO_Valve_Storage_DB"."AV-35.06".FB_OPEN )
   END_RUNG wire#w15
   RUNG wire#powerrail
      Contact( "IO_Valve_Storage_DB"."AV-35.08".FB_OPEN )
   END_RUNG wire#w15
   RUNG wire#powerrail
      Contact( "IO_Valve_Storage_DB"."AV-35.05".FB_OPEN )
      wire#w16
      Coil( "T-35.00".State."Line_AV5&AV6" )
   END_RUNG
   RUNG wire#powerrail
      Contact( "IO_Valve_Storage_DB"."AV-35.06".FB_OPEN )
   END_RUNG wire#w16
   // the same network as SCL:
   "T-33.00".State."Line_AV4&AV5" := "IO_Valve_Storage_DB"."AV-33.04".FB_OPEN OR "IO_Valve_Storage_DB"."AV-33.05".FB_OPEN;
   "T-34.00".State."Line_AV4&AV5" := "IO_Valve_Storage_DB"."AV-34.04".FB_OPEN OR "IO_Valve_Storage_DB"."AV-34.05".FB_OPEN;
   "T-35.00".State."Line_AV4&AV5" := "IO_Valve_Storage_DB"."AV-35.04".FB_OPEN OR "IO_Valve_Storage_DB"."AV-35.05".FB_OPEN;
   "T-39.00".State."Line_AV1&AV2" := "IO_Valve_Storage_DB"."AV-39.01".FB_OPEN OR "IO_Valve_Storage_DB"."AV-39.02".FB_OPEN;
   "T-33.00".State."Line_AV7&AV8" := "IO_Valve_Storage_DB"."AV-33.07".FB_OPEN OR "IO_Valve_Storage_DB"."AV-33.08".FB_OPEN;
   "T-34.00".State."Line_AV7&AV8" := "IO_Valve_Storage_DB"."AV-34.07".FB_OPEN OR "IO_Valve_Storage_DB"."AV-34.08".FB_OPEN;
   "T-35.00".State."Line_AV7&AV8" := "IO_Valve_Storage_DB"."AV-35.07".FB_OPEN OR "IO_Valve_Storage_DB"."AV-35.08".FB_OPEN;
   "T-33.00".State."Line_AV10&AV11" := "IO_Valve_Storage_DB"."AV-33.11".FB_OPEN OR "IO_Valve_Storage_DB"."AV-33.10".FB_OPEN;
   "T-34.00".State."Line_AV10&AV11" := "T-33.00".State."Line_AV10&AV11" OR "IO_Valve_Storage_DB"."AV-34.10".FB_OPEN;
   "T-33.00".State.CIP_Line1_ON := "IO_Valve_Storage_DB"."AV-33.11".FB_OPEN OR "IO_Valve_Storage_DB"."AV-33.05".FB_OPEN OR "IO_Valve_Storage_DB"."AV-33.06".FB_OPEN OR "IO_Valve_Storage_DB"."AV-34.05".FB_OPEN OR "IO_Valve_Storage_DB"."AV-34.06".FB_OPEN OR "IO_Valve_Storage_DB"."AV-35.05".FB_OPEN OR "IO_Valve_Storage_DB"."AV-35.06".FB_OPEN OR "IO_Valve_Storage_DB"."AV-35.08".FB_OPEN;
   "T-33.00".State.CIP_Line2_ON := "IO_Valve_Storage_DB"."AV-33.05".FB_OPEN OR "IO_Valve_Storage_DB"."AV-33.06".FB_OPEN OR "IO_Valve_Storage_DB"."AV-34.05".FB_OPEN OR "IO_Valve_Storage_DB"."AV-34.06".FB_OPEN OR "IO_Valve_Storage_DB"."AV-35.05".FB_OPEN OR "IO_Valve_Storage_DB"."AV-35.06".FB_OPEN OR "IO_Valve_Storage_DB"."AV-35.08".FB_OPEN;
   "T-33.00".State."Line_AV5&AV6" := "IO_Valve_Storage_DB"."AV-33.05".FB_OPEN OR "IO_Valve_Storage_DB"."AV-33.06".FB_OPEN;
   "T-34.00".State.CIP_Line1_ON := "IO_Valve_Storage_DB"."AV-34.05".FB_OPEN OR "IO_Valve_Storage_DB"."AV-34.06".FB_OPEN OR "IO_Valve_Storage_DB"."AV-35.05".FB_OPEN OR "IO_Valve_Storage_DB"."AV-35.06".FB_OPEN OR "IO_Valve_Storage_DB"."AV-35.08".FB_OPEN;
   "T-34.00".State."Line_AV5&AV6" := "IO_Valve_Storage_DB"."AV-34.05".FB_OPEN OR "IO_Valve_Storage_DB"."AV-34.06".FB_OPEN;
   "T-35.00".State.CIP_Line1_ON := "IO_Valve_Storage_DB"."AV-35.05".FB_OPEN OR "IO_Valve_Storage_DB"."AV-35.06".FB_OPEN OR "IO_Valve_Storage_DB"."AV-35.08".FB_OPEN;
   "T-35.00".State."Line_AV5&AV6" := "IO_Valve_Storage_DB"."AV-35.05".FB_OPEN OR "IO_Valve_Storage_DB"."AV-35.06".FB_OPEN;
END_REGION

REGION Network 32: T-81.00
   // Inload 1 : PHE-2
   // Inload 2 : THE-1
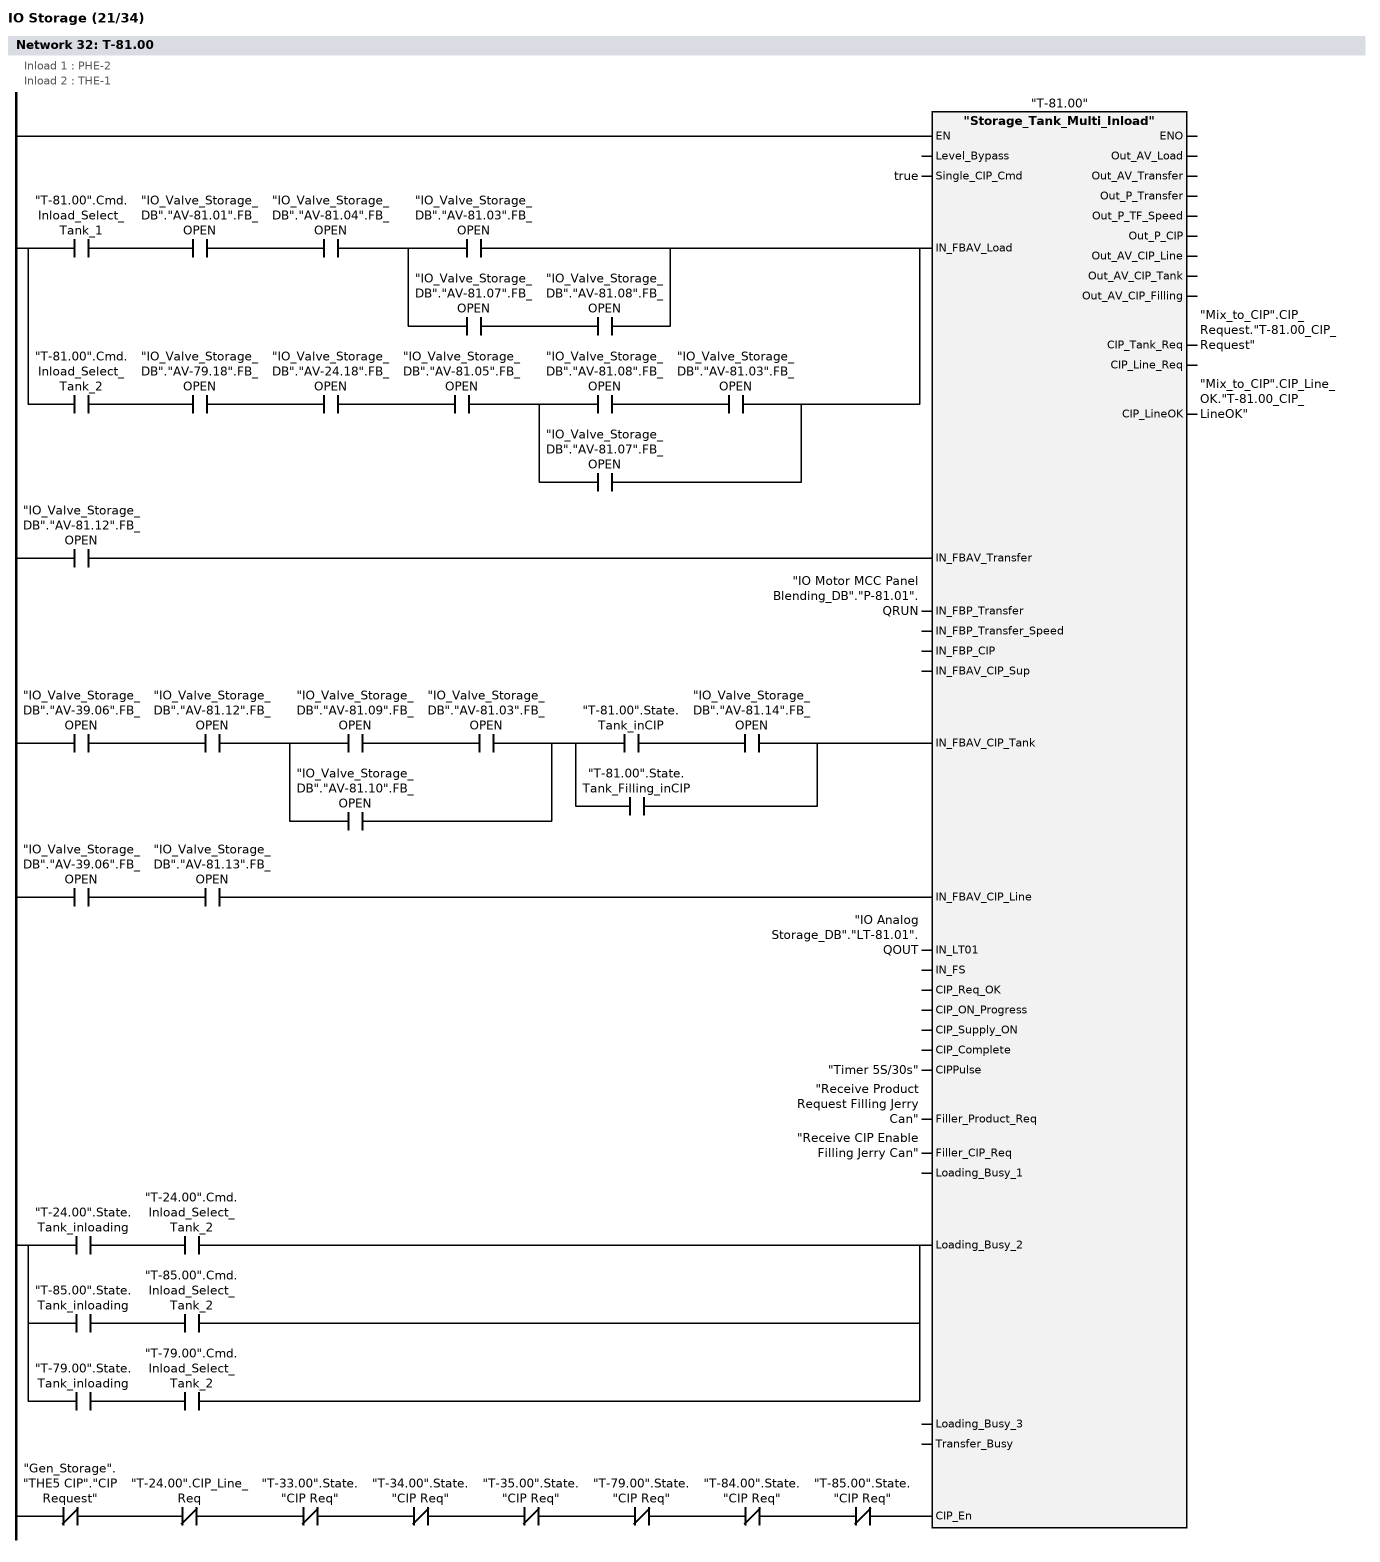
   RUNG wire#powerrail
      "T-81.00"(IN_FBAV_Load := wire#w3, IN_FBAV_Transfer := wire#w4, IN_FBAV_CIP_Tank := wire#w7, IN_FBAV_CIP_Line := wire#w8, Loading_Busy_2 := wire#w9, CIP_En := wire#w10, Level_Bypass :=, Single_CIP_Cmd := true, IN_FBP_Transfer := "IO Motor MCC Panel Blending_DB"."P-81.01".QRUN, IN_FBP_Transfer_Speed :=, IN_FBP_CIP :=, IN_FBAV_CIP_Sup :=, IN_LT01 := "IO Analog Storage_DB"."LT-81.01".QOUT, IN_FS :=, CIP_Req_OK :=, CIP_ON_Progress :=, CIP_Supply_ON :=, CIP_Complete :=, CIPPulse := "Timer 5S/30s", Filler_Product_Req := "Receive Product Request Filling Jerry Can", Filler_CIP_Req := "Receive CIP Enable Filling Jerry Can", Loading_Busy_1 :=, Loading_Busy_3 :=, Transfer_Busy :=, Out_AV_Load =>, Out_AV_Transfer =>, Out_P_Transfer =>, Out_P_TF_Speed =>, Out_P_CIP =>, Out_AV_CIP_Line =>, Out_AV_CIP_Tank =>, Out_AV_CIP_Filling =>, CIP_Tank_Req => "Mix_to_CIP".CIP_Request."T-81.00_CIP_Request", CIP_Line_Req =>, CIP_LineOK => "Mix_to_CIP".CIP_Line_OK."T-81.00_CIP_LineOK")
   END_RUNG
   RUNG wire#powerrail
      Contact( "T-81.00".Cmd.Inload_Select_Tank_1 )
      Contact( "IO_Valve_Storage_DB"."AV-81.01".FB_OPEN )
      Contact( "IO_Valve_Storage_DB"."AV-81.04".FB_OPEN )
      wire#w1
      Contact( "IO_Valve_Storage_DB"."AV-81.03".FB_OPEN )
   END_RUNG wire#w3
   RUNG wire#w1
      Contact( "IO_Valve_Storage_DB"."AV-81.07".FB_OPEN )
      Contact( "IO_Valve_Storage_DB"."AV-81.08".FB_OPEN )
   END_RUNG wire#w3
   RUNG wire#powerrail
      Contact( "T-81.00".Cmd.Inload_Select_Tank_2 )
      Contact( "IO_Valve_Storage_DB"."AV-79.18".FB_OPEN )
      Contact( "IO_Valve_Storage_DB"."AV-24.18".FB_OPEN )
      Contact( "IO_Valve_Storage_DB"."AV-81.05".FB_OPEN )
      wire#w2
      Contact( "IO_Valve_Storage_DB"."AV-81.08".FB_OPEN )
      Contact( "IO_Valve_Storage_DB"."AV-81.03".FB_OPEN )
   END_RUNG wire#w3
   RUNG wire#w2
      Contact( "IO_Valve_Storage_DB"."AV-81.07".FB_OPEN )
   END_RUNG wire#w3
   RUNG wire#powerrail
      Contact( "IO_Valve_Storage_DB"."AV-81.12".FB_OPEN )
   END_RUNG wire#w4
   RUNG wire#powerrail
      Contact( "IO_Valve_Storage_DB"."AV-39.06".FB_OPEN )
      Contact( "IO_Valve_Storage_DB"."AV-81.12".FB_OPEN )
      wire#w5
      Contact( "IO_Valve_Storage_DB"."AV-81.09".FB_OPEN )
      Contact( "IO_Valve_Storage_DB"."AV-81.03".FB_OPEN )
      wire#w6
      Contact( "T-81.00".State.Tank_inCIP )
      Contact( "IO_Valve_Storage_DB"."AV-81.14".FB_OPEN )
   END_RUNG wire#w7
   RUNG wire#w5
      Contact( "IO_Valve_Storage_DB"."AV-81.10".FB_OPEN )
   END_RUNG wire#w6
   RUNG wire#w6
      Contact( "T-81.00".State.Tank_Filling_inCIP )
   END_RUNG wire#w7
   RUNG wire#powerrail
      Contact( "IO_Valve_Storage_DB"."AV-39.06".FB_OPEN )
      Contact( "IO_Valve_Storage_DB"."AV-81.13".FB_OPEN )
   END_RUNG wire#w8
   RUNG wire#powerrail
      Contact( "T-24.00".State.Tank_inloading )
      Contact( "T-24.00".Cmd.Inload_Select_Tank_2 )
   END_RUNG wire#w9
   RUNG wire#powerrail
      Contact( "T-85.00".State.Tank_inloading )
      Contact( "T-85.00".Cmd.Inload_Select_Tank_2 )
   END_RUNG wire#w9
   RUNG wire#powerrail
      Contact( "T-79.00".State.Tank_inloading )
      Contact( "T-79.00".Cmd.Inload_Select_Tank_2 )
   END_RUNG wire#w9
   RUNG wire#powerrail
      I_Contact( "Gen_Storage"."THE5 CIP"."CIP Request" )
      I_Contact( "T-24.00".CIP_Line_Req )
      I_Contact( "T-33.00".State."CIP Req" )
      I_Contact( "T-34.00".State."CIP Req" )
      I_Contact( "T-35.00".State."CIP Req" )
      I_Contact( "T-79.00".State."CIP Req" )
      I_Contact( "T-84.00".State."CIP Req" )
      I_Contact( "T-85.00".State."CIP Req" )
   END_RUNG wire#w10
   // the same network as SCL:
   "T-81.00"(Single_CIP_Cmd := true,   // "Storage_Tank_Multi_Inload"
             IN_FBAV_Load := ("T-81.00".Cmd.Inload_Select_Tank_1 AND "IO_Valve_Storage_DB"."AV-81.01".FB_OPEN AND "IO_Valve_Storage_DB"."AV-81.04".FB_OPEN AND ("IO_Valve_Storage_DB"."AV-81.03".FB_OPEN OR ("IO_Valve_Storage_DB"."AV-81.07".FB_OPEN AND "IO_Valve_Storage_DB"."AV-81.08".FB_OPEN))) OR ("T-81.00".Cmd.Inload_Select_Tank_2 AND "IO_Valve_Storage_DB"."AV-79.18".FB_OPEN AND "IO_Valve_Storage_DB"."AV-24.18".FB_OPEN AND "IO_Valve_Storage_DB"."AV-81.05".FB_OPEN AND (("IO_Valve_Storage_DB"."AV-81.08".FB_OPEN AND "IO_Valve_Storage_DB"."AV-81.03".FB_OPEN) OR "IO_Valve_Storage_DB"."AV-81.07".FB_OPEN)),
             IN_FBAV_Transfer := "IO_Valve_Storage_DB"."AV-81.12".FB_OPEN,
             IN_FBP_Transfer := "IO Motor MCC Panel Blending_DB"."P-81.01".QRUN,
             IN_FBAV_CIP_Tank := "IO_Valve_Storage_DB"."AV-39.06".FB_OPEN AND "IO_Valve_Storage_DB"."AV-81.12".FB_OPEN AND (("IO_Valve_Storage_DB"."AV-81.09".FB_OPEN AND "IO_Valve_Storage_DB"."AV-81.03".FB_OPEN) OR "IO_Valve_Storage_DB"."AV-81.10".FB_OPEN) AND (("T-81.00".State.Tank_inCIP AND "IO_Valve_Storage_DB"."AV-81.14".FB_OPEN) OR "T-81.00".State.Tank_Filling_inCIP),
             IN_FBAV_CIP_Line := "IO_Valve_Storage_DB"."AV-39.06".FB_OPEN AND "IO_Valve_Storage_DB"."AV-81.13".FB_OPEN,
             IN_LT01 := "IO Analog Storage_DB"."LT-81.01".QOUT,
             CIPPulse := "Timer 5S/30s",
             Filler_Product_Req := "Receive Product Request Filling Jerry Can",
             Filler_CIP_Req := "Receive CIP Enable Filling Jerry Can",
             Loading_Busy_2 := ("T-24.00".State.Tank_inloading AND "T-24.00".Cmd.Inload_Select_Tank_2) OR ("T-85.00".State.Tank_inloading AND "T-85.00".Cmd.Inload_Select_Tank_2) OR ("T-79.00".State.Tank_inloading AND "T-79.00".Cmd.Inload_Select_Tank_2),
             CIP_En := NOT "Gen_Storage"."THE5 CIP"."CIP Request" AND NOT "T-24.00".CIP_Line_Req AND NOT "T-33.00".State."CIP Req" AND NOT "T-34.00".State."CIP Req" AND NOT "T-35.00".State."CIP Req" AND NOT "T-79.00".State."CIP Req" AND NOT "T-84.00".State."CIP Req" AND NOT "T-85.00".State."CIP Req",
             CIP_Tank_Req => "Mix_to_CIP".CIP_Request."T-81.00_CIP_Request",
             CIP_LineOK => "Mix_to_CIP".CIP_Line_OK."T-81.00_CIP_LineOK");
END_REGION

REGION Network 33: T-81 Valve
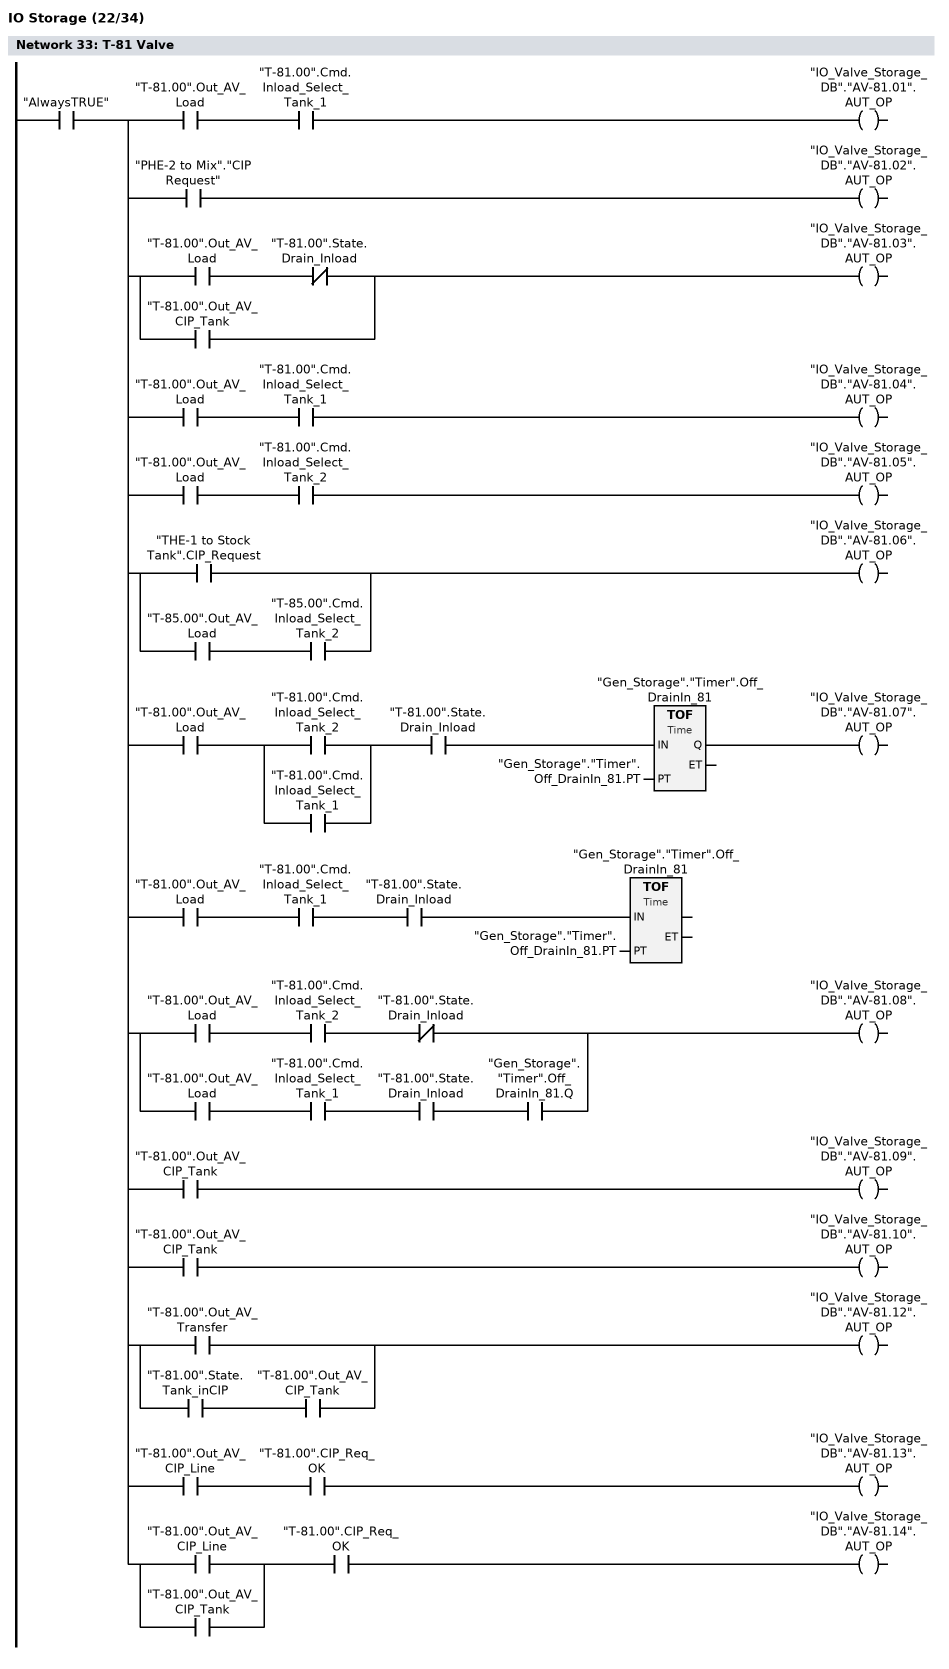
   RUNG wire#powerrail
      Contact( "AlwaysTRUE" )
      wire#w1
      Contact( "T-81.00".Out_AV_Load )
      Contact( "T-81.00".Cmd.Inload_Select_Tank_1 )
      Coil( "IO_Valve_Storage_DB"."AV-81.01".AUT_OP )
   END_RUNG
   RUNG wire#w1
      Contact( "PHE-2 to Mix"."CIP Request" )
      Coil( "IO_Valve_Storage_DB"."AV-81.02".AUT_OP )
   END_RUNG
   RUNG wire#w1
      Contact( "T-81.00".Out_AV_Load )
      I_Contact( "T-81.00".State.Drain_Inload )
      wire#w2
      Coil( "IO_Valve_Storage_DB"."AV-81.03".AUT_OP )
   END_RUNG
   RUNG wire#w1
      Contact( "T-81.00".Out_AV_CIP_Tank )
   END_RUNG wire#w2
   RUNG wire#w1
      Contact( "T-81.00".Out_AV_Load )
      Contact( "T-81.00".Cmd.Inload_Select_Tank_1 )
      Coil( "IO_Valve_Storage_DB"."AV-81.04".AUT_OP )
   END_RUNG
   RUNG wire#w1
      Contact( "T-81.00".Out_AV_Load )
      Contact( "T-81.00".Cmd.Inload_Select_Tank_2 )
      Coil( "IO_Valve_Storage_DB"."AV-81.05".AUT_OP )
   END_RUNG
   RUNG wire#w1
      Contact( "THE-1 to Stock Tank".CIP_Request )
      wire#w3
      Coil( "IO_Valve_Storage_DB"."AV-81.06".AUT_OP )
   END_RUNG
   RUNG wire#w1
      Contact( "T-85.00".Out_AV_Load )
      Contact( "T-85.00".Cmd.Inload_Select_Tank_2 )
   END_RUNG wire#w3
   RUNG wire#w1
      Contact( "T-81.00".Out_AV_Load )
      wire#w4
      Contact( "T-81.00".Cmd.Inload_Select_Tank_2 )
      wire#w5
      Contact( "T-81.00".State.Drain_Inload )
      { S7_Templates := "time_type := Time" } "Gen_Storage"."Timer".Off_DrainIn_81.TOF(pt := "Gen_Storage"."Timer".Off_DrainIn_81.PT, et =>)
      Coil( "IO_Valve_Storage_DB"."AV-81.07".AUT_OP )
   END_RUNG
   RUNG wire#w4
      Contact( "T-81.00".Cmd.Inload_Select_Tank_1 )
   END_RUNG wire#w5
   RUNG wire#w1
      Contact( "T-81.00".Out_AV_Load )
      Contact( "T-81.00".Cmd.Inload_Select_Tank_1 )
      Contact( "T-81.00".State.Drain_Inload )
      { S7_Templates := "time_type := Time" } "Gen_Storage"."Timer".Off_DrainIn_81.TOF(pt := "Gen_Storage"."Timer".Off_DrainIn_81.PT, et =>)
   END_RUNG
   RUNG wire#w1
      Contact( "T-81.00".Out_AV_Load )
      Contact( "T-81.00".Cmd.Inload_Select_Tank_2 )
      I_Contact( "T-81.00".State.Drain_Inload )
      wire#w6
      Coil( "IO_Valve_Storage_DB"."AV-81.08".AUT_OP )
   END_RUNG
   RUNG wire#w1
      Contact( "T-81.00".Out_AV_Load )
      Contact( "T-81.00".Cmd.Inload_Select_Tank_1 )
      Contact( "T-81.00".State.Drain_Inload )
      Contact( "Gen_Storage"."Timer".Off_DrainIn_81.Q )
   END_RUNG wire#w6
   RUNG wire#w1
      Contact( "T-81.00".Out_AV_CIP_Tank )
      Coil( "IO_Valve_Storage_DB"."AV-81.09".AUT_OP )
   END_RUNG
   RUNG wire#w1
      Contact( "T-81.00".Out_AV_CIP_Tank )
      Coil( "IO_Valve_Storage_DB"."AV-81.10".AUT_OP )
   END_RUNG
   RUNG wire#w1
      Contact( "T-81.00".Out_AV_Transfer )
      wire#w7
      Coil( "IO_Valve_Storage_DB"."AV-81.12".AUT_OP )
   END_RUNG
   RUNG wire#w1
      Contact( "T-81.00".State.Tank_inCIP )
      Contact( "T-81.00".Out_AV_CIP_Tank )
   END_RUNG wire#w7
   RUNG wire#w1
      Contact( "T-81.00".Out_AV_CIP_Line )
      Contact( "T-81.00".CIP_Req_OK )
      Coil( "IO_Valve_Storage_DB"."AV-81.13".AUT_OP )
   END_RUNG
   RUNG wire#w1
      Contact( "T-81.00".Out_AV_CIP_Line )
      wire#w8
      Contact( "T-81.00".CIP_Req_OK )
      Coil( "IO_Valve_Storage_DB"."AV-81.14".AUT_OP )
   END_RUNG
   RUNG wire#w1
      Contact( "T-81.00".Out_AV_CIP_Tank )
   END_RUNG wire#w8
   // the same network as SCL:
   "IO_Valve_Storage_DB"."AV-81.01".AUT_OP := "AlwaysTRUE" AND "T-81.00".Out_AV_Load AND "T-81.00".Cmd.Inload_Select_Tank_1;
   "IO_Valve_Storage_DB"."AV-81.02".AUT_OP := "AlwaysTRUE" AND "PHE-2 to Mix"."CIP Request";
   "IO_Valve_Storage_DB"."AV-81.03".AUT_OP := "AlwaysTRUE" AND (("T-81.00".Out_AV_Load AND NOT "T-81.00".State.Drain_Inload) OR "T-81.00".Out_AV_CIP_Tank);
   "IO_Valve_Storage_DB"."AV-81.04".AUT_OP := "AlwaysTRUE" AND "T-81.00".Out_AV_Load AND "T-81.00".Cmd.Inload_Select_Tank_1;
   "IO_Valve_Storage_DB"."AV-81.05".AUT_OP := "AlwaysTRUE" AND "T-81.00".Out_AV_Load AND "T-81.00".Cmd.Inload_Select_Tank_2;
   "IO_Valve_Storage_DB"."AV-81.06".AUT_OP := "AlwaysTRUE" AND ("THE-1 to Stock Tank".CIP_Request OR ("T-85.00".Out_AV_Load AND "T-85.00".Cmd.Inload_Select_Tank_2));
   "Gen_Storage"."Timer".Off_DrainIn_81.TOF(IN := "AlwaysTRUE" AND "T-81.00".Out_AV_Load AND ("T-81.00".Cmd.Inload_Select_Tank_2 OR "T-81.00".Cmd.Inload_Select_Tank_1) AND "T-81.00".State.Drain_Inload,
                           PT := "Gen_Storage"."Timer".Off_DrainIn_81.PT);
   "IO_Valve_Storage_DB"."AV-81.07".AUT_OP := "Gen_Storage"."Timer".Off_DrainIn_81.Q;
   "Gen_Storage"."Timer".Off_DrainIn_81.TOF(IN := "AlwaysTRUE" AND "T-81.00".Out_AV_Load AND "T-81.00".Cmd.Inload_Select_Tank_1 AND "T-81.00".State.Drain_Inload,
                           PT := "Gen_Storage"."Timer".Off_DrainIn_81.PT);
   "IO_Valve_Storage_DB"."AV-81.08".AUT_OP := "AlwaysTRUE" AND (("T-81.00".Out_AV_Load AND "T-81.00".Cmd.Inload_Select_Tank_2 AND NOT "T-81.00".State.Drain_Inload) OR ("T-81.00".Out_AV_Load AND "T-81.00".Cmd.Inload_Select_Tank_1 AND "T-81.00".State.Drain_Inload AND "Gen_Storage"."Timer".Off_DrainIn_81.Q));
   "IO_Valve_Storage_DB"."AV-81.09".AUT_OP := "AlwaysTRUE" AND "T-81.00".Out_AV_CIP_Tank;
   "IO_Valve_Storage_DB"."AV-81.10".AUT_OP := "AlwaysTRUE" AND "T-81.00".Out_AV_CIP_Tank;
   "IO_Valve_Storage_DB"."AV-81.12".AUT_OP := "AlwaysTRUE" AND ("T-81.00".Out_AV_Transfer OR ("T-81.00".State.Tank_inCIP AND "T-81.00".Out_AV_CIP_Tank));
   "IO_Valve_Storage_DB"."AV-81.13".AUT_OP := "AlwaysTRUE" AND "T-81.00".Out_AV_CIP_Line AND "T-81.00".CIP_Req_OK;
   "IO_Valve_Storage_DB"."AV-81.14".AUT_OP := "AlwaysTRUE" AND ("T-81.00".Out_AV_CIP_Line OR "T-81.00".Out_AV_CIP_Tank) AND "T-81.00".CIP_Req_OK;
END_REGION

REGION Network 34: Comm T-81 to THE-1
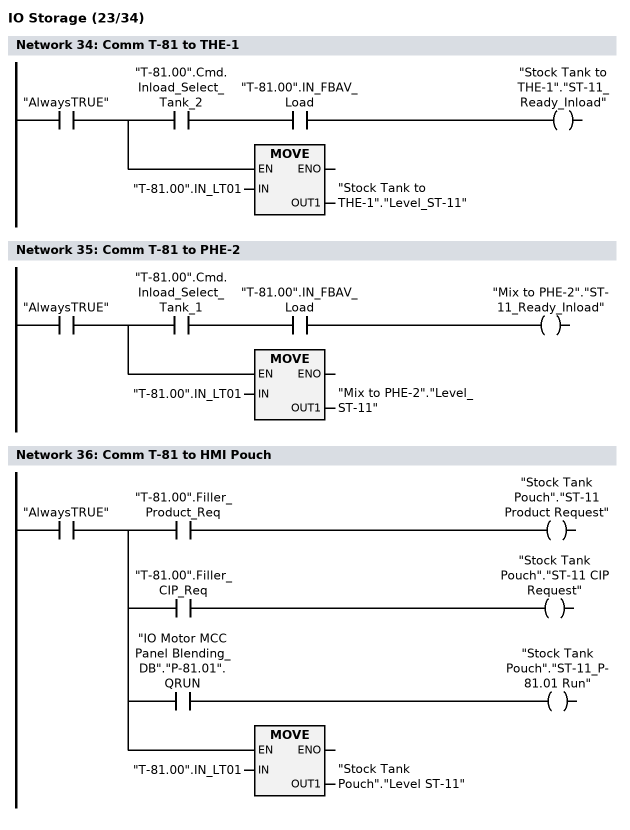
   RUNG wire#powerrail
      Contact( "AlwaysTRUE" )
      wire#w1
      Contact( "T-81.00".Cmd.Inload_Select_Tank_2 )
      Contact( "T-81.00".IN_FBAV_Load )
      Coil( "Stock Tank to THE-1"."ST-11_Ready_Inload" )
   END_RUNG
   RUNG wire#w1
      Move(in := "T-81.00".IN_LT01, out1 => "Stock Tank to THE-1"."Level_ST-11")
   END_RUNG
   // the same network as SCL:
   "Stock Tank to THE-1"."ST-11_Ready_Inload" := "AlwaysTRUE" AND "T-81.00".Cmd.Inload_Select_Tank_2 AND "T-81.00".IN_FBAV_Load;
   IF "AlwaysTRUE" THEN "Stock Tank to THE-1"."Level_ST-11" := "T-81.00".IN_LT01; END_IF;
END_REGION

REGION Network 35: Comm T-81 to PHE-2
   RUNG wire#powerrail
      Contact( "AlwaysTRUE" )
      wire#w1
      Contact( "T-81.00".Cmd.Inload_Select_Tank_1 )
      Contact( "T-81.00".IN_FBAV_Load )
      Coil( "Mix to PHE-2"."ST-11_Ready_Inload" )
   END_RUNG
   RUNG wire#w1
      Move(in := "T-81.00".IN_LT01, out1 => "Mix to PHE-2"."Level_ST-11")
   END_RUNG
   // the same network as SCL:
   "Mix to PHE-2"."ST-11_Ready_Inload" := "AlwaysTRUE" AND "T-81.00".Cmd.Inload_Select_Tank_1 AND "T-81.00".IN_FBAV_Load;
   IF "AlwaysTRUE" THEN "Mix to PHE-2"."Level_ST-11" := "T-81.00".IN_LT01; END_IF;
END_REGION

REGION Network 36: Comm T-81 to HMI Pouch
   RUNG wire#powerrail
      Contact( "AlwaysTRUE" )
      wire#w1
      Contact( "T-81.00".Filler_Product_Req )
      Coil( "Stock Tank Pouch"."ST-11 Product Request" )
   END_RUNG
   RUNG wire#w1
      Contact( "T-81.00".Filler_CIP_Req )
      Coil( "Stock Tank Pouch"."ST-11 CIP Request" )
   END_RUNG
   RUNG wire#w1
      Contact( "IO Motor MCC Panel Blending_DB"."P-81.01".QRUN )
      Coil( "Stock Tank Pouch"."ST-11_P-81.01 Run" )
   END_RUNG
   RUNG wire#w1
      Move(in := "T-81.00".IN_LT01, out1 => "Stock Tank Pouch"."Level ST-11")
   END_RUNG
   // the same network as SCL:
   "Stock Tank Pouch"."ST-11 Product Request" := "AlwaysTRUE" AND "T-81.00".Filler_Product_Req;
   "Stock Tank Pouch"."ST-11 CIP Request" := "AlwaysTRUE" AND "T-81.00".Filler_CIP_Req;
   "Stock Tank Pouch"."ST-11_P-81.01 Run" := "AlwaysTRUE" AND "IO Motor MCC Panel Blending_DB"."P-81.01".QRUN;
   IF "AlwaysTRUE" THEN "Stock Tank Pouch"."Level ST-11" := "T-81.00".IN_LT01; END_IF;
END_REGION

REGION Network 38: T-85.00 ST-16
   // Inload 1 : PHE-1
   // Inload 2 : THE-1
   // Inload 3 : THE-3
